REGION Network 14: CYL 6 COUNTER
   RUNG wire#powerrail
      Contact( "AlwaysTRUE" )
      Contact( #ENABLE_CYLINDER[6] )
      Contact( #CYCLE_OK )
      Contact( #CYL_SENSOR6 )
      { S7_Templates := "time_type := Time" } #CYL_STAB_S6.TON(pt := #"SENSING TIME", et =>)
      wire#w1
      Contact( #FIRST_CYCLE )
      P_Trig( #"PLUS BIT"[11] )
      { S7_Templates := "SrcType := Int" } NE_Contact(in1 := #CYL_COUNTER_S6.CV, in2 := #First_Cylinder[6])
      { S7_Templates := "value_type := Int" } #CYL_COUNTER_S6.CTU(r := #"COUNTER RESET", pv := #First_Cylinder[6], cv =>)
   END_RUNG
   RUNG wire#w1
      Contact( #CYCLE_RESTART )
      P_Trig( #"PLUS BIT"[12] )
      { S7_Templates := "SrcType := Int" } NE_Contact(in1 := #CYL_COUNT_CONT_S6.CV, in2 := #"CYL COUNT  VALUE")
      { S7_Templates := "value_type := Int" } #CYL_COUNT_CONT_S6.CTU(r := #"COUNTER RESET", pv := #"CYL COUNT  VALUE", cv =>)
   END_RUNG
   // the same network as SCL:
   #CYL_STAB_S6(IN := "AlwaysTRUE" AND #ENABLE_CYLINDER[6] AND #CYCLE_OK AND #CYL_SENSOR6,   // TON
                PT := #"SENSING TIME");
   #_w1 := #CYL_STAB_S6.Q AND #FIRST_CYCLE;
   #_w2 := #_w1 AND NOT #"PLUS BIT"[11];   // rising edge
   #"PLUS BIT"[11] := #_w1;
   #CYL_COUNTER_S6(CU := #_w2 AND (#CYL_COUNTER_S6.CV <> #First_Cylinder[6]),   // CTU
                   R := #"COUNTER RESET",
                   PV := #First_Cylinder[6]);
   #_w3 := #CYL_STAB_S6.Q AND #CYCLE_RESTART;
   #_w4 := #_w3 AND NOT #"PLUS BIT"[12];   // rising edge
   #"PLUS BIT"[12] := #_w3;
   #CYL_COUNT_CONT_S6(CU := #_w4 AND (#CYL_COUNT_CONT_S6.CV <> #"CYL COUNT  VALUE"),   // CTU
                      R := #"COUNTER RESET",
                      PV := #"CYL COUNT  VALUE");
END_REGION

REGION Network 15: CYL 11 COUNTER
   RUNG wire#powerrail
      Contact( "AlwaysFALSE" )
      Contact( #CYCLE_OK )
      Contact( #"DOWN CONVEYOR" )
      { S7_Templates := "value_type := Int" } #CYL_COUNTER_S11.CTU(r := #"COUNTER RESET", pv := #"CYL COUNT  VALUE", cv =>)
   END_RUNG
   // the same network as SCL:
   #CYL_COUNTER_S11(CU := "AlwaysFALSE" AND #CYCLE_OK AND #"DOWN CONVEYOR",   // CTU
                    R := #"COUNTER RESET",
                    PV := #"CYL COUNT  VALUE");
END_REGION

REGION Network 16: CYL 1 LOCK
   RUNG wire#powerrail
      Contact( "AlwaysTRUE" )
      Contact( #ENABLE_CYLINDER[1] )
      Contact( #CYCLE_OK )
      wire#w1
      Contact( #FIRST_CYCLE )
      { S7_Templates := "SrcType := Int" } EQ_Contact(in1 := #CYL_COUNTER_S1.CV, in2 := #First_Cylinder[1])
      wire#w2
      S_Coil( #"LIFT TABLE1" )
      { S7_Templates := "time_type := Time" } #FILL_STT_1.TON(pt := T#0S, et =>)
      P_Trig( #"PLUS BIT"[31] )
      Contact( #AUTO )
      S_Coil( #FILL_STT_SEQ1 )
   END_RUNG
   RUNG wire#w1
      Contact( #CYCLE_RESTART )
      { S7_Templates := "SrcType := Int" } EQ_Contact(in1 := #CYL_COUNT_CONT_S1.CV, in2 := #"CYL COUNT  VALUE")
   END_RUNG wire#w2
   RUNG wire#w2
      Contact( "Tag_75" )
      S_Coil( #GUN_DOWN1 )
   END_RUNG
   // the same network as SCL:
   #_w1 := "AlwaysTRUE" AND #ENABLE_CYLINDER[1] AND #CYCLE_OK AND ((#FIRST_CYCLE AND (#CYL_COUNTER_S1.CV = #First_Cylinder[1])) OR (#CYCLE_RESTART AND (#CYL_COUNT_CONT_S1.CV = #"CYL COUNT  VALUE")));
   IF #_w1 THEN #"LIFT TABLE1" := TRUE; END_IF;
   #FILL_STT_1(IN := #_w1, PT := T#0S);   // TON
   #_w2 := #FILL_STT_1.Q AND NOT #"PLUS BIT"[31];   // rising edge
   #"PLUS BIT"[31] := #FILL_STT_1.Q;
   IF #_w2 AND #AUTO THEN #FILL_STT_SEQ1 := TRUE; END_IF;
   IF #_w1 AND "Tag_75" THEN #GUN_DOWN1 := TRUE; END_IF;
END_REGION

REGION Network 17: CYL 2 LOCK
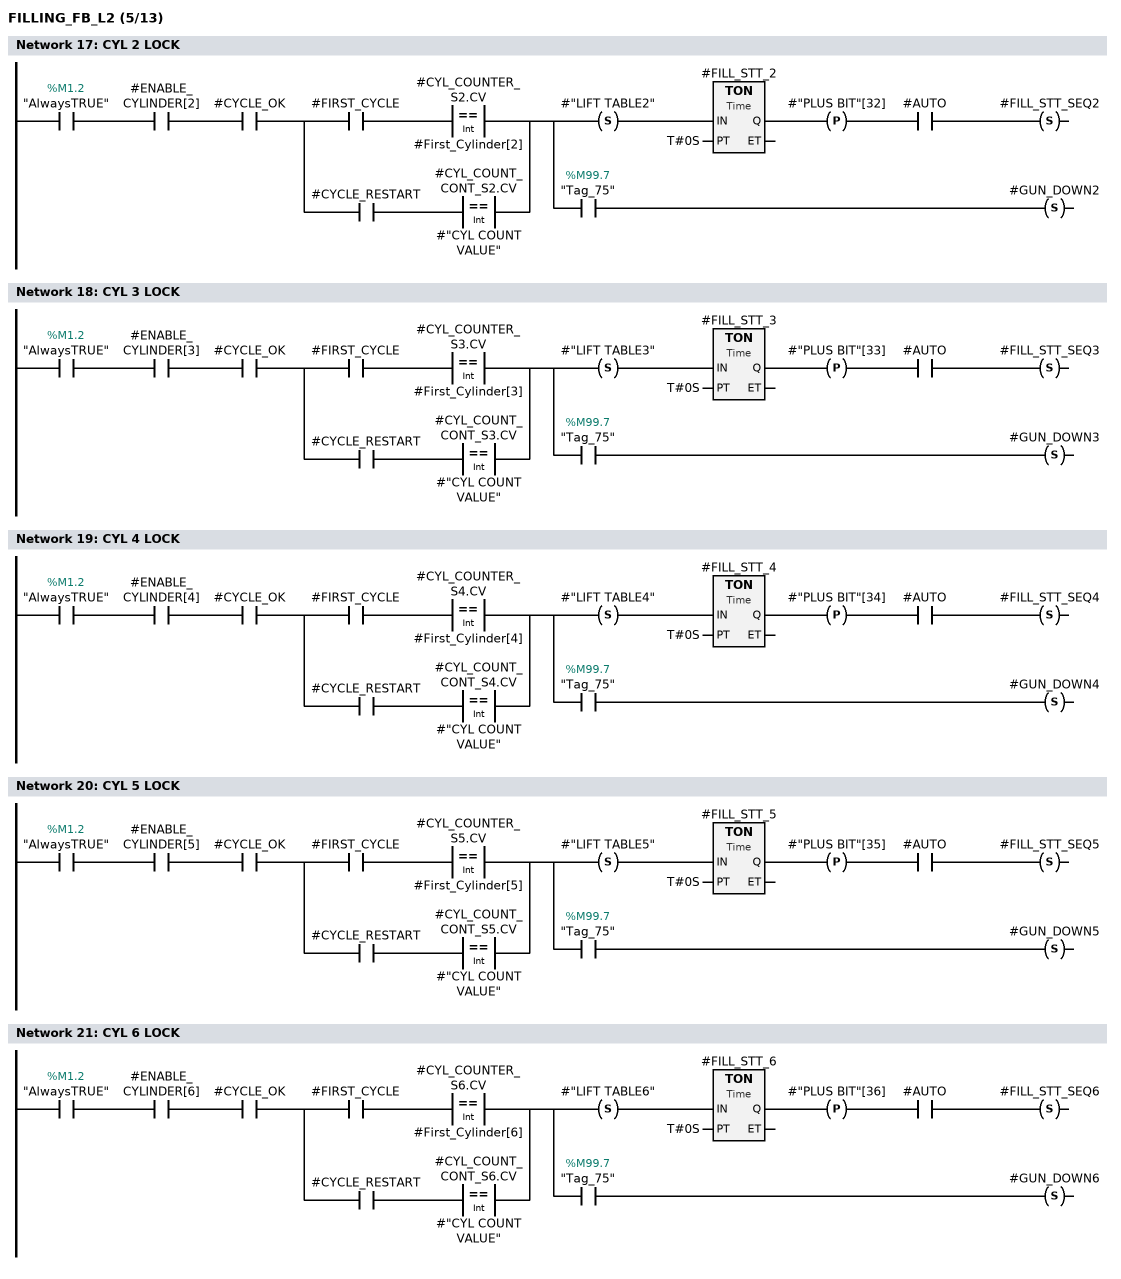
   RUNG wire#powerrail
      Contact( "AlwaysTRUE" )
      Contact( #ENABLE_CYLINDER[2] )
      Contact( #CYCLE_OK )
      wire#w1
      Contact( #FIRST_CYCLE )
      { S7_Templates := "SrcType := Int" } EQ_Contact(in1 := #CYL_COUNTER_S2.CV, in2 := #First_Cylinder[2])
      wire#w2
      S_Coil( #"LIFT TABLE2" )
      { S7_Templates := "time_type := Time" } #FILL_STT_2.TON(pt := T#0S, et =>)
      P_Trig( #"PLUS BIT"[32] )
      Contact( #AUTO )
      S_Coil( #FILL_STT_SEQ2 )
   END_RUNG
   RUNG wire#w1
      Contact( #CYCLE_RESTART )
      { S7_Templates := "SrcType := Int" } EQ_Contact(in1 := #CYL_COUNT_CONT_S2.CV, in2 := #"CYL COUNT  VALUE")
   END_RUNG wire#w2
   RUNG wire#w2
      Contact( "Tag_75" )
      S_Coil( #GUN_DOWN2 )
   END_RUNG
   // the same network as SCL:
   #_w1 := "AlwaysTRUE" AND #ENABLE_CYLINDER[2] AND #CYCLE_OK AND ((#FIRST_CYCLE AND (#CYL_COUNTER_S2.CV = #First_Cylinder[2])) OR (#CYCLE_RESTART AND (#CYL_COUNT_CONT_S2.CV = #"CYL COUNT  VALUE")));
   IF #_w1 THEN #"LIFT TABLE2" := TRUE; END_IF;
   #FILL_STT_2(IN := #_w1, PT := T#0S);   // TON
   #_w2 := #FILL_STT_2.Q AND NOT #"PLUS BIT"[32];   // rising edge
   #"PLUS BIT"[32] := #FILL_STT_2.Q;
   IF #_w2 AND #AUTO THEN #FILL_STT_SEQ2 := TRUE; END_IF;
   IF #_w1 AND "Tag_75" THEN #GUN_DOWN2 := TRUE; END_IF;
END_REGION

REGION Network 18: CYL 3 LOCK
   RUNG wire#powerrail
      Contact( "AlwaysTRUE" )
      Contact( #ENABLE_CYLINDER[3] )
      Contact( #CYCLE_OK )
      wire#w1
      Contact( #FIRST_CYCLE )
      { S7_Templates := "SrcType := Int" } EQ_Contact(in1 := #CYL_COUNTER_S3.CV, in2 := #First_Cylinder[3])
      wire#w2
      S_Coil( #"LIFT TABLE3" )
      { S7_Templates := "time_type := Time" } #FILL_STT_3.TON(pt := T#0S, et =>)
      P_Trig( #"PLUS BIT"[33] )
      Contact( #AUTO )
      S_Coil( #FILL_STT_SEQ3 )
   END_RUNG
   RUNG wire#w1
      Contact( #CYCLE_RESTART )
      { S7_Templates := "SrcType := Int" } EQ_Contact(in1 := #CYL_COUNT_CONT_S3.CV, in2 := #"CYL COUNT  VALUE")
   END_RUNG wire#w2
   RUNG wire#w2
      Contact( "Tag_75" )
      S_Coil( #GUN_DOWN3 )
   END_RUNG
   // the same network as SCL:
   #_w1 := "AlwaysTRUE" AND #ENABLE_CYLINDER[3] AND #CYCLE_OK AND ((#FIRST_CYCLE AND (#CYL_COUNTER_S3.CV = #First_Cylinder[3])) OR (#CYCLE_RESTART AND (#CYL_COUNT_CONT_S3.CV = #"CYL COUNT  VALUE")));
   IF #_w1 THEN #"LIFT TABLE3" := TRUE; END_IF;
   #FILL_STT_3(IN := #_w1, PT := T#0S);   // TON
   #_w2 := #FILL_STT_3.Q AND NOT #"PLUS BIT"[33];   // rising edge
   #"PLUS BIT"[33] := #FILL_STT_3.Q;
   IF #_w2 AND #AUTO THEN #FILL_STT_SEQ3 := TRUE; END_IF;
   IF #_w1 AND "Tag_75" THEN #GUN_DOWN3 := TRUE; END_IF;
END_REGION

REGION Network 19: CYL 4 LOCK
   RUNG wire#powerrail
      Contact( "AlwaysTRUE" )
      Contact( #ENABLE_CYLINDER[4] )
      Contact( #CYCLE_OK )
      wire#w1
      Contact( #FIRST_CYCLE )
      { S7_Templates := "SrcType := Int" } EQ_Contact(in1 := #CYL_COUNTER_S4.CV, in2 := #First_Cylinder[4])
      wire#w2
      S_Coil( #"LIFT TABLE4" )
      { S7_Templates := "time_type := Time" } #FILL_STT_4.TON(pt := T#0S, et =>)
      P_Trig( #"PLUS BIT"[34] )
      Contact( #AUTO )
      S_Coil( #FILL_STT_SEQ4 )
   END_RUNG
   RUNG wire#w1
      Contact( #CYCLE_RESTART )
      { S7_Templates := "SrcType := Int" } EQ_Contact(in1 := #CYL_COUNT_CONT_S4.CV, in2 := #"CYL COUNT  VALUE")
   END_RUNG wire#w2
   RUNG wire#w2
      Contact( "Tag_75" )
      S_Coil( #GUN_DOWN4 )
   END_RUNG
   // the same network as SCL:
   #_w1 := "AlwaysTRUE" AND #ENABLE_CYLINDER[4] AND #CYCLE_OK AND ((#FIRST_CYCLE AND (#CYL_COUNTER_S4.CV = #First_Cylinder[4])) OR (#CYCLE_RESTART AND (#CYL_COUNT_CONT_S4.CV = #"CYL COUNT  VALUE")));
   IF #_w1 THEN #"LIFT TABLE4" := TRUE; END_IF;
   #FILL_STT_4(IN := #_w1, PT := T#0S);   // TON
   #_w2 := #FILL_STT_4.Q AND NOT #"PLUS BIT"[34];   // rising edge
   #"PLUS BIT"[34] := #FILL_STT_4.Q;
   IF #_w2 AND #AUTO THEN #FILL_STT_SEQ4 := TRUE; END_IF;
   IF #_w1 AND "Tag_75" THEN #GUN_DOWN4 := TRUE; END_IF;
END_REGION

REGION Network 20: CYL 5 LOCK
   RUNG wire#powerrail
      Contact( "AlwaysTRUE" )
      Contact( #ENABLE_CYLINDER[5] )
      Contact( #CYCLE_OK )
      wire#w1
      Contact( #FIRST_CYCLE )
      { S7_Templates := "SrcType := Int" } EQ_Contact(in1 := #CYL_COUNTER_S5.CV, in2 := #First_Cylinder[5])
      wire#w2
      S_Coil( #"LIFT TABLE5" )
      { S7_Templates := "time_type := Time" } #FILL_STT_5.TON(pt := T#0S, et =>)
      P_Trig( #"PLUS BIT"[35] )
      Contact( #AUTO )
      S_Coil( #FILL_STT_SEQ5 )
   END_RUNG
   RUNG wire#w1
      Contact( #CYCLE_RESTART )
      { S7_Templates := "SrcType := Int" } EQ_Contact(in1 := #CYL_COUNT_CONT_S5.CV, in2 := #"CYL COUNT  VALUE")
   END_RUNG wire#w2
   RUNG wire#w2
      Contact( "Tag_75" )
      S_Coil( #GUN_DOWN5 )
   END_RUNG
   // the same network as SCL:
   #_w1 := "AlwaysTRUE" AND #ENABLE_CYLINDER[5] AND #CYCLE_OK AND ((#FIRST_CYCLE AND (#CYL_COUNTER_S5.CV = #First_Cylinder[5])) OR (#CYCLE_RESTART AND (#CYL_COUNT_CONT_S5.CV = #"CYL COUNT  VALUE")));
   IF #_w1 THEN #"LIFT TABLE5" := TRUE; END_IF;
   #FILL_STT_5(IN := #_w1, PT := T#0S);   // TON
   #_w2 := #FILL_STT_5.Q AND NOT #"PLUS BIT"[35];   // rising edge
   #"PLUS BIT"[35] := #FILL_STT_5.Q;
   IF #_w2 AND #AUTO THEN #FILL_STT_SEQ5 := TRUE; END_IF;
   IF #_w1 AND "Tag_75" THEN #GUN_DOWN5 := TRUE; END_IF;
END_REGION

REGION Network 21: CYL 6 LOCK
   RUNG wire#powerrail
      Contact( "AlwaysTRUE" )
      Contact( #ENABLE_CYLINDER[6] )
      Contact( #CYCLE_OK )
      wire#w1
      Contact( #FIRST_CYCLE )
      { S7_Templates := "SrcType := Int" } EQ_Contact(in1 := #CYL_COUNTER_S6.CV, in2 := #First_Cylinder[6])
      wire#w2
      S_Coil( #"LIFT TABLE6" )
      { S7_Templates := "time_type := Time" } #FILL_STT_6.TON(pt := T#0S, et =>)
      P_Trig( #"PLUS BIT"[36] )
      Contact( #AUTO )
      S_Coil( #FILL_STT_SEQ6 )
   END_RUNG
   RUNG wire#w1
      Contact( #CYCLE_RESTART )
      { S7_Templates := "SrcType := Int" } EQ_Contact(in1 := #CYL_COUNT_CONT_S6.CV, in2 := #"CYL COUNT  VALUE")
   END_RUNG wire#w2
   RUNG wire#w2
      Contact( "Tag_75" )
      S_Coil( #GUN_DOWN6 )
   END_RUNG
   // the same network as SCL:
   #_w1 := "AlwaysTRUE" AND #ENABLE_CYLINDER[6] AND #CYCLE_OK AND ((#FIRST_CYCLE AND (#CYL_COUNTER_S6.CV = #First_Cylinder[6])) OR (#CYCLE_RESTART AND (#CYL_COUNT_CONT_S6.CV = #"CYL COUNT  VALUE")));
   IF #_w1 THEN #"LIFT TABLE6" := TRUE; END_IF;
   #FILL_STT_6(IN := #_w1, PT := T#0S);   // TON
   #_w2 := #FILL_STT_6.Q AND NOT #"PLUS BIT"[36];   // rising edge
   #"PLUS BIT"[36] := #FILL_STT_6.Q;
   IF #_w2 AND #AUTO THEN #FILL_STT_SEQ6 := TRUE; END_IF;
   IF #_w1 AND "Tag_75" THEN #GUN_DOWN6 := TRUE; END_IF;
END_REGION

REGION Network 22: TIMER TIME MULTIFLY
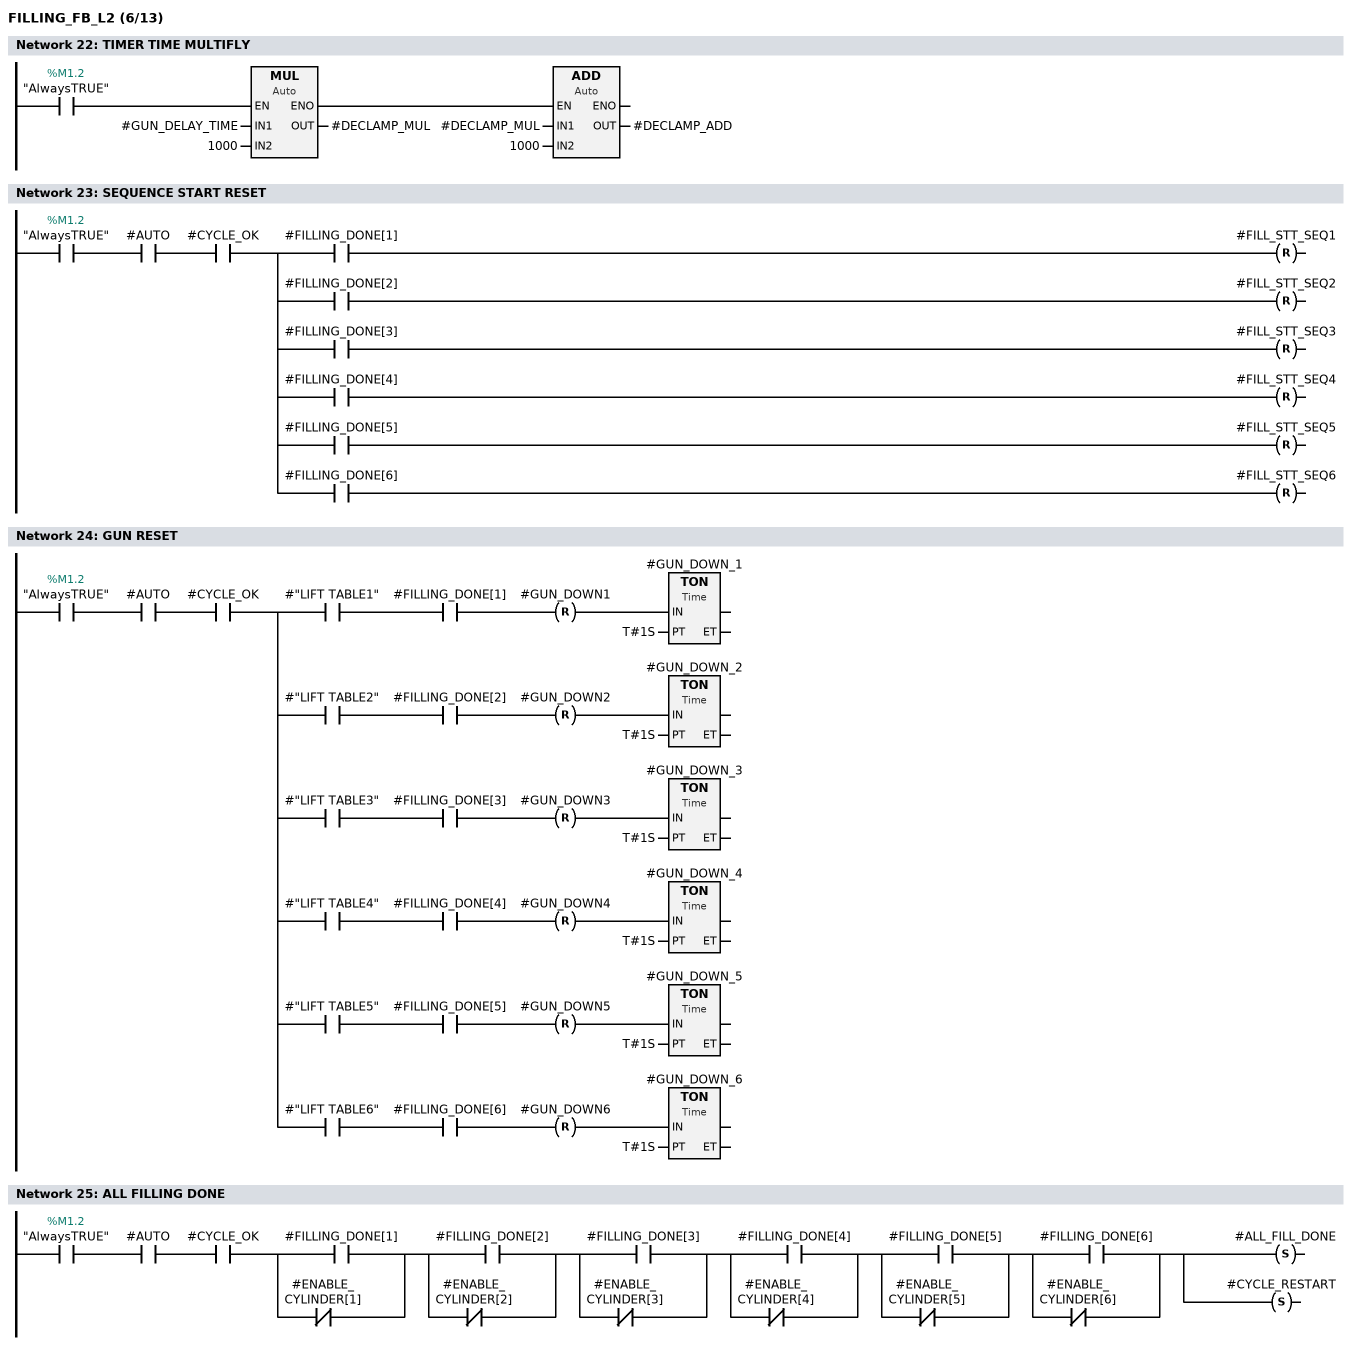
   RUNG wire#powerrail
      Contact( "AlwaysTRUE" )
      Mul(in1 := #GUN_DELAY_TIME, in2 := 1000, out => #DECLAMP_MUL)
      Add(in1 := #DECLAMP_MUL, in2 := 1000, out => #DECLAMP_ADD)
   END_RUNG
   // the same network as SCL:
   IF "AlwaysTRUE" THEN
       #DECLAMP_MUL := #GUN_DELAY_TIME * 1000;
       #DECLAMP_ADD := #DECLAMP_MUL + 1000;
   END_IF;
END_REGION

REGION Network 23: SEQUENCE START RESET
   RUNG wire#powerrail
      Contact( "AlwaysTRUE" )
      Contact( #AUTO )
      Contact( #CYCLE_OK )
      wire#w1
      Contact( #FILLING_DONE[1] )
      R_Coil( #FILL_STT_SEQ1 )
   END_RUNG
   RUNG wire#w1
      Contact( #FILLING_DONE[2] )
      R_Coil( #FILL_STT_SEQ2 )
   END_RUNG
   RUNG wire#w1
      Contact( #FILLING_DONE[3] )
      R_Coil( #FILL_STT_SEQ3 )
   END_RUNG
   RUNG wire#w1
      Contact( #FILLING_DONE[4] )
      R_Coil( #FILL_STT_SEQ4 )
   END_RUNG
   RUNG wire#w1
      Contact( #FILLING_DONE[5] )
      R_Coil( #FILL_STT_SEQ5 )
   END_RUNG
   RUNG wire#w1
      Contact( #FILLING_DONE[6] )
      R_Coil( #FILL_STT_SEQ6 )
   END_RUNG
   // the same network as SCL:
   #_w1 := "AlwaysTRUE" AND #AUTO AND #CYCLE_OK;
   IF #_w1 AND #FILLING_DONE[1] THEN #FILL_STT_SEQ1 := FALSE; END_IF;
   IF #_w1 AND #FILLING_DONE[2] THEN #FILL_STT_SEQ2 := FALSE; END_IF;
   IF #_w1 AND #FILLING_DONE[3] THEN #FILL_STT_SEQ3 := FALSE; END_IF;
   IF #_w1 AND #FILLING_DONE[4] THEN #FILL_STT_SEQ4 := FALSE; END_IF;
   IF #_w1 AND #FILLING_DONE[5] THEN #FILL_STT_SEQ5 := FALSE; END_IF;
   IF #_w1 AND #FILLING_DONE[6] THEN #FILL_STT_SEQ6 := FALSE; END_IF;
END_REGION

REGION Network 24: GUN RESET
   RUNG wire#powerrail
      Contact( "AlwaysTRUE" )
      Contact( #AUTO )
      Contact( #CYCLE_OK )
      wire#w1
      Contact( #"LIFT TABLE1" )
      Contact( #FILLING_DONE[1] )
      R_Coil( #GUN_DOWN1 )
      { S7_Templates := "time_type := Time" } #GUN_DOWN_1.TON(pt := T#1S, et =>)
   END_RUNG
   RUNG wire#w1
      Contact( #"LIFT TABLE2" )
      Contact( #FILLING_DONE[2] )
      R_Coil( #GUN_DOWN2 )
      { S7_Templates := "time_type := Time" } #GUN_DOWN_2.TON(pt := T#1S, et =>)
   END_RUNG
   RUNG wire#w1
      Contact( #"LIFT TABLE3" )
      Contact( #FILLING_DONE[3] )
      R_Coil( #GUN_DOWN3 )
      { S7_Templates := "time_type := Time" } #GUN_DOWN_3.TON(pt := T#1S, et =>)
   END_RUNG
   RUNG wire#w1
      Contact( #"LIFT TABLE4" )
      Contact( #FILLING_DONE[4] )
      R_Coil( #GUN_DOWN4 )
      { S7_Templates := "time_type := Time" } #GUN_DOWN_4.TON(pt := T#1S, et =>)
   END_RUNG
   RUNG wire#w1
      Contact( #"LIFT TABLE5" )
      Contact( #FILLING_DONE[5] )
      R_Coil( #GUN_DOWN5 )
      { S7_Templates := "time_type := Time" } #GUN_DOWN_5.TON(pt := T#1S, et =>)
   END_RUNG
   RUNG wire#w1
      Contact( #"LIFT TABLE6" )
      Contact( #FILLING_DONE[6] )
      R_Coil( #GUN_DOWN6 )
      { S7_Templates := "time_type := Time" } #GUN_DOWN_6.TON(pt := T#1S, et =>)
   END_RUNG
   // the same network as SCL:
   #_w1 := "AlwaysTRUE" AND #AUTO AND #CYCLE_OK;
   #_w2 := #_w1 AND #"LIFT TABLE1" AND #FILLING_DONE[1];
   IF #_w2 THEN #GUN_DOWN1 := FALSE; END_IF;
   #GUN_DOWN_1(IN := #_w2, PT := T#1S);   // TON
   #_w3 := #_w1 AND #"LIFT TABLE2" AND #FILLING_DONE[2];
   IF #_w3 THEN #GUN_DOWN2 := FALSE; END_IF;
   #GUN_DOWN_2(IN := #_w3, PT := T#1S);   // TON
   #_w4 := #_w1 AND #"LIFT TABLE3" AND #FILLING_DONE[3];
   IF #_w4 THEN #GUN_DOWN3 := FALSE; END_IF;
   #GUN_DOWN_3(IN := #_w4, PT := T#1S);   // TON
   #_w5 := #_w1 AND #"LIFT TABLE4" AND #FILLING_DONE[4];
   IF #_w5 THEN #GUN_DOWN4 := FALSE; END_IF;
   #GUN_DOWN_4(IN := #_w5, PT := T#1S);   // TON
   #_w6 := #_w1 AND #"LIFT TABLE5" AND #FILLING_DONE[5];
   IF #_w6 THEN #GUN_DOWN5 := FALSE; END_IF;
   #GUN_DOWN_5(IN := #_w6, PT := T#1S);   // TON
   #_w7 := #_w1 AND #"LIFT TABLE6" AND #FILLING_DONE[6];
   IF #_w7 THEN #GUN_DOWN6 := FALSE; END_IF;
   #GUN_DOWN_6(IN := #_w7, PT := T#1S);   // TON
END_REGION

REGION Network 25: ALL FILLING DONE
   RUNG wire#powerrail
      Contact( "AlwaysTRUE" )
      Contact( #AUTO )
      Contact( #CYCLE_OK )
      wire#w1
      Contact( #FILLING_DONE[1] )
      wire#w2
      Contact( #FILLING_DONE[2] )
      wire#w3
      Contact( #FILLING_DONE[3] )
      wire#w4
      Contact( #FILLING_DONE[4] )
      wire#w5
      Contact( #FILLING_DONE[5] )
      wire#w6
      Contact( #FILLING_DONE[6] )
      wire#w7
      S_Coil( #ALL_FILL_DONE )
   END_RUNG
   RUNG wire#w1
      I_Contact( #ENABLE_CYLINDER[1] )
   END_RUNG wire#w2
   RUNG wire#w2
      I_Contact( #ENABLE_CYLINDER[2] )
   END_RUNG wire#w3
   RUNG wire#w3
      I_Contact( #ENABLE_CYLINDER[3] )
   END_RUNG wire#w4
   RUNG wire#w4
      I_Contact( #ENABLE_CYLINDER[4] )
   END_RUNG wire#w5
   RUNG wire#w5
      I_Contact( #ENABLE_CYLINDER[5] )
   END_RUNG wire#w6
   RUNG wire#w6
      I_Contact( #ENABLE_CYLINDER[6] )
   END_RUNG wire#w7
   RUNG wire#w7
      S_Coil( #CYCLE_RESTART )
   END_RUNG
   // the same network as SCL:
   IF "AlwaysTRUE" AND #AUTO AND #CYCLE_OK AND (#FILLING_DONE[1] OR NOT #ENABLE_CYLINDER[1]) AND (#FILLING_DONE[2] OR NOT #ENABLE_CYLINDER[2]) AND (#FILLING_DONE[3] OR NOT #ENABLE_CYLINDER[3]) AND (#FILLING_DONE[4] OR NOT #ENABLE_CYLINDER[4]) AND (#FILLING_DONE[5] OR NOT #ENABLE_CYLINDER[5]) AND (#FILLING_DONE[6] OR NOT #ENABLE_CYLINDER[6]) THEN
       #ALL_FILL_DONE := TRUE;
       #CYCLE_RESTART := TRUE;
   END_IF;
END_REGION

REGION Network 26: ALL GUN UP
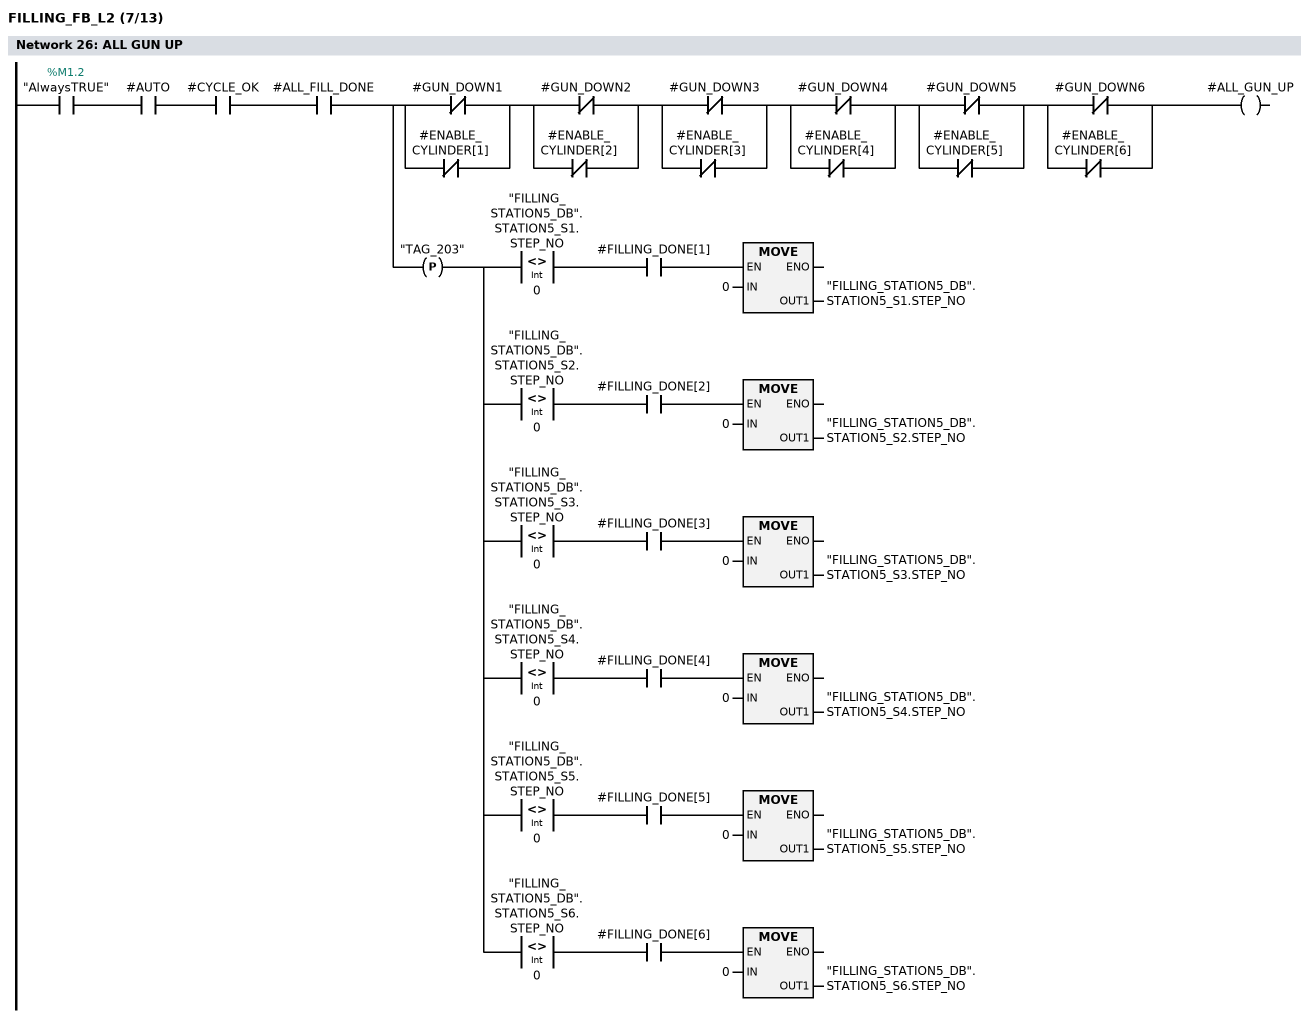
   RUNG wire#powerrail
      Contact( "AlwaysTRUE" )
      Contact( #AUTO )
      Contact( #CYCLE_OK )
      Contact( #ALL_FILL_DONE )
      wire#w1
      I_Contact( #GUN_DOWN1 )
      wire#w2
      I_Contact( #GUN_DOWN2 )
      wire#w3
      I_Contact( #GUN_DOWN3 )
      wire#w4
      I_Contact( #GUN_DOWN4 )
      wire#w5
      I_Contact( #GUN_DOWN5 )
      wire#w6
      I_Contact( #GUN_DOWN6 )
      wire#w7
      Coil( #ALL_GUN_UP )
   END_RUNG
   RUNG wire#w1
      I_Contact( #ENABLE_CYLINDER[1] )
   END_RUNG wire#w2
   RUNG wire#w2
      I_Contact( #ENABLE_CYLINDER[2] )
   END_RUNG wire#w3
   RUNG wire#w3
      I_Contact( #ENABLE_CYLINDER[3] )
   END_RUNG wire#w4
   RUNG wire#w4
      I_Contact( #ENABLE_CYLINDER[4] )
   END_RUNG wire#w5
   RUNG wire#w5
      I_Contact( #ENABLE_CYLINDER[5] )
   END_RUNG wire#w6
   RUNG wire#w6
      I_Contact( #ENABLE_CYLINDER[6] )
   END_RUNG wire#w7
   RUNG wire#w1
      P_Trig( "TAG_203" )
      wire#w8
      { S7_Templates := "SrcType := Int" } NE_Contact(in1 := "FILLING_STATION5_DB".STATION5_S1.STEP_NO, in2 := 0)
      Contact( #FILLING_DONE[1] )
      Move(in := 0, out1 => "FILLING_STATION5_DB".STATION5_S1.STEP_NO)
   END_RUNG
   RUNG wire#w8
      { S7_Templates := "SrcType := Int" } NE_Contact(in1 := "FILLING_STATION5_DB".STATION5_S2.STEP_NO, in2 := 0)
      Contact( #FILLING_DONE[2] )
      Move(in := 0, out1 => "FILLING_STATION5_DB".STATION5_S2.STEP_NO)
   END_RUNG
   RUNG wire#w8
      { S7_Templates := "SrcType := Int" } NE_Contact(in1 := "FILLING_STATION5_DB".STATION5_S3.STEP_NO, in2 := 0)
      Contact( #FILLING_DONE[3] )
      Move(in := 0, out1 => "FILLING_STATION5_DB".STATION5_S3.STEP_NO)
   END_RUNG
   RUNG wire#w8
      { S7_Templates := "SrcType := Int" } NE_Contact(in1 := "FILLING_STATION5_DB".STATION5_S4.STEP_NO, in2 := 0)
      Contact( #FILLING_DONE[4] )
      Move(in := 0, out1 => "FILLING_STATION5_DB".STATION5_S4.STEP_NO)
   END_RUNG
   RUNG wire#w8
      { S7_Templates := "SrcType := Int" } NE_Contact(in1 := "FILLING_STATION5_DB".STATION5_S5.STEP_NO, in2 := 0)
      Contact( #FILLING_DONE[5] )
      Move(in := 0, out1 => "FILLING_STATION5_DB".STATION5_S5.STEP_NO)
   END_RUNG
   RUNG wire#w8
      { S7_Templates := "SrcType := Int" } NE_Contact(in1 := "FILLING_STATION5_DB".STATION5_S6.STEP_NO, in2 := 0)
      Contact( #FILLING_DONE[6] )
      Move(in := 0, out1 => "FILLING_STATION5_DB".STATION5_S6.STEP_NO)
   END_RUNG
   // the same network as SCL:
   #_w1 := "AlwaysTRUE" AND #AUTO AND #CYCLE_OK AND #ALL_FILL_DONE;
   #ALL_GUN_UP := #_w1 AND (NOT #GUN_DOWN1 OR NOT #ENABLE_CYLINDER[1]) AND (NOT #GUN_DOWN2 OR NOT #ENABLE_CYLINDER[2]) AND (NOT #GUN_DOWN3 OR NOT #ENABLE_CYLINDER[3]) AND (NOT #GUN_DOWN4 OR NOT #ENABLE_CYLINDER[4]) AND (NOT #GUN_DOWN5 OR NOT #ENABLE_CYLINDER[5]) AND (NOT #GUN_DOWN6 OR NOT #ENABLE_CYLINDER[6]);
   #_w2 := #_w1 AND NOT "TAG_203";   // rising edge
   "TAG_203" := #_w1;
   IF #_w2 AND ("FILLING_STATION5_DB".STATION5_S1.STEP_NO <> 0) AND #FILLING_DONE[1] THEN
       "FILLING_STATION5_DB".STATION5_S1.STEP_NO := 0;
   END_IF;
   IF #_w2 AND ("FILLING_STATION5_DB".STATION5_S2.STEP_NO <> 0) AND #FILLING_DONE[2] THEN
       "FILLING_STATION5_DB".STATION5_S2.STEP_NO := 0;
   END_IF;
   IF #_w2 AND ("FILLING_STATION5_DB".STATION5_S3.STEP_NO <> 0) AND #FILLING_DONE[3] THEN
       "FILLING_STATION5_DB".STATION5_S3.STEP_NO := 0;
   END_IF;
   IF #_w2 AND ("FILLING_STATION5_DB".STATION5_S4.STEP_NO <> 0) AND #FILLING_DONE[4] THEN
       "FILLING_STATION5_DB".STATION5_S4.STEP_NO := 0;
   END_IF;
   IF #_w2 AND ("FILLING_STATION5_DB".STATION5_S5.STEP_NO <> 0) AND #FILLING_DONE[5] THEN
       "FILLING_STATION5_DB".STATION5_S5.STEP_NO := 0;
   END_IF;
   IF #_w2 AND ("FILLING_STATION5_DB".STATION5_S6.STEP_NO <> 0) AND #FILLING_DONE[6] THEN
       "FILLING_STATION5_DB".STATION5_S6.STEP_NO := 0;
   END_IF;
END_REGION

REGION Network 27: CYCLE COMPLETED
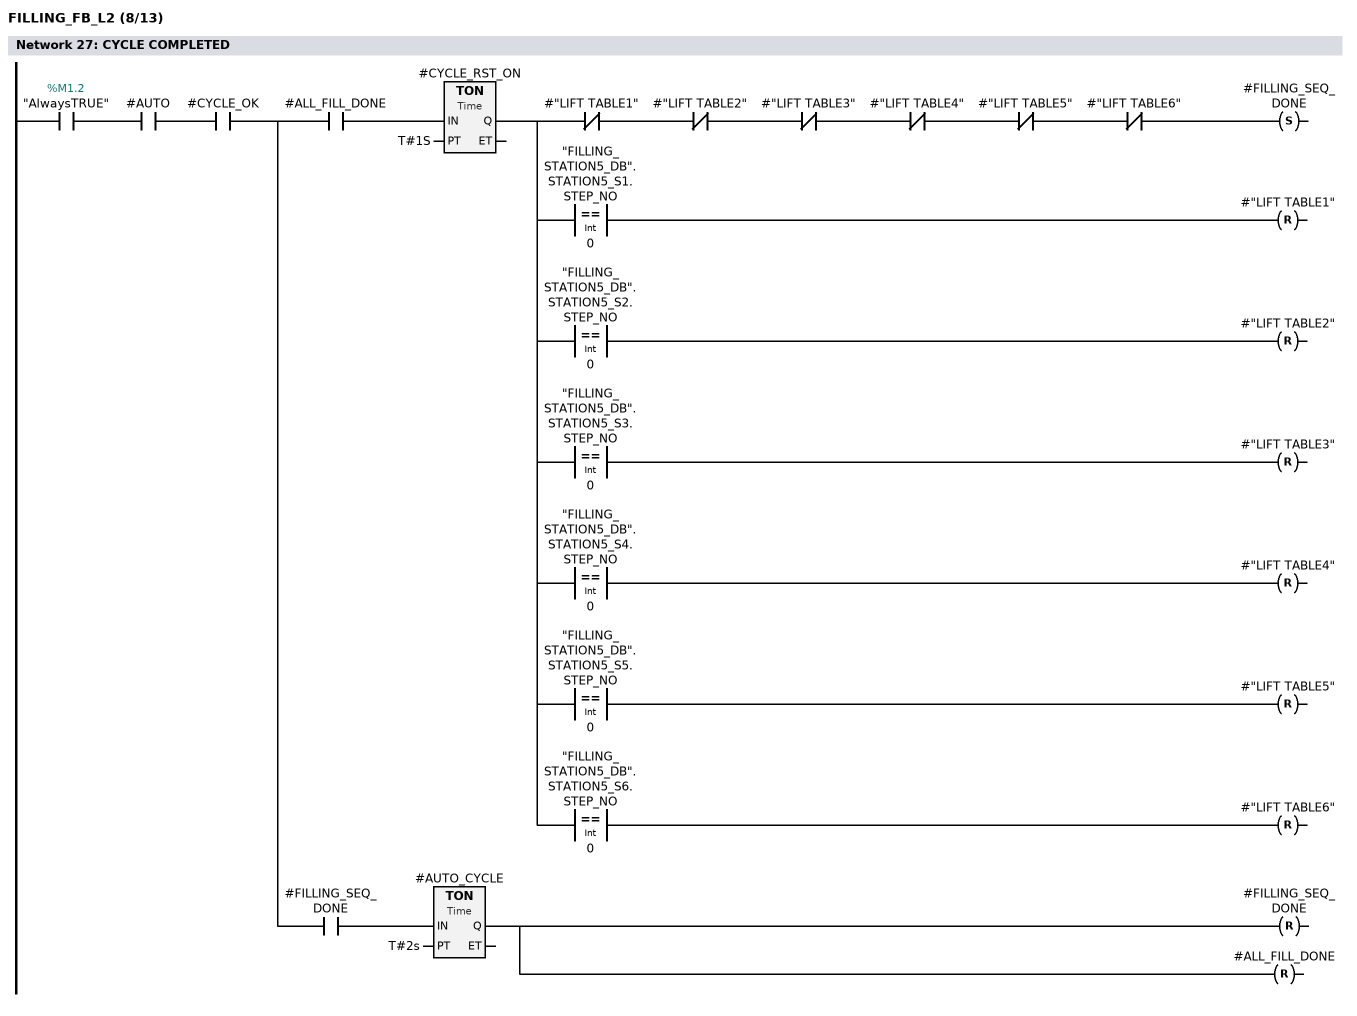
   RUNG wire#powerrail
      Contact( "AlwaysTRUE" )
      Contact( #AUTO )
      Contact( #CYCLE_OK )
      wire#w1
      Contact( #ALL_FILL_DONE )
      { S7_Templates := "time_type := Time" } #CYCLE_RST_ON.TON(pt := T#1S, et =>)
      wire#w2
      I_Contact( #"LIFT TABLE1" )
      I_Contact( #"LIFT TABLE2" )
      I_Contact( #"LIFT TABLE3" )
      I_Contact( #"LIFT TABLE4" )
      I_Contact( #"LIFT TABLE5" )
      I_Contact( #"LIFT TABLE6" )
      S_Coil( #FILLING_SEQ_DONE )
   END_RUNG
   RUNG wire#w2
      { S7_Templates := "SrcType := Int" } EQ_Contact(in1 := "FILLING_STATION5_DB".STATION5_S1.STEP_NO, in2 := 0)
      R_Coil( #"LIFT TABLE1" )
   END_RUNG
   RUNG wire#w2
      { S7_Templates := "SrcType := Int" } EQ_Contact(in1 := "FILLING_STATION5_DB".STATION5_S2.STEP_NO, in2 := 0)
      R_Coil( #"LIFT TABLE2" )
   END_RUNG
   RUNG wire#w2
      { S7_Templates := "SrcType := Int" } EQ_Contact(in1 := "FILLING_STATION5_DB".STATION5_S3.STEP_NO, in2 := 0)
      R_Coil( #"LIFT TABLE3" )
   END_RUNG
   RUNG wire#w2
      { S7_Templates := "SrcType := Int" } EQ_Contact(in1 := "FILLING_STATION5_DB".STATION5_S4.STEP_NO, in2 := 0)
      R_Coil( #"LIFT TABLE4" )
   END_RUNG
   RUNG wire#w2
      { S7_Templates := "SrcType := Int" } EQ_Contact(in1 := "FILLING_STATION5_DB".STATION5_S5.STEP_NO, in2 := 0)
      R_Coil( #"LIFT TABLE5" )
   END_RUNG
   RUNG wire#w2
      { S7_Templates := "SrcType := Int" } EQ_Contact(in1 := "FILLING_STATION5_DB".STATION5_S6.STEP_NO, in2 := 0)
      R_Coil( #"LIFT TABLE6" )
   END_RUNG
   RUNG wire#w1
      Contact( #FILLING_SEQ_DONE )
      { S7_Templates := "time_type := Time" } #AUTO_CYCLE.TON(pt := T#2s, et =>)
      wire#w3
      R_Coil( #FILLING_SEQ_DONE )
   END_RUNG
   RUNG wire#w3
      R_Coil( #ALL_FILL_DONE )
   END_RUNG
   // the same network as SCL:
   #_w1 := "AlwaysTRUE" AND #AUTO AND #CYCLE_OK;
   #CYCLE_RST_ON(IN := #_w1 AND #ALL_FILL_DONE, PT := T#1S);   // TON
   IF #CYCLE_RST_ON.Q AND NOT #"LIFT TABLE1" AND NOT #"LIFT TABLE2" AND NOT #"LIFT TABLE3" AND NOT #"LIFT TABLE4" AND NOT #"LIFT TABLE5" AND NOT #"LIFT TABLE6" THEN
       #FILLING_SEQ_DONE := TRUE;
   END_IF;
   IF #CYCLE_RST_ON.Q AND ("FILLING_STATION5_DB".STATION5_S1.STEP_NO = 0) THEN
       #"LIFT TABLE1" := FALSE;
   END_IF;
   IF #CYCLE_RST_ON.Q AND ("FILLING_STATION5_DB".STATION5_S2.STEP_NO = 0) THEN
       #"LIFT TABLE2" := FALSE;
   END_IF;
   IF #CYCLE_RST_ON.Q AND ("FILLING_STATION5_DB".STATION5_S3.STEP_NO = 0) THEN
       #"LIFT TABLE3" := FALSE;
   END_IF;
   IF #CYCLE_RST_ON.Q AND ("FILLING_STATION5_DB".STATION5_S4.STEP_NO = 0) THEN
       #"LIFT TABLE4" := FALSE;
   END_IF;
   IF #CYCLE_RST_ON.Q AND ("FILLING_STATION5_DB".STATION5_S5.STEP_NO = 0) THEN
       #"LIFT TABLE5" := FALSE;
   END_IF;
   IF #CYCLE_RST_ON.Q AND ("FILLING_STATION5_DB".STATION5_S6.STEP_NO = 0) THEN
       #"LIFT TABLE6" := FALSE;
   END_IF;
   #AUTO_CYCLE(IN := #_w1 AND #FILLING_SEQ_DONE, PT := T#2s);   // TON
   IF #AUTO_CYCLE.Q THEN
       #FILLING_SEQ_DONE := FALSE;
       #ALL_FILL_DONE := FALSE;
   END_IF;
END_REGION

REGION Network 28: CYCLE RESET
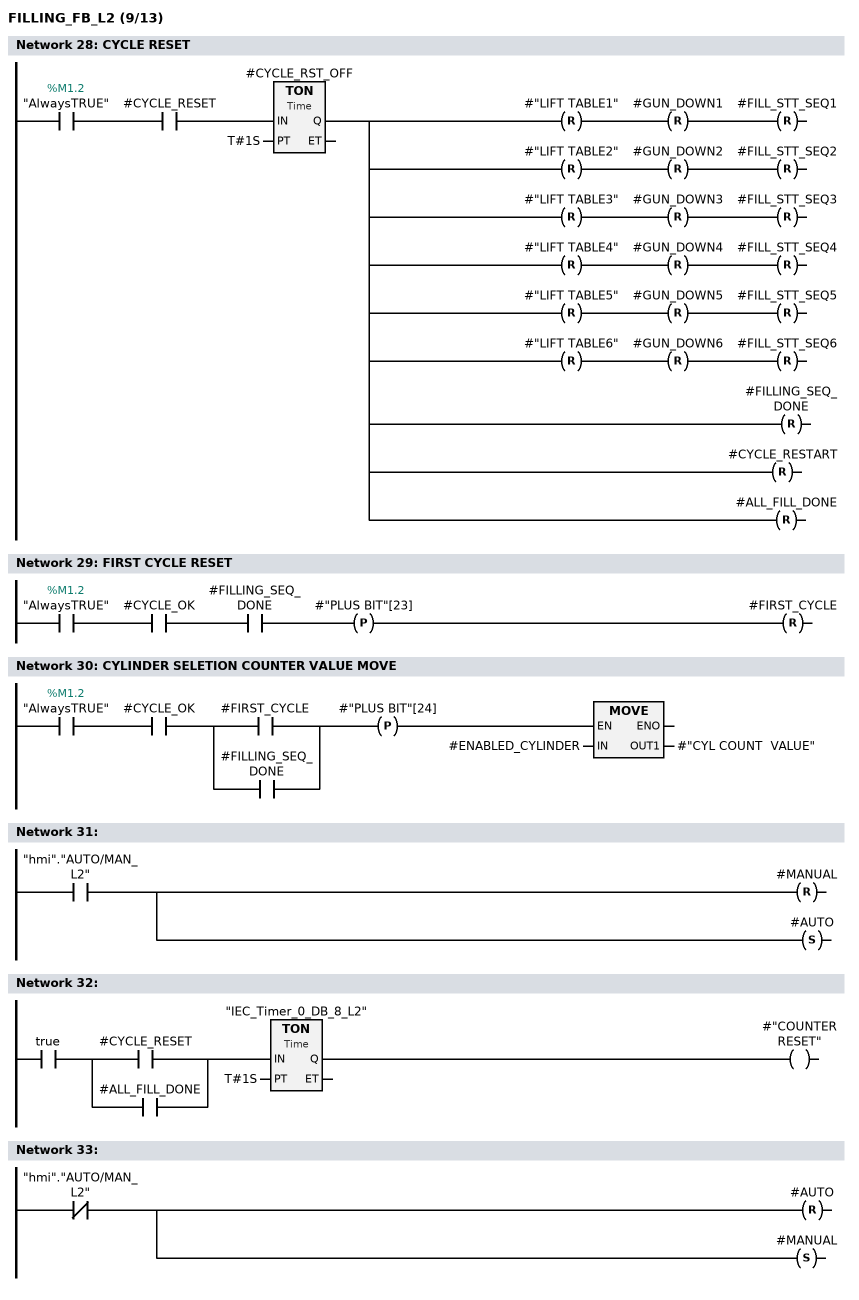
   RUNG wire#powerrail
      Contact( "AlwaysTRUE" )
      Contact( #CYCLE_RESET )
      { S7_Templates := "time_type := Time" } #CYCLE_RST_OFF.TON(pt := T#1S, et =>)
      wire#w1
      R_Coil( #"LIFT TABLE1" )
      R_Coil( #GUN_DOWN1 )
      R_Coil( #FILL_STT_SEQ1 )
   END_RUNG
   RUNG wire#w1
      R_Coil( #"LIFT TABLE2" )
      R_Coil( #GUN_DOWN2 )
      R_Coil( #FILL_STT_SEQ2 )
   END_RUNG
   RUNG wire#w1
      R_Coil( #"LIFT TABLE3" )
      R_Coil( #GUN_DOWN3 )
      R_Coil( #FILL_STT_SEQ3 )
   END_RUNG
   RUNG wire#w1
      R_Coil( #"LIFT TABLE4" )
      R_Coil( #GUN_DOWN4 )
      R_Coil( #FILL_STT_SEQ4 )
   END_RUNG
   RUNG wire#w1
      R_Coil( #"LIFT TABLE5" )
      R_Coil( #GUN_DOWN5 )
      R_Coil( #FILL_STT_SEQ5 )
   END_RUNG
   RUNG wire#w1
      R_Coil( #"LIFT TABLE6" )
      R_Coil( #GUN_DOWN6 )
      R_Coil( #FILL_STT_SEQ6 )
   END_RUNG
   RUNG wire#w1
      R_Coil( #FILLING_SEQ_DONE )
   END_RUNG
   RUNG wire#w1
      R_Coil( #CYCLE_RESTART )
   END_RUNG
   RUNG wire#w1
      R_Coil( #ALL_FILL_DONE )
   END_RUNG
   // the same network as SCL:
   #CYCLE_RST_OFF(IN := "AlwaysTRUE" AND #CYCLE_RESET, PT := T#1S);   // TON
   IF #CYCLE_RST_OFF.Q THEN
       #"LIFT TABLE1" := FALSE;
       #GUN_DOWN1 := FALSE;
       #FILL_STT_SEQ1 := FALSE;
       #"LIFT TABLE2" := FALSE;
       #GUN_DOWN2 := FALSE;
       #FILL_STT_SEQ2 := FALSE;
       #"LIFT TABLE3" := FALSE;
       #GUN_DOWN3 := FALSE;
       #FILL_STT_SEQ3 := FALSE;
       #"LIFT TABLE4" := FALSE;
       #GUN_DOWN4 := FALSE;
       #FILL_STT_SEQ4 := FALSE;
       #"LIFT TABLE5" := FALSE;
       #GUN_DOWN5 := FALSE;
       #FILL_STT_SEQ5 := FALSE;
       #"LIFT TABLE6" := FALSE;
       #GUN_DOWN6 := FALSE;
       #FILL_STT_SEQ6 := FALSE;
       #FILLING_SEQ_DONE := FALSE;
       #CYCLE_RESTART := FALSE;
       #ALL_FILL_DONE := FALSE;
   END_IF;
END_REGION

REGION Network 29: FIRST CYCLE RESET
   RUNG wire#powerrail
      Contact( "AlwaysTRUE" )
      Contact( #CYCLE_OK )
      Contact( #FILLING_SEQ_DONE )
      P_Trig( #"PLUS BIT"[23] )
      R_Coil( #FIRST_CYCLE )
   END_RUNG
   // the same network as SCL:
   #_w1 := "AlwaysTRUE" AND #CYCLE_OK AND #FILLING_SEQ_DONE;
   #_w2 := #_w1 AND NOT #"PLUS BIT"[23];   // rising edge
   #"PLUS BIT"[23] := #_w1;
   IF #_w2 THEN #FIRST_CYCLE := FALSE; END_IF;
END_REGION

REGION Network 30: CYLINDER SELETION COUNTER VALUE MOVE
   RUNG wire#powerrail
      Contact( "AlwaysTRUE" )
      Contact( #CYCLE_OK )
      wire#w1
      Contact( #FIRST_CYCLE )
      wire#w2
      P_Trig( #"PLUS BIT"[24] )
      Move(in := #ENABLED_CYLINDER, out1 => #"CYL COUNT  VALUE")
   END_RUNG
   RUNG wire#w1
      Contact( #FILLING_SEQ_DONE )
   END_RUNG wire#w2
   // the same network as SCL:
   #_w1 := "AlwaysTRUE" AND #CYCLE_OK AND (#FIRST_CYCLE OR #FILLING_SEQ_DONE);
   #_w2 := #_w1 AND NOT #"PLUS BIT"[24];   // rising edge
   #"PLUS BIT"[24] := #_w1;
   IF #_w2 THEN #"CYL COUNT  VALUE" := #ENABLED_CYLINDER; END_IF;
END_REGION

REGION Network 31
   RUNG wire#powerrail
      Contact( "hmi"."AUTO/MAN_L2" )
      wire#w1
      R_Coil( #MANUAL )
   END_RUNG
   RUNG wire#w1
      S_Coil( #AUTO )
   END_RUNG
   // the same network as SCL:
   IF "hmi"."AUTO/MAN_L2" THEN
       #MANUAL := FALSE;
       #AUTO := TRUE;
   END_IF;
END_REGION

REGION Network 32
   RUNG wire#powerrail
      Contact( true )
      wire#w1
      Contact( #CYCLE_RESET )
      wire#w2
      { S7_Templates := "time_type := Time" } "IEC_Timer_0_DB_8_L2".TON(pt := T#1S, et =>)
      Coil( #"COUNTER RESET" )
   END_RUNG
   RUNG wire#w1
      Contact( #ALL_FILL_DONE )
   END_RUNG wire#w2
   // the same network as SCL:
   "IEC_Timer_0_DB_8_L2".TON(IN := true AND (#CYCLE_RESET OR #ALL_FILL_DONE), PT := T#1S);
   #"COUNTER RESET" := "IEC_Timer_0_DB_8_L2".Q;
END_REGION

REGION Network 33
   RUNG wire#powerrail
      I_Contact( "hmi"."AUTO/MAN_L2" )
      wire#w1
      R_Coil( #AUTO )
   END_RUNG
   RUNG wire#w1
      S_Coil( #MANUAL )
   END_RUNG
   // the same network as SCL:
   IF NOT "hmi"."AUTO/MAN_L2" THEN
       #AUTO := FALSE;
       #MANUAL := TRUE;
   END_IF;
END_REGION

REGION Network 34
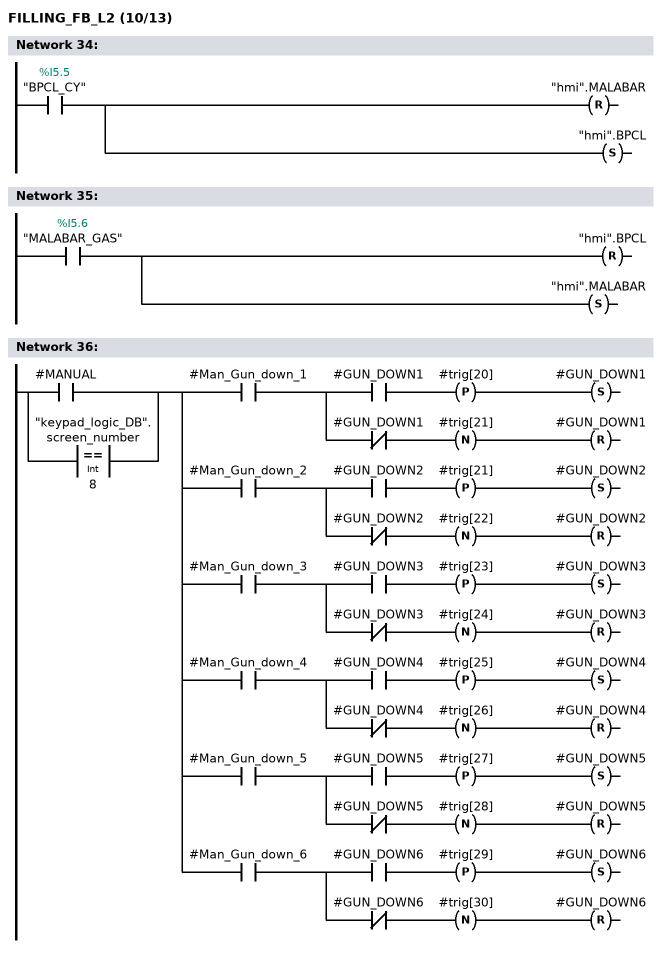
   RUNG wire#powerrail
      Contact( "BPCL_CY" )
      wire#w1
      R_Coil( "hmi".MALABAR )
   END_RUNG
   RUNG wire#w1
      S_Coil( "hmi".BPCL )
   END_RUNG
   // the same network as SCL:
   IF "BPCL_CY" THEN
       "hmi".MALABAR := FALSE;
       "hmi".BPCL := TRUE;
   END_IF;
END_REGION

REGION Network 35
   RUNG wire#powerrail
      Contact( "MALABAR_GAS" )
      wire#w1
      R_Coil( "hmi".BPCL )
   END_RUNG
   RUNG wire#w1
      S_Coil( "hmi".MALABAR )
   END_RUNG
   // the same network as SCL:
   IF "MALABAR_GAS" THEN
       "hmi".BPCL := FALSE;
       "hmi".MALABAR := TRUE;
   END_IF;
END_REGION

REGION Network 36
   RUNG wire#powerrail
      Contact( #MANUAL )
      wire#w1
      Contact( #Man_Gun_down_1 )
      wire#w2
      Contact( #GUN_DOWN1 )
      P_Trig( #trig[20] )
      S_Coil( #GUN_DOWN1 )
   END_RUNG
   RUNG wire#powerrail
      { S7_Templates := "SrcType := Int" } EQ_Contact(in1 := "keypad_logic_DB".screen_number, in2 := 8)
   END_RUNG wire#w1
   RUNG wire#w2
      I_Contact( #GUN_DOWN1 )
      N_Trig( #trig[21] )
      R_Coil( #GUN_DOWN1 )
   END_RUNG
   RUNG wire#w1
      Contact( #Man_Gun_down_2 )
      wire#w3
      Contact( #GUN_DOWN2 )
      P_Trig( #trig[21] )
      S_Coil( #GUN_DOWN2 )
   END_RUNG
   RUNG wire#w3
      I_Contact( #GUN_DOWN2 )
      N_Trig( #trig[22] )
      R_Coil( #GUN_DOWN2 )
   END_RUNG
   RUNG wire#w1
      Contact( #Man_Gun_down_3 )
      wire#w4
      Contact( #GUN_DOWN3 )
      P_Trig( #trig[23] )
      S_Coil( #GUN_DOWN3 )
   END_RUNG
   RUNG wire#w4
      I_Contact( #GUN_DOWN3 )
      N_Trig( #trig[24] )
      R_Coil( #GUN_DOWN3 )
   END_RUNG
   RUNG wire#w1
      Contact( #Man_Gun_down_4 )
      wire#w5
      Contact( #GUN_DOWN4 )
      P_Trig( #trig[25] )
      S_Coil( #GUN_DOWN4 )
   END_RUNG
   RUNG wire#w5
      I_Contact( #GUN_DOWN4 )
      N_Trig( #trig[26] )
      R_Coil( #GUN_DOWN4 )
   END_RUNG
   RUNG wire#w1
      Contact( #Man_Gun_down_5 )
      wire#w6
      Contact( #GUN_DOWN5 )
      P_Trig( #trig[27] )
      S_Coil( #GUN_DOWN5 )
   END_RUNG
   RUNG wire#w6
      I_Contact( #GUN_DOWN5 )
      N_Trig( #trig[28] )
      R_Coil( #GUN_DOWN5 )
   END_RUNG
   RUNG wire#w1
      Contact( #Man_Gun_down_6 )
      wire#w7
      Contact( #GUN_DOWN6 )
      P_Trig( #trig[29] )
      S_Coil( #GUN_DOWN6 )
   END_RUNG
   RUNG wire#w7
      I_Contact( #GUN_DOWN6 )
      N_Trig( #trig[30] )
      R_Coil( #GUN_DOWN6 )
   END_RUNG
   // the same network as SCL:
   #_w1 := #MANUAL OR ("keypad_logic_DB".screen_number = 8);
   #_w2 := #_w1 AND #Man_Gun_down_1;
   #_w3 := #_w2 AND #GUN_DOWN1;
   #_w4 := #_w3 AND NOT #trig[20];   // rising edge
   #trig[20] := #_w3;
   IF #_w4 THEN #GUN_DOWN1 := TRUE; END_IF;
   #_w5 := #_w2 AND NOT #GUN_DOWN1;
   #_w6 := NOT #_w5 AND #trig[21];   // falling edge
   #trig[21] := #_w5;
   IF #_w6 THEN #GUN_DOWN1 := FALSE; END_IF;
   #_w7 := #_w1 AND #Man_Gun_down_2;
   #_w8 := #_w7 AND #GUN_DOWN2;
   #_w9 := #_w8 AND NOT #trig[21];   // rising edge
   #trig[21] := #_w8;
   IF #_w9 THEN #GUN_DOWN2 := TRUE; END_IF;
   #_w10 := #_w7 AND NOT #GUN_DOWN2;
   #_w11 := NOT #_w10 AND #trig[22];   // falling edge
   #trig[22] := #_w10;
   IF #_w11 THEN #GUN_DOWN2 := FALSE; END_IF;
   #_w12 := #_w1 AND #Man_Gun_down_3;
   #_w13 := #_w12 AND #GUN_DOWN3;
   #_w14 := #_w13 AND NOT #trig[23];   // rising edge
   #trig[23] := #_w13;
   IF #_w14 THEN #GUN_DOWN3 := TRUE; END_IF;
   #_w15 := #_w12 AND NOT #GUN_DOWN3;
   #_w16 := NOT #_w15 AND #trig[24];   // falling edge
   #trig[24] := #_w15;
   IF #_w16 THEN #GUN_DOWN3 := FALSE; END_IF;
   #_w17 := #_w1 AND #Man_Gun_down_4;
   #_w18 := #_w17 AND #GUN_DOWN4;
   #_w19 := #_w18 AND NOT #trig[25];   // rising edge
   #trig[25] := #_w18;
   IF #_w19 THEN #GUN_DOWN4 := TRUE; END_IF;
   #_w20 := #_w17 AND NOT #GUN_DOWN4;
   #_w21 := NOT #_w20 AND #trig[26];   // falling edge
   #trig[26] := #_w20;
   IF #_w21 THEN #GUN_DOWN4 := FALSE; END_IF;
   #_w22 := #_w1 AND #Man_Gun_down_5;
   #_w23 := #_w22 AND #GUN_DOWN5;
   #_w24 := #_w23 AND NOT #trig[27];   // rising edge
   #trig[27] := #_w23;
   IF #_w24 THEN #GUN_DOWN5 := TRUE; END_IF;
   #_w25 := #_w22 AND NOT #GUN_DOWN5;
   #_w26 := NOT #_w25 AND #trig[28];   // falling edge
   #trig[28] := #_w25;
   IF #_w26 THEN #GUN_DOWN5 := FALSE; END_IF;
   #_w27 := #_w1 AND #Man_Gun_down_6;
   #_w28 := #_w27 AND #GUN_DOWN6;
   #_w29 := #_w28 AND NOT #trig[29];   // rising edge
   #trig[29] := #_w28;
   IF #_w29 THEN #GUN_DOWN6 := TRUE; END_IF;
   #_w30 := #_w27 AND NOT #GUN_DOWN6;
   #_w31 := NOT #_w30 AND #trig[30];   // falling edge
   #trig[30] := #_w30;
   IF #_w31 THEN #GUN_DOWN6 := FALSE; END_IF;
END_REGION

REGION Network 37
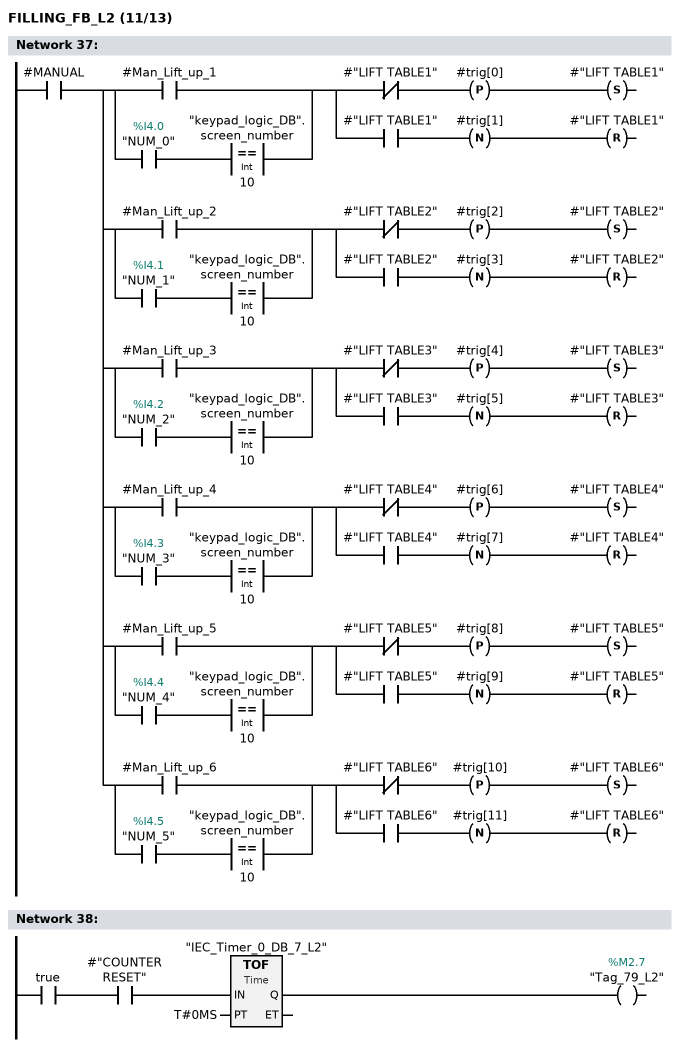
   RUNG wire#powerrail
      Contact( #MANUAL )
      wire#w1
      Contact( #Man_Lift_up_1 )
      wire#w2
      I_Contact( #"LIFT TABLE1" )
      P_Trig( #trig[0] )
      S_Coil( #"LIFT TABLE1" )
   END_RUNG
   RUNG wire#w1
      Contact( "NUM_0" )
      { S7_Templates := "SrcType := Int" } EQ_Contact(in1 := "keypad_logic_DB".screen_number, in2 := 10)
   END_RUNG wire#w2
   RUNG wire#w2
      Contact( #"LIFT TABLE1" )
      N_Trig( #trig[1] )
      R_Coil( #"LIFT TABLE1" )
   END_RUNG
   RUNG wire#w1
      Contact( #Man_Lift_up_2 )
      wire#w3
      I_Contact( #"LIFT TABLE2" )
      P_Trig( #trig[2] )
      S_Coil( #"LIFT TABLE2" )
   END_RUNG
   RUNG wire#w1
      Contact( "NUM_1" )
      { S7_Templates := "SrcType := Int" } EQ_Contact(in1 := "keypad_logic_DB".screen_number, in2 := 10)
   END_RUNG wire#w3
   RUNG wire#w3
      Contact( #"LIFT TABLE2" )
      N_Trig( #trig[3] )
      R_Coil( #"LIFT TABLE2" )
   END_RUNG
   RUNG wire#w1
      Contact( #Man_Lift_up_3 )
      wire#w4
      I_Contact( #"LIFT TABLE3" )
      P_Trig( #trig[4] )
      S_Coil( #"LIFT TABLE3" )
   END_RUNG
   RUNG wire#w1
      Contact( "NUM_2" )
      { S7_Templates := "SrcType := Int" } EQ_Contact(in1 := "keypad_logic_DB".screen_number, in2 := 10)
   END_RUNG wire#w4
   RUNG wire#w4
      Contact( #"LIFT TABLE3" )
      N_Trig( #trig[5] )
      R_Coil( #"LIFT TABLE3" )
   END_RUNG
   RUNG wire#w1
      Contact( #Man_Lift_up_4 )
      wire#w5
      I_Contact( #"LIFT TABLE4" )
      P_Trig( #trig[6] )
      S_Coil( #"LIFT TABLE4" )
   END_RUNG
   RUNG wire#w1
      Contact( "NUM_3" )
      { S7_Templates := "SrcType := Int" } EQ_Contact(in1 := "keypad_logic_DB".screen_number, in2 := 10)
   END_RUNG wire#w5
   RUNG wire#w5
      Contact( #"LIFT TABLE4" )
      N_Trig( #trig[7] )
      R_Coil( #"LIFT TABLE4" )
   END_RUNG
   RUNG wire#w1
      Contact( #Man_Lift_up_5 )
      wire#w6
      I_Contact( #"LIFT TABLE5" )
      P_Trig( #trig[8] )
      S_Coil( #"LIFT TABLE5" )
   END_RUNG
   RUNG wire#w1
      Contact( "NUM_4" )
      { S7_Templates := "SrcType := Int" } EQ_Contact(in1 := "keypad_logic_DB".screen_number, in2 := 10)
   END_RUNG wire#w6
   RUNG wire#w6
      Contact( #"LIFT TABLE5" )
      N_Trig( #trig[9] )
      R_Coil( #"LIFT TABLE5" )
   END_RUNG
   RUNG wire#w1
      Contact( #Man_Lift_up_6 )
      wire#w7
      I_Contact( #"LIFT TABLE6" )
      P_Trig( #trig[10] )
      S_Coil( #"LIFT TABLE6" )
   END_RUNG
   RUNG wire#w1
      Contact( "NUM_5" )
      { S7_Templates := "SrcType := Int" } EQ_Contact(in1 := "keypad_logic_DB".screen_number, in2 := 10)
   END_RUNG wire#w7
   RUNG wire#w7
      Contact( #"LIFT TABLE6" )
      N_Trig( #trig[11] )
      R_Coil( #"LIFT TABLE6" )
   END_RUNG
   // the same network as SCL:
   #_w1 := #MANUAL AND (#Man_Lift_up_1 OR ("NUM_0" AND ("keypad_logic_DB".screen_number = 10)));
   #_w2 := #_w1 AND NOT #"LIFT TABLE1";
   #_w3 := #_w2 AND NOT #trig[0];   // rising edge
   #trig[0] := #_w2;
   IF #_w3 THEN #"LIFT TABLE1" := TRUE; END_IF;
   #_w4 := #_w1 AND #"LIFT TABLE1";
   #_w5 := NOT #_w4 AND #trig[1];   // falling edge
   #trig[1] := #_w4;
   IF #_w5 THEN #"LIFT TABLE1" := FALSE; END_IF;
   #_w6 := #MANUAL AND (#Man_Lift_up_2 OR ("NUM_1" AND ("keypad_logic_DB".screen_number = 10)));
   #_w7 := #_w6 AND NOT #"LIFT TABLE2";
   #_w8 := #_w7 AND NOT #trig[2];   // rising edge
   #trig[2] := #_w7;
   IF #_w8 THEN #"LIFT TABLE2" := TRUE; END_IF;
   #_w9 := #_w6 AND #"LIFT TABLE2";
   #_w10 := NOT #_w9 AND #trig[3];   // falling edge
   #trig[3] := #_w9;
   IF #_w10 THEN #"LIFT TABLE2" := FALSE; END_IF;
   #_w11 := #MANUAL AND (#Man_Lift_up_3 OR ("NUM_2" AND ("keypad_logic_DB".screen_number = 10)));
   #_w12 := #_w11 AND NOT #"LIFT TABLE3";
   #_w13 := #_w12 AND NOT #trig[4];   // rising edge
   #trig[4] := #_w12;
   IF #_w13 THEN #"LIFT TABLE3" := TRUE; END_IF;
   #_w14 := #_w11 AND #"LIFT TABLE3";
   #_w15 := NOT #_w14 AND #trig[5];   // falling edge
   #trig[5] := #_w14;
   IF #_w15 THEN #"LIFT TABLE3" := FALSE; END_IF;
   #_w16 := #MANUAL AND (#Man_Lift_up_4 OR ("NUM_3" AND ("keypad_logic_DB".screen_number = 10)));
   #_w17 := #_w16 AND NOT #"LIFT TABLE4";
   #_w18 := #_w17 AND NOT #trig[6];   // rising edge
   #trig[6] := #_w17;
   IF #_w18 THEN #"LIFT TABLE4" := TRUE; END_IF;
   #_w19 := #_w16 AND #"LIFT TABLE4";
   #_w20 := NOT #_w19 AND #trig[7];   // falling edge
   #trig[7] := #_w19;
   IF #_w20 THEN #"LIFT TABLE4" := FALSE; END_IF;
   #_w21 := #MANUAL AND (#Man_Lift_up_5 OR ("NUM_4" AND ("keypad_logic_DB".screen_number = 10)));
   #_w22 := #_w21 AND NOT #"LIFT TABLE5";
   #_w23 := #_w22 AND NOT #trig[8];   // rising edge
   #trig[8] := #_w22;
   IF #_w23 THEN #"LIFT TABLE5" := TRUE; END_IF;
   #_w24 := #_w21 AND #"LIFT TABLE5";
   #_w25 := NOT #_w24 AND #trig[9];   // falling edge
   #trig[9] := #_w24;
   IF #_w25 THEN #"LIFT TABLE5" := FALSE; END_IF;
   #_w26 := #MANUAL AND (#Man_Lift_up_6 OR ("NUM_5" AND ("keypad_logic_DB".screen_number = 10)));
   #_w27 := #_w26 AND NOT #"LIFT TABLE6";
   #_w28 := #_w27 AND NOT #trig[10];   // rising edge
   #trig[10] := #_w27;
   IF #_w28 THEN #"LIFT TABLE6" := TRUE; END_IF;
   #_w29 := #_w26 AND #"LIFT TABLE6";
   #_w30 := NOT #_w29 AND #trig[11];   // falling edge
   #trig[11] := #_w29;
   IF #_w30 THEN #"LIFT TABLE6" := FALSE; END_IF;
END_REGION

REGION Network 38
   RUNG wire#powerrail
      Contact( true )
      Contact( #"COUNTER RESET" )
      { S7_Templates := "time_type := Time" } "IEC_Timer_0_DB_7_L2".TOF(pt := T#0MS, et =>)
      Coil( "Tag_79_L2" )
   END_RUNG
   // the same network as SCL:
   "IEC_Timer_0_DB_7_L2".TOF(IN := true AND #"COUNTER RESET", PT := T#0MS);
   "Tag_79_L2" := "IEC_Timer_0_DB_7_L2".Q;
END_REGION

REGION Network 39
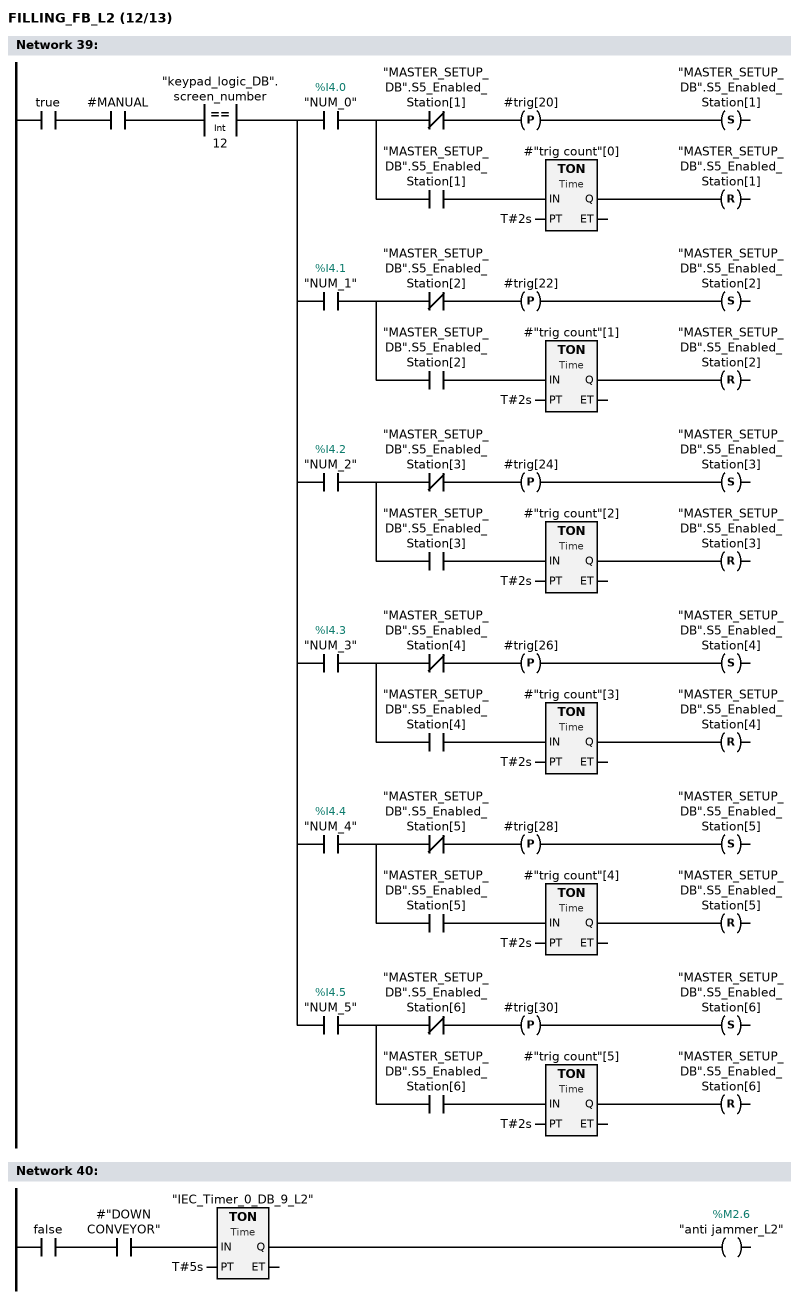
   RUNG wire#powerrail
      Contact( true )
      Contact( #MANUAL )
      { S7_Templates := "SrcType := Int" } EQ_Contact(in1 := "keypad_logic_DB".screen_number, in2 := 12)
      wire#w1
      Contact( "NUM_0" )
      wire#w2
      I_Contact( "MASTER_SETUP_DB".S5_Enabled_Station[1] )
      P_Trig( #trig[20] )
      S_Coil( "MASTER_SETUP_DB".S5_Enabled_Station[1] )
   END_RUNG
   RUNG wire#w2
      Contact( "MASTER_SETUP_DB".S5_Enabled_Station[1] )
      { S7_Templates := "time_type := Time" } #"trig count"[0].TON(pt := T#2s, et =>)
      R_Coil( "MASTER_SETUP_DB".S5_Enabled_Station[1] )
   END_RUNG
   RUNG wire#w1
      Contact( "NUM_1" )
      wire#w3
      I_Contact( "MASTER_SETUP_DB".S5_Enabled_Station[2] )
      P_Trig( #trig[22] )
      S_Coil( "MASTER_SETUP_DB".S5_Enabled_Station[2] )
   END_RUNG
   RUNG wire#w3
      Contact( "MASTER_SETUP_DB".S5_Enabled_Station[2] )
      { S7_Templates := "time_type := Time" } #"trig count"[1].TON(pt := T#2s, et =>)
      R_Coil( "MASTER_SETUP_DB".S5_Enabled_Station[2] )
   END_RUNG
   RUNG wire#w1
      Contact( "NUM_2" )
      wire#w4
      I_Contact( "MASTER_SETUP_DB".S5_Enabled_Station[3] )
      P_Trig( #trig[24] )
      S_Coil( "MASTER_SETUP_DB".S5_Enabled_Station[3] )
   END_RUNG
   RUNG wire#w4
      Contact( "MASTER_SETUP_DB".S5_Enabled_Station[3] )
      { S7_Templates := "time_type := Time" } #"trig count"[2].TON(pt := T#2s, et =>)
      R_Coil( "MASTER_SETUP_DB".S5_Enabled_Station[3] )
   END_RUNG
   RUNG wire#w1
      Contact( "NUM_3" )
      wire#w5
      I_Contact( "MASTER_SETUP_DB".S5_Enabled_Station[4] )
      P_Trig( #trig[26] )
      S_Coil( "MASTER_SETUP_DB".S5_Enabled_Station[4] )
   END_RUNG
   RUNG wire#w5
      Contact( "MASTER_SETUP_DB".S5_Enabled_Station[4] )
      { S7_Templates := "time_type := Time" } #"trig count"[3].TON(pt := T#2s, et =>)
      R_Coil( "MASTER_SETUP_DB".S5_Enabled_Station[4] )
   END_RUNG
   RUNG wire#w1
      Contact( "NUM_4" )
      wire#w6
      I_Contact( "MASTER_SETUP_DB".S5_Enabled_Station[5] )
      P_Trig( #trig[28] )
      S_Coil( "MASTER_SETUP_DB".S5_Enabled_Station[5] )
   END_RUNG
   RUNG wire#w6
      Contact( "MASTER_SETUP_DB".S5_Enabled_Station[5] )
      { S7_Templates := "time_type := Time" } #"trig count"[4].TON(pt := T#2s, et =>)
      R_Coil( "MASTER_SETUP_DB".S5_Enabled_Station[5] )
   END_RUNG
   RUNG wire#w1
      Contact( "NUM_5" )
      wire#w7
      I_Contact( "MASTER_SETUP_DB".S5_Enabled_Station[6] )
      P_Trig( #trig[30] )
      S_Coil( "MASTER_SETUP_DB".S5_Enabled_Station[6] )
   END_RUNG
   RUNG wire#w7
      Contact( "MASTER_SETUP_DB".S5_Enabled_Station[6] )
      { S7_Templates := "time_type := Time" } #"trig count"[5].TON(pt := T#2s, et =>)
      R_Coil( "MASTER_SETUP_DB".S5_Enabled_Station[6] )
   END_RUNG
   // the same network as SCL:
   #_w1 := true AND #MANUAL AND ("keypad_logic_DB".screen_number = 12);
   #_w2 := #_w1 AND "NUM_0";
   #_w3 := #_w2 AND NOT "MASTER_SETUP_DB".S5_Enabled_Station[1];
   #_w4 := #_w3 AND NOT #trig[20];   // rising edge
   #trig[20] := #_w3;
   IF #_w4 THEN "MASTER_SETUP_DB".S5_Enabled_Station[1] := TRUE; END_IF;
   #"trig count"[0].TON(IN := #_w2 AND "MASTER_SETUP_DB".S5_Enabled_Station[1], PT := T#2s);
   IF #"trig count"[0].Q THEN "MASTER_SETUP_DB".S5_Enabled_Station[1] := FALSE; END_IF;
   #_w5 := #_w1 AND "NUM_1";
   #_w6 := #_w5 AND NOT "MASTER_SETUP_DB".S5_Enabled_Station[2];
   #_w7 := #_w6 AND NOT #trig[22];   // rising edge
   #trig[22] := #_w6;
   IF #_w7 THEN "MASTER_SETUP_DB".S5_Enabled_Station[2] := TRUE; END_IF;
   #"trig count"[1].TON(IN := #_w5 AND "MASTER_SETUP_DB".S5_Enabled_Station[2], PT := T#2s);
   IF #"trig count"[1].Q THEN "MASTER_SETUP_DB".S5_Enabled_Station[2] := FALSE; END_IF;
   #_w8 := #_w1 AND "NUM_2";
   #_w9 := #_w8 AND NOT "MASTER_SETUP_DB".S5_Enabled_Station[3];
   #_w10 := #_w9 AND NOT #trig[24];   // rising edge
   #trig[24] := #_w9;
   IF #_w10 THEN "MASTER_SETUP_DB".S5_Enabled_Station[3] := TRUE; END_IF;
   #"trig count"[2].TON(IN := #_w8 AND "MASTER_SETUP_DB".S5_Enabled_Station[3], PT := T#2s);
   IF #"trig count"[2].Q THEN "MASTER_SETUP_DB".S5_Enabled_Station[3] := FALSE; END_IF;
   #_w11 := #_w1 AND "NUM_3";
   #_w12 := #_w11 AND NOT "MASTER_SETUP_DB".S5_Enabled_Station[4];
   #_w13 := #_w12 AND NOT #trig[26];   // rising edge
   #trig[26] := #_w12;
   IF #_w13 THEN "MASTER_SETUP_DB".S5_Enabled_Station[4] := TRUE; END_IF;
   #"trig count"[3].TON(IN := #_w11 AND "MASTER_SETUP_DB".S5_Enabled_Station[4], PT := T#2s);
   IF #"trig count"[3].Q THEN "MASTER_SETUP_DB".S5_Enabled_Station[4] := FALSE; END_IF;
   #_w14 := #_w1 AND "NUM_4";
   #_w15 := #_w14 AND NOT "MASTER_SETUP_DB".S5_Enabled_Station[5];
   #_w16 := #_w15 AND NOT #trig[28];   // rising edge
   #trig[28] := #_w15;
   IF #_w16 THEN "MASTER_SETUP_DB".S5_Enabled_Station[5] := TRUE; END_IF;
   #"trig count"[4].TON(IN := #_w14 AND "MASTER_SETUP_DB".S5_Enabled_Station[5], PT := T#2s);
   IF #"trig count"[4].Q THEN "MASTER_SETUP_DB".S5_Enabled_Station[5] := FALSE; END_IF;
   #_w17 := #_w1 AND "NUM_5";
   #_w18 := #_w17 AND NOT "MASTER_SETUP_DB".S5_Enabled_Station[6];
   #_w19 := #_w18 AND NOT #trig[30];   // rising edge
   #trig[30] := #_w18;
   IF #_w19 THEN "MASTER_SETUP_DB".S5_Enabled_Station[6] := TRUE; END_IF;
   #"trig count"[5].TON(IN := #_w17 AND "MASTER_SETUP_DB".S5_Enabled_Station[6], PT := T#2s);
   IF #"trig count"[5].Q THEN "MASTER_SETUP_DB".S5_Enabled_Station[6] := FALSE; END_IF;
END_REGION

REGION Network 40
   RUNG wire#powerrail
      Contact( false )
      Contact( #"DOWN CONVEYOR" )
      { S7_Templates := "time_type := Time" } "IEC_Timer_0_DB_9_L2".TON(pt := T#5s, et =>)
      Coil( "anti jammer_L2" )
   END_RUNG
   // the same network as SCL:
   "IEC_Timer_0_DB_9_L2".TON(IN := false AND #"DOWN CONVEYOR", PT := T#5s);
   "anti jammer_L2" := "IEC_Timer_0_DB_9_L2".Q;
END_REGION

REGION Network 41
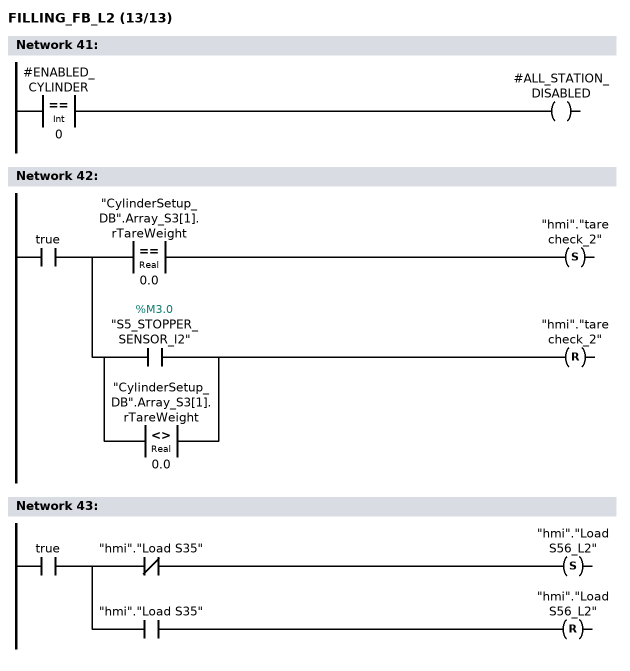
   RUNG wire#powerrail
      { S7_Templates := "SrcType := Int" } EQ_Contact(in1 := #ENABLED_CYLINDER, in2 := 0)
      Coil( #ALL_STATION_DISABLED )
   END_RUNG
   // the same network as SCL:
   #ALL_STATION_DISABLED := #ENABLED_CYLINDER = 0;
END_REGION

REGION Network 42
   RUNG wire#powerrail
      Contact( true )
      wire#w1
      { S7_Templates := "SrcType := Real" } EQ_Contact(in1 := "CylinderSetup_DB".Array_S3[1].rTareWeight, in2 := 0.0)
      S_Coil( "hmi"."tare check_2" )
   END_RUNG
   RUNG wire#w1
      Contact( "S5_STOPPER_SENSOR_l2" )
      wire#w2
      R_Coil( "hmi"."tare check_2" )
   END_RUNG
   RUNG wire#w1
      { S7_Templates := "SrcType := Real" } NE_Contact(in1 := "CylinderSetup_DB".Array_S3[1].rTareWeight, in2 := 0.0)
   END_RUNG wire#w2
   // the same network as SCL:
   IF true AND ("CylinderSetup_DB".Array_S3[1].rTareWeight = 0.0) THEN "hmi"."tare check_2" := TRUE; END_IF;
   IF true AND ("S5_STOPPER_SENSOR_l2" OR ("CylinderSetup_DB".Array_S3[1].rTareWeight <> 0.0)) THEN
       "hmi"."tare check_2" := FALSE;
   END_IF;
END_REGION

REGION Network 43
   RUNG wire#powerrail
      Contact( true )
      wire#w1
      I_Contact( "hmi"."Load S35" )
      S_Coil( "hmi"."Load S56_L2" )
   END_RUNG
   RUNG wire#w1
      Contact( "hmi"."Load S35" )
      R_Coil( "hmi"."Load S56_L2" )
   END_RUNG
   // the same network as SCL:
   IF true AND NOT "hmi"."Load S35" THEN "hmi"."Load S56_L2" := TRUE; END_IF;
   IF true AND "hmi"."Load S35" THEN "hmi"."Load S56_L2" := FALSE; END_IF;
END_REGION
END_FUNCTION_BLOCK

FUNCTION_BLOCK "keypad_logic"   // FB6, LAD
{ S7_Optimized_Access := 'TRUE' }
VERSION : 0.1
// stored: AutoNumber true, IsIECCheckEnabled false, IsRetainMemResEnabled false, MemoryReserve 100, SetENOAutomatically false, UDAEnableTagReadback false
   VAR_INPUT
      Num_0 : Bool;
      Num_1 : Bool;
      Num_2 : Bool;
      Num_3 : Bool;
      Num_4 : Bool;
      Num_5 : Bool;
      Num_6 : Bool;
      Num_7 : Bool;
      Num_8 : Bool;
      Num_9 : Bool;
      enter : Bool;
      clear : Bool;
   END_VAR
   VAR
      count_0 : CTU_INT;
   END_VAR
   VAR RETAIN
      Tens { S7_SetPoint := 'True'} : Int;
   END_VAR
   VAR
      ones : Int;
      decimal : Int;
      P_TRIG : Bool;
      MUL : Int;
      MUL_1 : Int;
      Tare_weight : Real;
      "count _reset" : Bool;
      Tare_Entry : Real;
      "screen count" : Int;
      screen_number : Int;
      screen_reset : Bool;
      MUL_2 : Int;
      count_1 : CTU_INT;
      count_cv_1 : Int;
      "BPCL COUNT" : Int;
      DOMESTIC : Bool;
      COMMERCIAL : Bool;
      MALALBAR_COUNT : Int;
   END_VAR
   VAR RETAIN
      SENSE_1 : Int;
      SENSE_2 : Int;
      SENSE_3 : Int;
      SENSE_4 : Int;
   END_VAR
   VAR
      "SENSI NG_TIME" : Int;
      sens_reset : Bool;
      "open screen" : Bool;
      DOMESTIC_1 : Bool;
      COMMERCIAL_1 : Bool;
      count_2 : CTU_INT;
   END_VAR
   VAR RETAIN
      password { S7_SetPoint := 'True'} : Int;
   END_VAR
   VAR
      password_1 : Int;
      password_2 : Int;
      password_3 : Int;
      password_4 : Int;
      password_5 : Int;
      mul_3 : Int;
      mul_4 : Int;
      mul_5 : Int;
      mul_6 : Int;
      password_reset : Bool;
      sens : Bool;
   END_VAR
   VAR_TEMP
      value_0 : Int;
      count_cv_0 : Int;
   END_VAR
   VAR_TEMP   // added for the SCL form of the ladder/FBD networks
      _w1 : Bool;
      _w2 : Bool;
      _w3 : Bool;
      _w4 : Bool;
      _w5 : Bool;
      _w6 : Bool;
   END_VAR
BEGIN

REGION Network 1
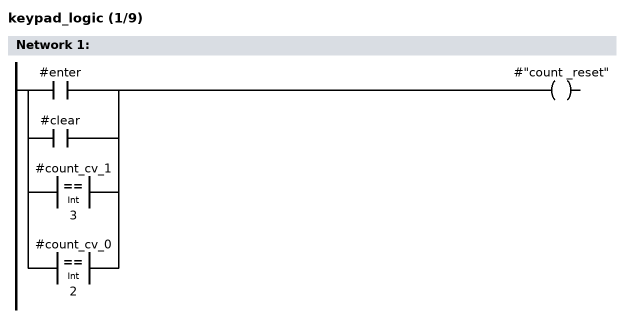
   RUNG wire#powerrail
      Contact( #enter )
      wire#w1
      Coil( #"count _reset" )
   END_RUNG
   RUNG wire#powerrail
      Contact( #clear )
   END_RUNG wire#w1
   RUNG wire#powerrail
      { S7_Templates := "SrcType := Int" } EQ_Contact(in1 := #count_cv_1, in2 := 3)
   END_RUNG wire#w1
   RUNG wire#powerrail
      { S7_Templates := "SrcType := Int" } EQ_Contact(in1 := #count_cv_0, in2 := 2)
   END_RUNG wire#w1
   // the same network as SCL:
   #"count _reset" := #enter OR #clear OR (#count_cv_1 = 3) OR (#count_cv_0 = 2);
END_REGION

REGION Network 2
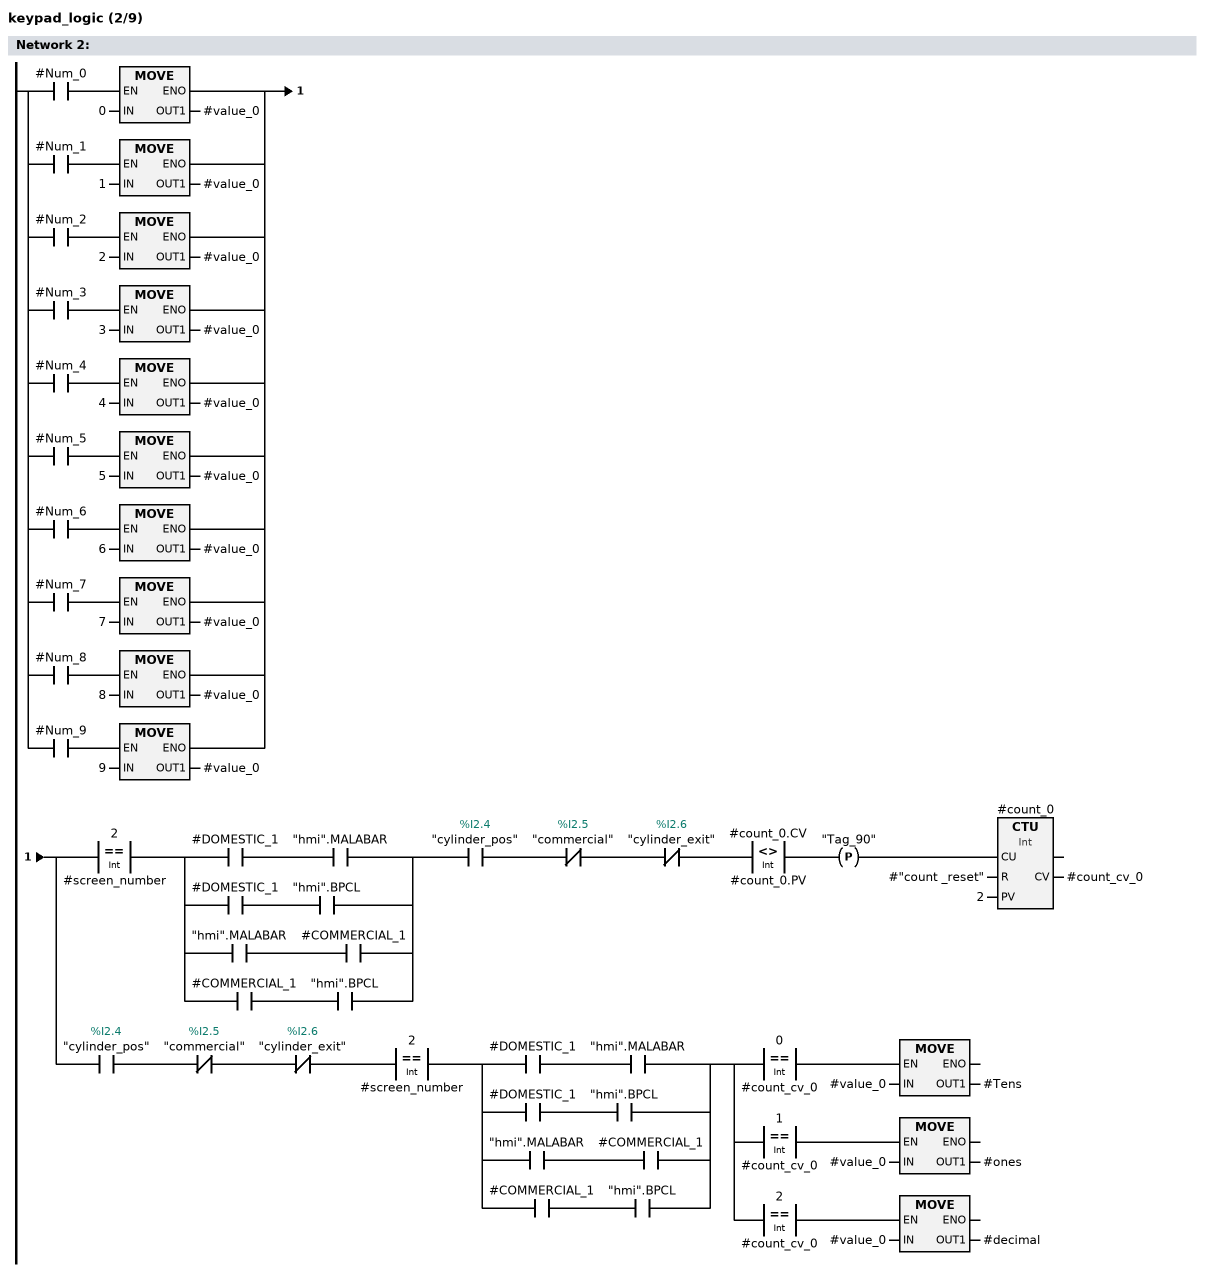
   RUNG wire#powerrail
      Contact( #Num_0 )
      Move(in := 0, out1 => #value_0)
      wire#w1
      { S7_Templates := "SrcType := Int" } EQ_Contact(in1 := 2, in2 := #screen_number)
      wire#w2
      Contact( #DOMESTIC_1 )
      Contact( "hmi".MALABAR )
      wire#w3
      Contact( "cylinder_pos" )
      I_Contact( "commercial" )
      I_Contact( "cylinder_exit" )
      { S7_Templates := "SrcType := Int" } NE_Contact(in1 := #count_0.CV, in2 := #count_0.PV)
      P_Trig( "Tag_90" )
      { S7_Templates := "value_type := Int" } #count_0.CTU(r := #"count _reset", pv := 2, cv => #count_cv_0)
   END_RUNG
   RUNG wire#powerrail
      Contact( #Num_1 )
      Move(in := 1, out1 => #value_0)
   END_RUNG wire#w1
   RUNG wire#powerrail
      Contact( #Num_2 )
      Move(in := 2, out1 => #value_0)
   END_RUNG wire#w1
   RUNG wire#powerrail
      Contact( #Num_3 )
      Move(in := 3, out1 => #value_0)
   END_RUNG wire#w1
   RUNG wire#powerrail
      Contact( #Num_4 )
      Move(in := 4, out1 => #value_0)
   END_RUNG wire#w1
   RUNG wire#powerrail
      Contact( #Num_5 )
      Move(in := 5, out1 => #value_0)
   END_RUNG wire#w1
   RUNG wire#powerrail
      Contact( #Num_6 )
      Move(in := 6, out1 => #value_0)
   END_RUNG wire#w1
   RUNG wire#powerrail
      Contact( #Num_7 )
      Move(in := 7, out1 => #value_0)
   END_RUNG wire#w1
   RUNG wire#powerrail
      Contact( #Num_8 )
      Move(in := 8, out1 => #value_0)
   END_RUNG wire#w1
   RUNG wire#powerrail
      Contact( #Num_9 )
      Move(in := 9, out1 => #value_0)
   END_RUNG wire#w1
   RUNG wire#w2
      Contact( #DOMESTIC_1 )
      Contact( "hmi".BPCL )
   END_RUNG wire#w3
   RUNG wire#w2
      Contact( "hmi".MALABAR )
      Contact( #COMMERCIAL_1 )
   END_RUNG wire#w3
   RUNG wire#w2
      Contact( #COMMERCIAL_1 )
      Contact( "hmi".BPCL )
   END_RUNG wire#w3
   RUNG wire#w1
      Contact( "cylinder_pos" )
      I_Contact( "commercial" )
      I_Contact( "cylinder_exit" )
      { S7_Templates := "SrcType := Int" } EQ_Contact(in1 := 2, in2 := #screen_number)
      wire#w4
      Contact( #DOMESTIC_1 )
      Contact( "hmi".MALABAR )
      wire#w5
      { S7_Templates := "SrcType := Int" } EQ_Contact(in1 := 0, in2 := #count_cv_0)
      Move(in := #value_0, out1 => #Tens)
   END_RUNG
   RUNG wire#w4
      Contact( #DOMESTIC_1 )
      Contact( "hmi".BPCL )
   END_RUNG wire#w5
   RUNG wire#w4
      Contact( "hmi".MALABAR )
      Contact( #COMMERCIAL_1 )
   END_RUNG wire#w5
   RUNG wire#w4
      Contact( #COMMERCIAL_1 )
      Contact( "hmi".BPCL )
   END_RUNG wire#w5
   RUNG wire#w5
      { S7_Templates := "SrcType := Int" } EQ_Contact(in1 := 1, in2 := #count_cv_0)
      Move(in := #value_0, out1 => #ones)
   END_RUNG
   RUNG wire#w5
      { S7_Templates := "SrcType := Int" } EQ_Contact(in1 := 2, in2 := #count_cv_0)
      Move(in := #value_0, out1 => #decimal)
   END_RUNG
   // the same network as SCL:
   IF #Num_0 THEN #value_0 := 0; END_IF;
   IF #Num_1 THEN #value_0 := 1; END_IF;
   IF #Num_2 THEN #value_0 := 2; END_IF;
   IF #Num_3 THEN #value_0 := 3; END_IF;
   IF #Num_4 THEN #value_0 := 4; END_IF;
   IF #Num_5 THEN #value_0 := 5; END_IF;
   IF #Num_6 THEN #value_0 := 6; END_IF;
   IF #Num_7 THEN #value_0 := 7; END_IF;
   IF #Num_8 THEN #value_0 := 8; END_IF;
   IF #Num_9 THEN #value_0 := 9; END_IF;
   #_w1 := #Num_0 OR #Num_1 OR #Num_2 OR #Num_3 OR #Num_4 OR #Num_5 OR #Num_6 OR #Num_7 OR #Num_8 OR #Num_9;
   #_w2 := #_w1 AND (2 = #screen_number) AND ((#DOMESTIC_1 AND "hmi".MALABAR) OR (#DOMESTIC_1 AND "hmi".BPCL) OR ("hmi".MALABAR AND #COMMERCIAL_1) OR (#COMMERCIAL_1 AND "hmi".BPCL)) AND "cylinder_pos" AND NOT "commercial" AND NOT "cylinder_exit" AND (#count_0.CV <> #count_0.PV);
   #_w3 := #_w2 AND NOT "Tag_90";   // rising edge
   "Tag_90" := #_w2;
   #count_0(CU := #_w3, R := #"count _reset", PV := 2, CV => #count_cv_0);   // CTU
   #_w4 := #_w1 AND "cylinder_pos" AND NOT "commercial" AND NOT "cylinder_exit" AND (2 = #screen_number) AND ((#DOMESTIC_1 AND "hmi".MALABAR) OR (#DOMESTIC_1 AND "hmi".BPCL) OR ("hmi".MALABAR AND #COMMERCIAL_1) OR (#COMMERCIAL_1 AND "hmi".BPCL));
   IF #_w4 AND (0 = #count_cv_0) THEN #Tens := #value_0; END_IF;
   IF #_w4 AND (1 = #count_cv_0) THEN #ones := #value_0; END_IF;
   IF #_w4 AND (2 = #count_cv_0) THEN #decimal := #value_0; END_IF;
END_REGION

REGION Network 3
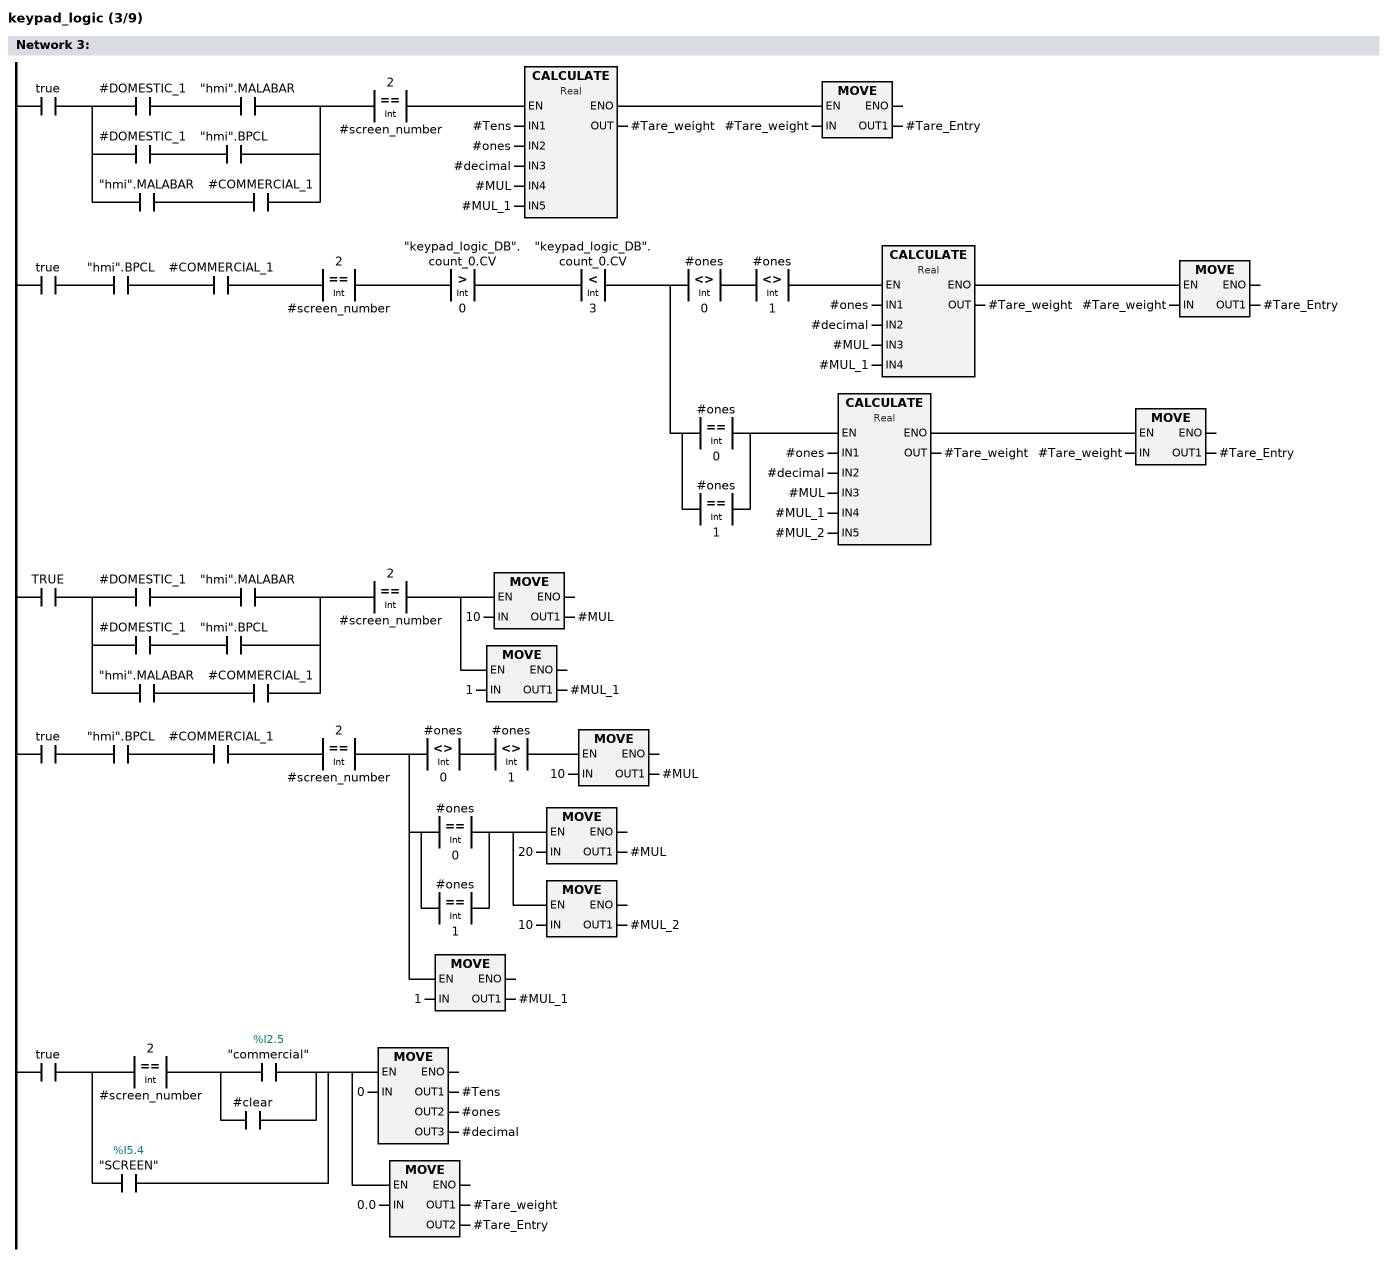
   RUNG wire#powerrail
      Contact( true )
      wire#w1
      Contact( #DOMESTIC_1 )
      Contact( "hmi".MALABAR )
      wire#w2
      { S7_Templates := "SrcType := Int" } EQ_Contact(in1 := 2, in2 := #screen_number)
      { S7_Templates := "SrcType := Real"; S7_Expression := "IN4+(IN2*IN5)+(IN3/IN4)" } Calculate(in1 := #Tens, in2 := #ones, in3 := #decimal, in4 := #MUL, in5 := #MUL_1, out => #Tare_weight)
      Move(in := #Tare_weight, out1 => #Tare_Entry)
   END_RUNG
   RUNG wire#w1
      Contact( #DOMESTIC_1 )
      Contact( "hmi".BPCL )
   END_RUNG wire#w2
   RUNG wire#w1
      Contact( "hmi".MALABAR )
      Contact( #COMMERCIAL_1 )
   END_RUNG wire#w2
   RUNG wire#powerrail
      Contact( true )
      Contact( "hmi".BPCL )
      Contact( #COMMERCIAL_1 )
      { S7_Templates := "SrcType := Int" } EQ_Contact(in1 := 2, in2 := #screen_number)
      { S7_Templates := "SrcType := Int" } GT_Contact(in1 := "keypad_logic_DB".count_0.CV, in2 := 0)
      { S7_Templates := "SrcType := Int" } LT_Contact(in1 := "keypad_logic_DB".count_0.CV, in2 := 3)
      wire#w3
      { S7_Templates := "SrcType := Int" } NE_Contact(in1 := #ones, in2 := 0)
      { S7_Templates := "SrcType := Int" } NE_Contact(in1 := #ones, in2 := 1)
      { S7_Templates := "SrcType := Real"; S7_Expression := "IN3+(IN1*IN4)+(IN2/IN3)" } Calculate(in1 := #ones, in2 := #decimal, in3 := #MUL, in4 := #MUL_1, out => #Tare_weight)
      Move(in := #Tare_weight, out1 => #Tare_Entry)
   END_RUNG
   RUNG wire#w3
      { S7_Templates := "SrcType := Int" } EQ_Contact(in1 := #ones, in2 := 0)
      wire#w4
      { S7_Templates := "SrcType := Real"; S7_Expression := "IN3+(IN1*IN4)+(IN2/IN5)" } Calculate(in1 := #ones, in2 := #decimal, in3 := #MUL, in4 := #MUL_1, in5 := #MUL_2, out => #Tare_weight)
      Move(in := #Tare_weight, out1 => #Tare_Entry)
   END_RUNG
   RUNG wire#w3
      { S7_Templates := "SrcType := Int" } EQ_Contact(in1 := #ones, in2 := 1)
   END_RUNG wire#w4
   RUNG wire#powerrail
      Contact( TRUE )
      wire#w5
      Contact( #DOMESTIC_1 )
      Contact( "hmi".MALABAR )
      wire#w6
      { S7_Templates := "SrcType := Int" } EQ_Contact(in1 := 2, in2 := #screen_number)
      wire#w7
      Move(in := 10, out1 => #MUL)
   END_RUNG
   RUNG wire#w5
      Contact( #DOMESTIC_1 )
      Contact( "hmi".BPCL )
   END_RUNG wire#w6
   RUNG wire#w5
      Contact( "hmi".MALABAR )
      Contact( #COMMERCIAL_1 )
   END_RUNG wire#w6
   RUNG wire#w7
      Move(in := 1, out1 => #MUL_1)
   END_RUNG
   RUNG wire#powerrail
      Contact( true )
      Contact( "hmi".BPCL )
      Contact( #COMMERCIAL_1 )
      { S7_Templates := "SrcType := Int" } EQ_Contact(in1 := 2, in2 := #screen_number)
      wire#w8
      { S7_Templates := "SrcType := Int" } NE_Contact(in1 := #ones, in2 := 0)
      { S7_Templates := "SrcType := Int" } NE_Contact(in1 := #ones, in2 := 1)
      Move(in := 10, out1 => #MUL)
   END_RUNG
   RUNG wire#w8
      { S7_Templates := "SrcType := Int" } EQ_Contact(in1 := #ones, in2 := 0)
      wire#w9
      Move(in := 20, out1 => #MUL)
   END_RUNG
   RUNG wire#w8
      { S7_Templates := "SrcType := Int" } EQ_Contact(in1 := #ones, in2 := 1)
   END_RUNG wire#w9
   RUNG wire#w9
      Move(in := 10, out1 => #MUL_2)
   END_RUNG
   RUNG wire#w8
      Move(in := 1, out1 => #MUL_1)
   END_RUNG
   RUNG wire#powerrail
      Contact( true )
      wire#w10
      { S7_Templates := "SrcType := Int" } EQ_Contact(in1 := 2, in2 := #screen_number)
      wire#w11
      Contact( "commercial" )
      wire#w12
      Move(in := 0, out1 => #Tens, out2 => #ones, out3 => #decimal)
   END_RUNG
   RUNG wire#w11
      Contact( #clear )
   END_RUNG wire#w12
   RUNG wire#w10
      Contact( "SCREEN" )
   END_RUNG wire#w12
   RUNG wire#w12
      Move(in := 0.0, out1 => #Tare_weight, out2 => #Tare_Entry)
   END_RUNG
   // the same network as SCL:
   IF true AND ((#DOMESTIC_1 AND "hmi".MALABAR) OR (#DOMESTIC_1 AND "hmi".BPCL) OR ("hmi".MALABAR AND #COMMERCIAL_1)) AND (2 = #screen_number) THEN
       #Tare_weight := #MUL+(#ones*#MUL_1)+(#decimal/#MUL);
       #Tare_Entry := #Tare_weight;
   END_IF;
   #_w1 := true AND "hmi".BPCL AND #COMMERCIAL_1 AND (2 = #screen_number) AND ("keypad_logic_DB".count_0.CV > 0) AND ("keypad_logic_DB".count_0.CV < 3);
   IF #_w1 AND (#ones <> 0) AND (#ones <> 1) THEN
       #Tare_weight := #MUL+(#ones*#MUL_1)+(#decimal/#MUL);
       #Tare_Entry := #Tare_weight;
   END_IF;
   IF #_w1 AND ((#ones = 0) OR (#ones = 1)) THEN
       #Tare_weight := #MUL+(#ones*#MUL_1)+(#decimal/#MUL_2);
       #Tare_Entry := #Tare_weight;
   END_IF;
   IF TRUE AND ((#DOMESTIC_1 AND "hmi".MALABAR) OR (#DOMESTIC_1 AND "hmi".BPCL) OR ("hmi".MALABAR AND #COMMERCIAL_1)) AND (2 = #screen_number) THEN
       #MUL := 10;
       #MUL_1 := 1;
   END_IF;
   #_w2 := true AND "hmi".BPCL AND #COMMERCIAL_1 AND (2 = #screen_number);
   IF #_w2 AND (#ones <> 0) AND (#ones <> 1) THEN #MUL := 10; END_IF;
   IF #_w2 AND ((#ones = 0) OR (#ones = 1)) THEN
       #MUL := 20;
       #MUL_2 := 10;
   END_IF;
   IF #_w2 THEN #MUL_1 := 1; END_IF;
   IF true AND (((2 = #screen_number) AND ("commercial" OR #clear)) OR "SCREEN") THEN
       #Tens := 0;
       #ones := 0;
       #decimal := 0;
       #Tare_weight := 0.0;
       #Tare_Entry := 0.0;
   END_IF;
END_REGION

REGION Network 4
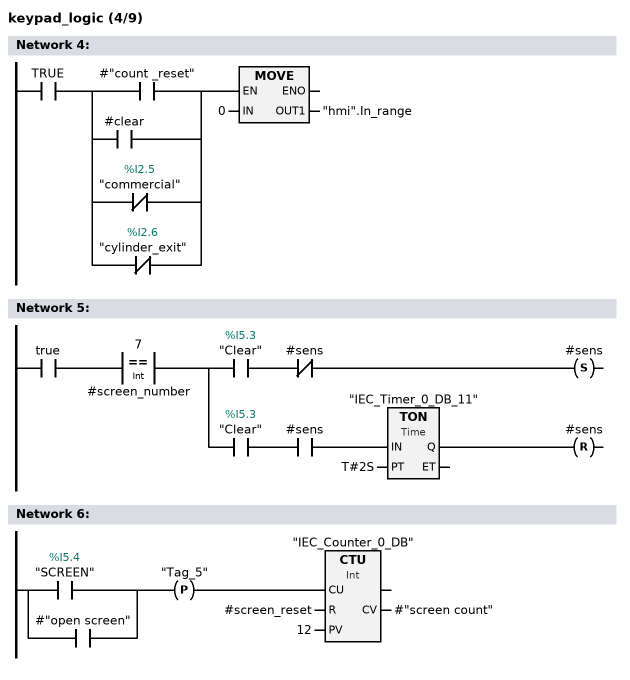
   RUNG wire#powerrail
      Contact( TRUE )
      wire#w1
      Contact( #"count _reset" )
      wire#w2
      Move(in := 0, out1 => "hmi".In_range)
   END_RUNG
   RUNG wire#w1
      Contact( #clear )
   END_RUNG wire#w2
   RUNG wire#w1
      I_Contact( "commercial" )
   END_RUNG wire#w2
   RUNG wire#w1
      I_Contact( "cylinder_exit" )
   END_RUNG wire#w2
   // the same network as SCL:
   IF TRUE AND (#"count _reset" OR #clear OR NOT "commercial" OR NOT "cylinder_exit") THEN
       "hmi".In_range := 0;
   END_IF;
END_REGION

REGION Network 5
   RUNG wire#powerrail
      Contact( true )
      { S7_Templates := "SrcType := Int" } EQ_Contact(in1 := 7, in2 := #screen_number)
      wire#w1
      Contact( "Clear" )
      I_Contact( #sens )
      S_Coil( #sens )
   END_RUNG
   RUNG wire#w1
      Contact( "Clear" )
      Contact( #sens )
      { S7_Templates := "time_type := Time" } "IEC_Timer_0_DB_11".TON(pt := T#2S, et =>)
      R_Coil( #sens )
   END_RUNG
   // the same network as SCL:
   #_w1 := true AND (7 = #screen_number);
   IF #_w1 AND "Clear" AND NOT #sens THEN #sens := TRUE; END_IF;
   "IEC_Timer_0_DB_11".TON(IN := #_w1 AND "Clear" AND #sens, PT := T#2S);
   IF "IEC_Timer_0_DB_11".Q THEN #sens := FALSE; END_IF;
END_REGION

REGION Network 6
   RUNG wire#powerrail
      Contact( "SCREEN" )
      wire#w1
      P_Trig( "Tag_5" )
      { S7_Templates := "value_type := Int" } "IEC_Counter_0_DB".CTU(r := #screen_reset, pv := 12, cv => #"screen count")
   END_RUNG
   RUNG wire#powerrail
      Contact( #"open screen" )
   END_RUNG wire#w1
   // the same network as SCL:
   #_w1 := "SCREEN" OR #"open screen";
   #_w2 := #_w1 AND NOT "Tag_5";   // rising edge
   "Tag_5" := #_w1;
   "IEC_Counter_0_DB".CTU(CU := #_w2, R := #screen_reset, PV := 12, CV => #"screen count");
END_REGION

REGION Network 7
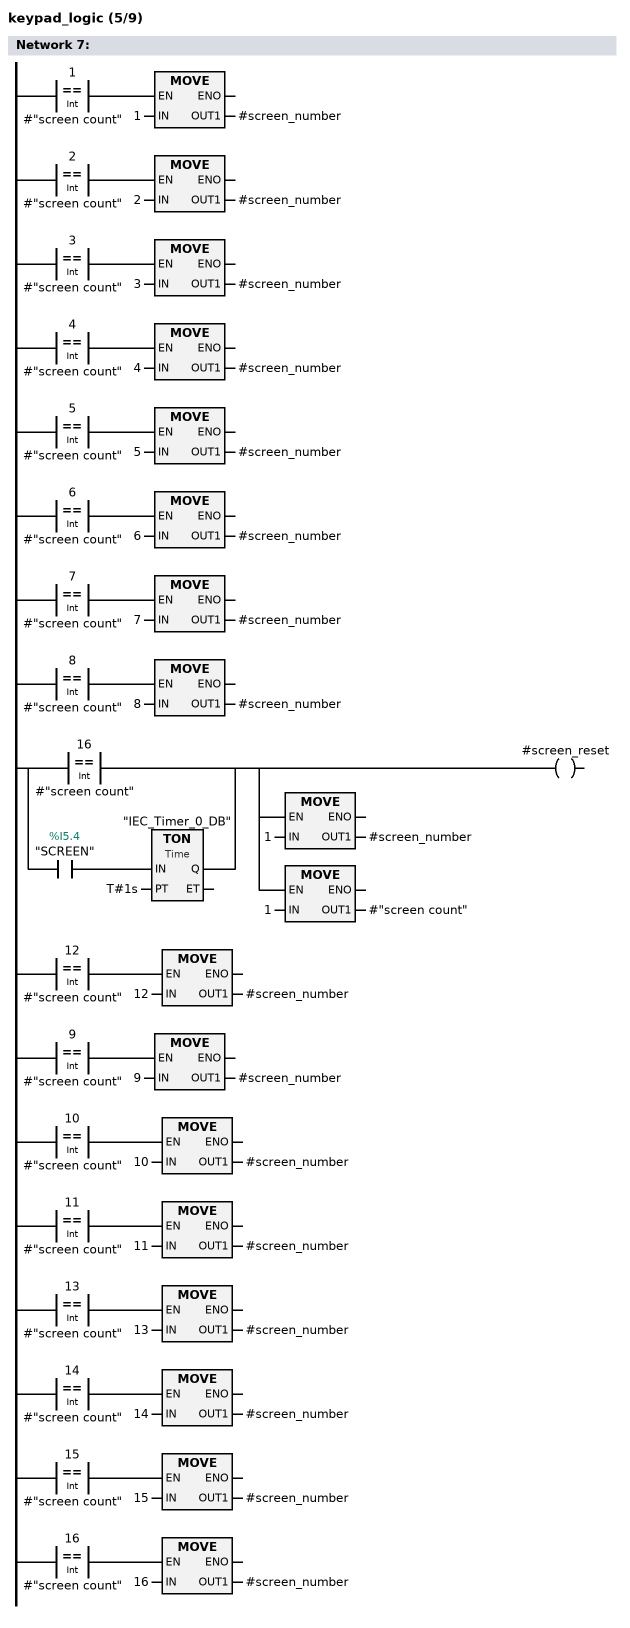
   RUNG wire#powerrail
      { S7_Templates := "SrcType := Int" } EQ_Contact(in1 := 1, in2 := #"screen count")
      Move(in := 1, out1 => #screen_number)
   END_RUNG
   RUNG wire#powerrail
      { S7_Templates := "SrcType := Int" } EQ_Contact(in1 := 2, in2 := #"screen count")
      Move(in := 2, out1 => #screen_number)
   END_RUNG
   RUNG wire#powerrail
      { S7_Templates := "SrcType := Int" } EQ_Contact(in1 := 3, in2 := #"screen count")
      Move(in := 3, out1 => #screen_number)
   END_RUNG
   RUNG wire#powerrail
      { S7_Templates := "SrcType := Int" } EQ_Contact(in1 := 4, in2 := #"screen count")
      Move(in := 4, out1 => #screen_number)
   END_RUNG
   RUNG wire#powerrail
      { S7_Templates := "SrcType := Int" } EQ_Contact(in1 := 5, in2 := #"screen count")
      Move(in := 5, out1 => #screen_number)
   END_RUNG
   RUNG wire#powerrail
      { S7_Templates := "SrcType := Int" } EQ_Contact(in1 := 6, in2 := #"screen count")
      Move(in := 6, out1 => #screen_number)
   END_RUNG
   RUNG wire#powerrail
      { S7_Templates := "SrcType := Int" } EQ_Contact(in1 := 7, in2 := #"screen count")
      Move(in := 7, out1 => #screen_number)
   END_RUNG
   RUNG wire#powerrail
      { S7_Templates := "SrcType := Int" } EQ_Contact(in1 := 8, in2 := #"screen count")
      Move(in := 8, out1 => #screen_number)
   END_RUNG
   RUNG wire#powerrail
      { S7_Templates := "SrcType := Int" } EQ_Contact(in1 := 16, in2 := #"screen count")
      wire#w1
      Coil( #screen_reset )
   END_RUNG
   RUNG wire#powerrail
      Contact( "SCREEN" )
      { S7_Templates := "time_type := Time" } "IEC_Timer_0_DB".TON(pt := T#1s, et =>)
   END_RUNG wire#w1
   RUNG wire#w1
      Move(in := 1, out1 => #screen_number)
   END_RUNG
   RUNG wire#w1
      Move(in := 1, out1 => #"screen count")
   END_RUNG
   RUNG wire#powerrail
      { S7_Templates := "SrcType := Int" } EQ_Contact(in1 := 12, in2 := #"screen count")
      Move(in := 12, out1 => #screen_number)
   END_RUNG
   RUNG wire#powerrail
      { S7_Templates := "SrcType := Int" } EQ_Contact(in1 := 9, in2 := #"screen count")
      Move(in := 9, out1 => #screen_number)
   END_RUNG
   RUNG wire#powerrail
      { S7_Templates := "SrcType := Int" } EQ_Contact(in1 := 10, in2 := #"screen count")
      Move(in := 10, out1 => #screen_number)
   END_RUNG
   RUNG wire#powerrail
      { S7_Templates := "SrcType := Int" } EQ_Contact(in1 := 11, in2 := #"screen count")
      Move(in := 11, out1 => #screen_number)
   END_RUNG
   RUNG wire#powerrail
      { S7_Templates := "SrcType := Int" } EQ_Contact(in1 := 13, in2 := #"screen count")
      Move(in := 13, out1 => #screen_number)
   END_RUNG
   RUNG wire#powerrail
      { S7_Templates := "SrcType := Int" } EQ_Contact(in1 := 14, in2 := #"screen count")
      Move(in := 14, out1 => #screen_number)
   END_RUNG
   RUNG wire#powerrail
      { S7_Templates := "SrcType := Int" } EQ_Contact(in1 := 15, in2 := #"screen count")
      Move(in := 15, out1 => #screen_number)
   END_RUNG
   RUNG wire#powerrail
      { S7_Templates := "SrcType := Int" } EQ_Contact(in1 := 16, in2 := #"screen count")
      Move(in := 16, out1 => #screen_number)
   END_RUNG
   // the same network as SCL:
   IF 1 = #"screen count" THEN #screen_number := 1; END_IF;
   IF 2 = #"screen count" THEN #screen_number := 2; END_IF;
   IF 3 = #"screen count" THEN #screen_number := 3; END_IF;
   IF 4 = #"screen count" THEN #screen_number := 4; END_IF;
   IF 5 = #"screen count" THEN #screen_number := 5; END_IF;
   IF 6 = #"screen count" THEN #screen_number := 6; END_IF;
   IF 7 = #"screen count" THEN #screen_number := 7; END_IF;
   IF 8 = #"screen count" THEN #screen_number := 8; END_IF;
   "IEC_Timer_0_DB".TON(IN := "SCREEN", PT := T#1s);
   #screen_reset := (16 = #"screen count") OR "IEC_Timer_0_DB".Q;
   IF #screen_reset THEN
       #screen_number := 1;
       #"screen count" := 1;
   END_IF;
   IF 12 = #"screen count" THEN #screen_number := 12; END_IF;
   IF 9 = #"screen count" THEN #screen_number := 9; END_IF;
   IF 10 = #"screen count" THEN #screen_number := 10; END_IF;
   IF 11 = #"screen count" THEN #screen_number := 11; END_IF;
   IF 13 = #"screen count" THEN #screen_number := 13; END_IF;
   IF 14 = #"screen count" THEN #screen_number := 14; END_IF;
   IF 15 = #"screen count" THEN #screen_number := 15; END_IF;
   IF 16 = #"screen count" THEN #screen_number := 16; END_IF;
END_REGION

REGION Network 8
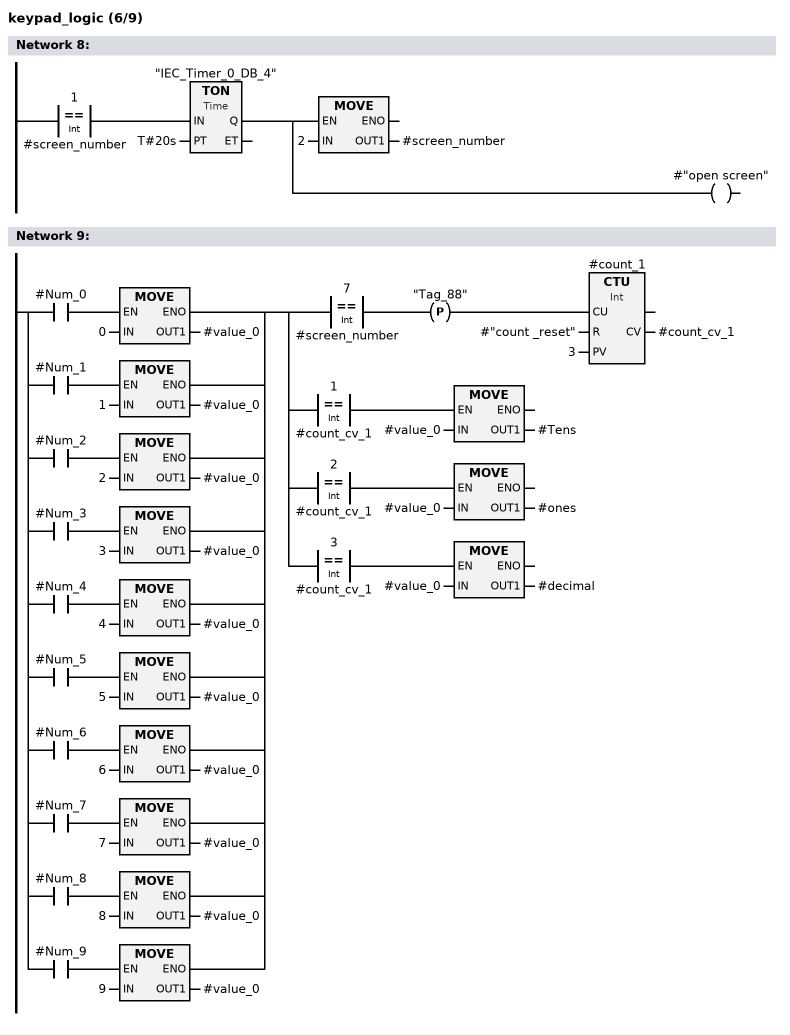
   RUNG wire#powerrail
      { S7_Templates := "SrcType := Int" } EQ_Contact(in1 := 1, in2 := #screen_number)
      { S7_Templates := "time_type := Time" } "IEC_Timer_0_DB_4".TON(pt := T#20s, et =>)
      wire#w1
      Move(in := 2, out1 => #screen_number)
   END_RUNG
   RUNG wire#w1
      Coil( #"open screen" )
   END_RUNG
   // the same network as SCL:
   "IEC_Timer_0_DB_4".TON(IN := 1 = #screen_number, PT := T#20s);
   IF "IEC_Timer_0_DB_4".Q THEN #screen_number := 2; END_IF;
   #"open screen" := "IEC_Timer_0_DB_4".Q;
END_REGION

REGION Network 9
   RUNG wire#powerrail
      Contact( #Num_0 )
      Move(in := 0, out1 => #value_0)
      wire#w1
      { S7_Templates := "SrcType := Int" } EQ_Contact(in1 := 7, in2 := #screen_number)
      P_Trig( "Tag_88" )
      { S7_Templates := "value_type := Int" } #count_1.CTU(r := #"count _reset", pv := 3, cv => #count_cv_1)
   END_RUNG
   RUNG wire#powerrail
      Contact( #Num_1 )
      Move(in := 1, out1 => #value_0)
   END_RUNG wire#w1
   RUNG wire#powerrail
      Contact( #Num_2 )
      Move(in := 2, out1 => #value_0)
   END_RUNG wire#w1
   RUNG wire#powerrail
      Contact( #Num_3 )
      Move(in := 3, out1 => #value_0)
   END_RUNG wire#w1
   RUNG wire#powerrail
      Contact( #Num_4 )
      Move(in := 4, out1 => #value_0)
   END_RUNG wire#w1
   RUNG wire#powerrail
      Contact( #Num_5 )
      Move(in := 5, out1 => #value_0)
   END_RUNG wire#w1
   RUNG wire#powerrail
      Contact( #Num_6 )
      Move(in := 6, out1 => #value_0)
   END_RUNG wire#w1
   RUNG wire#powerrail
      Contact( #Num_7 )
      Move(in := 7, out1 => #value_0)
   END_RUNG wire#w1
   RUNG wire#powerrail
      Contact( #Num_8 )
      Move(in := 8, out1 => #value_0)
   END_RUNG wire#w1
   RUNG wire#powerrail
      Contact( #Num_9 )
      Move(in := 9, out1 => #value_0)
   END_RUNG wire#w1
   RUNG wire#w1
      { S7_Templates := "SrcType := Int" } EQ_Contact(in1 := 1, in2 := #count_cv_1)
      Move(in := #value_0, out1 => #Tens)
   END_RUNG
   RUNG wire#w1
      { S7_Templates := "SrcType := Int" } EQ_Contact(in1 := 2, in2 := #count_cv_1)
      Move(in := #value_0, out1 => #ones)
   END_RUNG
   RUNG wire#w1
      { S7_Templates := "SrcType := Int" } EQ_Contact(in1 := 3, in2 := #count_cv_1)
      Move(in := #value_0, out1 => #decimal)
   END_RUNG
   // the same network as SCL:
   IF #Num_0 THEN #value_0 := 0; END_IF;
   IF #Num_1 THEN #value_0 := 1; END_IF;
   IF #Num_2 THEN #value_0 := 2; END_IF;
   IF #Num_3 THEN #value_0 := 3; END_IF;
   IF #Num_4 THEN #value_0 := 4; END_IF;
   IF #Num_5 THEN #value_0 := 5; END_IF;
   IF #Num_6 THEN #value_0 := 6; END_IF;
   IF #Num_7 THEN #value_0 := 7; END_IF;
   IF #Num_8 THEN #value_0 := 8; END_IF;
   IF #Num_9 THEN #value_0 := 9; END_IF;
   #_w1 := #Num_0 OR #Num_1 OR #Num_2 OR #Num_3 OR #Num_4 OR #Num_5 OR #Num_6 OR #Num_7 OR #Num_8 OR #Num_9;
   #_w2 := #_w1 AND (7 = #screen_number);
   #_w3 := #_w2 AND NOT "Tag_88";   // rising edge
   "Tag_88" := #_w2;
   #count_1(CU := #_w3, R := #"count _reset", PV := 3, CV => #count_cv_1);   // CTU
   IF #_w1 AND (1 = #count_cv_1) THEN #Tens := #value_0; END_IF;
   IF #_w1 AND (2 = #count_cv_1) THEN #ones := #value_0; END_IF;
   IF #_w1 AND (3 = #count_cv_1) THEN #decimal := #value_0; END_IF;
END_REGION

REGION Network 10
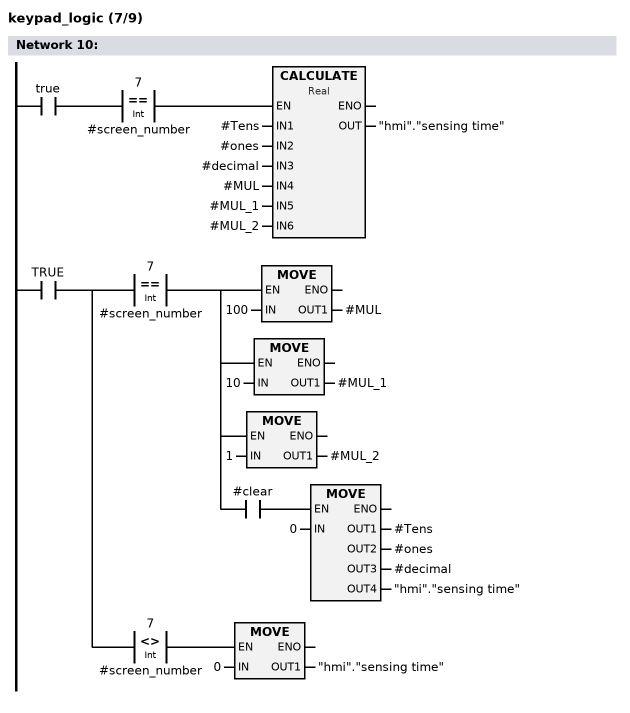
   RUNG wire#powerrail
      Contact( true )
      { S7_Templates := "SrcType := Int" } EQ_Contact(in1 := 7, in2 := #screen_number)
      { S7_Templates := "SrcType := Real"; S7_Expression := "(IN1*IN4)+(IN2*IN5)+(IN3*IN6)" } Calculate(in1 := #Tens, in2 := #ones, in3 := #decimal, in4 := #MUL, in5 := #MUL_1, in6 := #MUL_2, out => "hmi"."sensing time")
   END_RUNG
   RUNG wire#powerrail
      Contact( TRUE )
      wire#w1
      { S7_Templates := "SrcType := Int" } EQ_Contact(in1 := 7, in2 := #screen_number)
      wire#w2
      Move(in := 100, out1 => #MUL)
   END_RUNG
   RUNG wire#w2
      Move(in := 10, out1 => #MUL_1)
   END_RUNG
   RUNG wire#w2
      Move(in := 1, out1 => #MUL_2)
   END_RUNG
   RUNG wire#w2
      Contact( #clear )
      Move(in := 0, out1 => #Tens, out2 => #ones, out3 => #decimal, out4 => "hmi"."sensing time")
   END_RUNG
   RUNG wire#w1
      { S7_Templates := "SrcType := Int" } NE_Contact(in1 := 7, in2 := #screen_number)
      Move(in := 0, out1 => "hmi"."sensing time")
   END_RUNG
   // the same network as SCL:
   IF true AND (7 = #screen_number) THEN
       "hmi"."sensing time" := (#Tens*#MUL)+(#ones*#MUL_1)+(#decimal*#MUL_2);
   END_IF;
   #_w1 := TRUE AND (7 = #screen_number);
   IF #_w1 THEN
       #MUL := 100;
       #MUL_1 := 10;
       #MUL_2 := 1;
   END_IF;
   IF #_w1 AND #clear THEN
       #Tens := 0;
       #ones := 0;
       #decimal := 0;
       "hmi"."sensing time" := 0;
   END_IF;
   IF TRUE AND (7 <> #screen_number) THEN "hmi"."sensing time" := 0; END_IF;
END_REGION

REGION Network 11
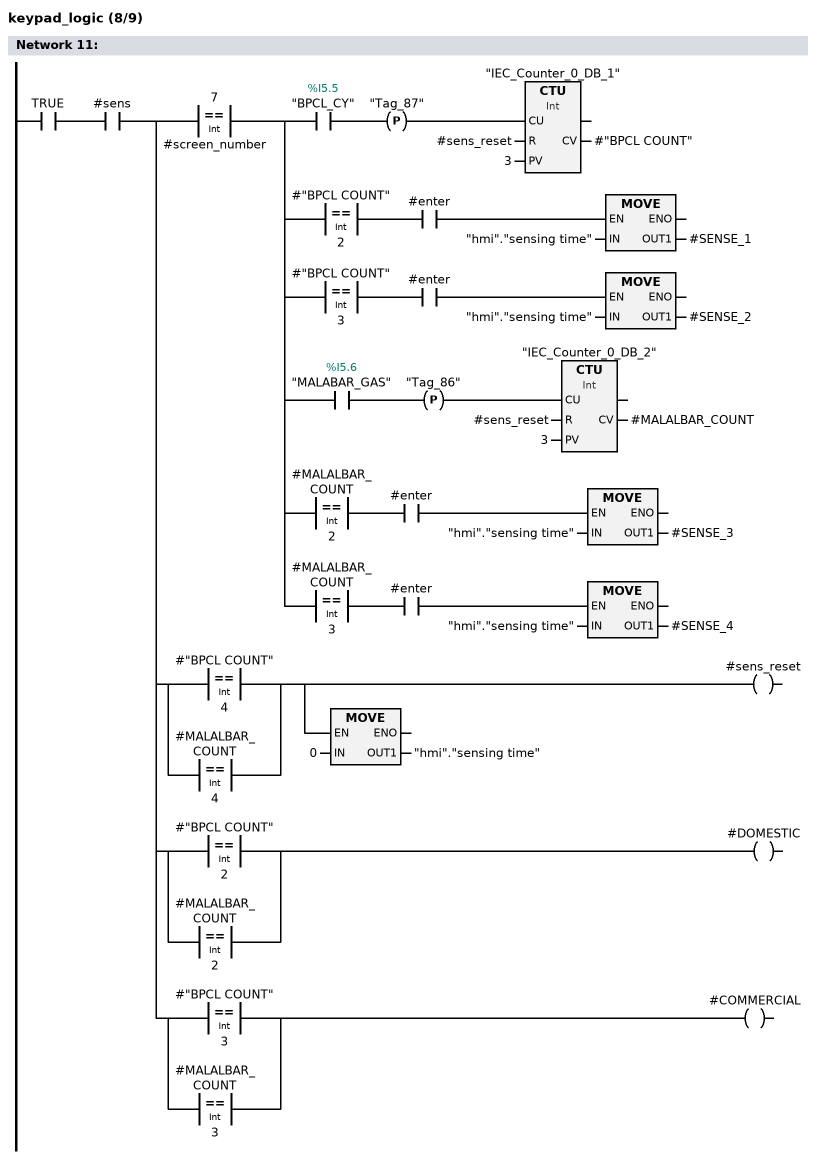
   RUNG wire#powerrail
      Contact( TRUE )
      Contact( #sens )
      wire#w1
      { S7_Templates := "SrcType := Int" } EQ_Contact(in1 := 7, in2 := #screen_number)
      wire#w2
      Contact( "BPCL_CY" )
      P_Trig( "Tag_87" )
      { S7_Templates := "value_type := Int" } "IEC_Counter_0_DB_1".CTU(r := #sens_reset, pv := 3, cv => #"BPCL COUNT")
   END_RUNG
   RUNG wire#w2
      { S7_Templates := "SrcType := Int" } EQ_Contact(in1 := #"BPCL COUNT", in2 := 2)
      Contact( #enter )
      Move(in := "hmi"."sensing time", out1 => #SENSE_1)
   END_RUNG
   RUNG wire#w2
      { S7_Templates := "SrcType := Int" } EQ_Contact(in1 := #"BPCL COUNT", in2 := 3)
      Contact( #enter )
      Move(in := "hmi"."sensing time", out1 => #SENSE_2)
   END_RUNG
   RUNG wire#w2
      Contact( "MALABAR_GAS" )
      P_Trig( "Tag_86" )
      { S7_Templates := "value_type := Int" } "IEC_Counter_0_DB_2".CTU(r := #sens_reset, pv := 3, cv => #MALALBAR_COUNT)
   END_RUNG
   RUNG wire#w2
      { S7_Templates := "SrcType := Int" } EQ_Contact(in1 := #MALALBAR_COUNT, in2 := 2)
      Contact( #enter )
      Move(in := "hmi"."sensing time", out1 => #SENSE_3)
   END_RUNG
   RUNG wire#w2
      { S7_Templates := "SrcType := Int" } EQ_Contact(in1 := #MALALBAR_COUNT, in2 := 3)
      Contact( #enter )
      Move(in := "hmi"."sensing time", out1 => #SENSE_4)
   END_RUNG
   RUNG wire#w1
      { S7_Templates := "SrcType := Int" } EQ_Contact(in1 := #"BPCL COUNT", in2 := 4)
      wire#w3
      Coil( #sens_reset )
   END_RUNG
   RUNG wire#w1
      { S7_Templates := "SrcType := Int" } EQ_Contact(in1 := #MALALBAR_COUNT, in2 := 4)
   END_RUNG wire#w3
   RUNG wire#w3
      Move(in := 0, out1 => "hmi"."sensing time")
   END_RUNG
   RUNG wire#w1
      { S7_Templates := "SrcType := Int" } EQ_Contact(in1 := #"BPCL COUNT", in2 := 2)
      wire#w4
      Coil( #DOMESTIC )
   END_RUNG
   RUNG wire#w1
      { S7_Templates := "SrcType := Int" } EQ_Contact(in1 := #MALALBAR_COUNT, in2 := 2)
   END_RUNG wire#w4
   RUNG wire#w1
      { S7_Templates := "SrcType := Int" } EQ_Contact(in1 := #"BPCL COUNT", in2 := 3)
      wire#w5
      Coil( #COMMERCIAL )
   END_RUNG
   RUNG wire#w1
      { S7_Templates := "SrcType := Int" } EQ_Contact(in1 := #MALALBAR_COUNT, in2 := 3)
   END_RUNG wire#w5
   // the same network as SCL:
   #_w1 := TRUE AND #sens;
   #_w2 := #_w1 AND (7 = #screen_number);
   #_w3 := #_w2 AND "BPCL_CY";
   #_w4 := #_w3 AND NOT "Tag_87";   // rising edge
   "Tag_87" := #_w3;
   "IEC_Counter_0_DB_1".CTU(CU := #_w4, R := #sens_reset, PV := 3, CV => #"BPCL COUNT");
   IF #_w2 AND (#"BPCL COUNT" = 2) AND #enter THEN #SENSE_1 := "hmi"."sensing time"; END_IF;
   IF #_w2 AND (#"BPCL COUNT" = 3) AND #enter THEN #SENSE_2 := "hmi"."sensing time"; END_IF;
   #_w5 := #_w2 AND "MALABAR_GAS";
   #_w6 := #_w5 AND NOT "Tag_86";   // rising edge
   "Tag_86" := #_w5;
   "IEC_Counter_0_DB_2".CTU(CU := #_w6, R := #sens_reset, PV := 3, CV => #MALALBAR_COUNT);
   IF #_w2 AND (#MALALBAR_COUNT = 2) AND #enter THEN #SENSE_3 := "hmi"."sensing time"; END_IF;
   IF #_w2 AND (#MALALBAR_COUNT = 3) AND #enter THEN #SENSE_4 := "hmi"."sensing time"; END_IF;
   #sens_reset := #_w1 AND ((#"BPCL COUNT" = 4) OR (#MALALBAR_COUNT = 4));
   IF #sens_reset THEN "hmi"."sensing time" := 0; END_IF;
   #DOMESTIC := #_w1 AND ((#"BPCL COUNT" = 2) OR (#MALALBAR_COUNT = 2));
   #COMMERCIAL := #_w1 AND ((#"BPCL COUNT" = 3) OR (#MALALBAR_COUNT = 3));
END_REGION

REGION Network 12
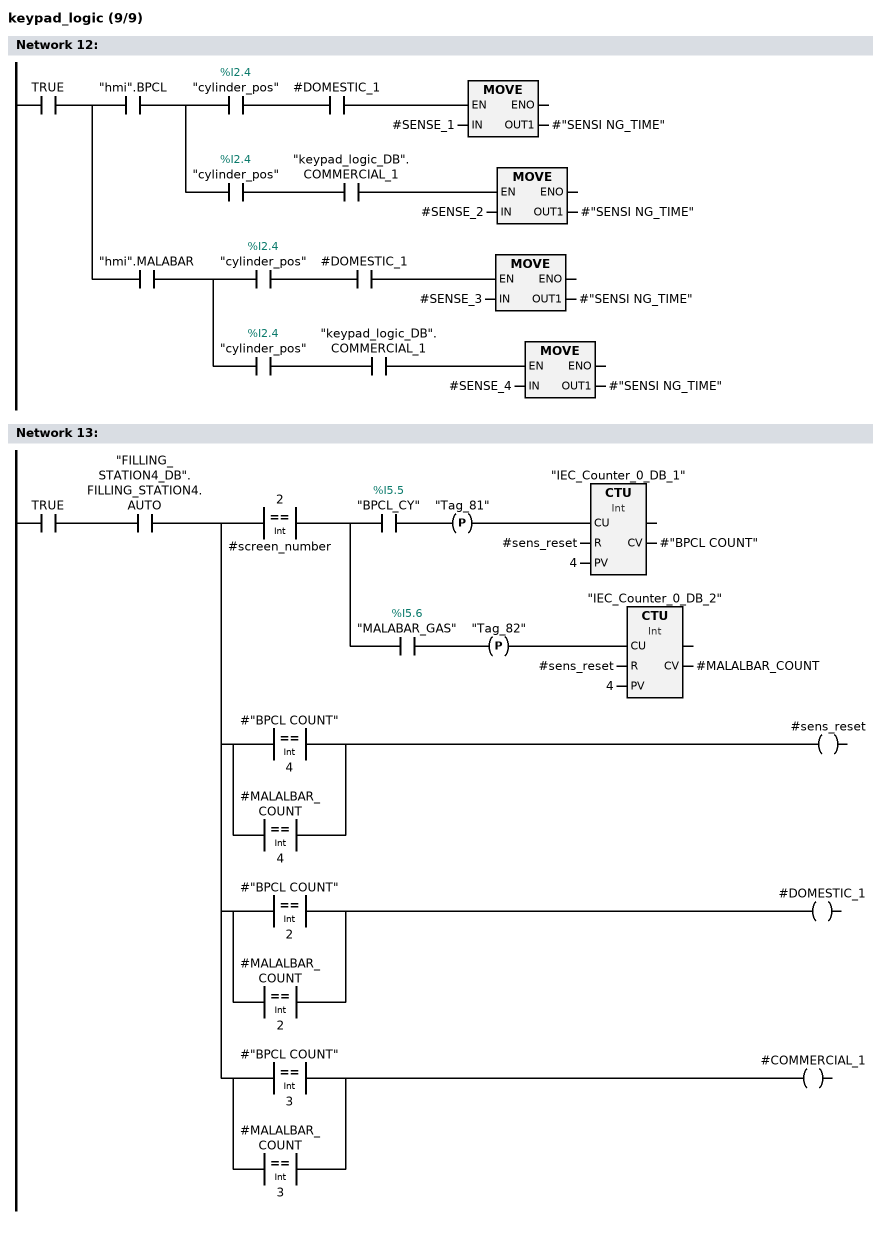
   RUNG wire#powerrail
      Contact( TRUE )
      wire#w1
      Contact( "hmi".BPCL )
      wire#w2
      Contact( "cylinder_pos" )
      Contact( #DOMESTIC_1 )
      Move(in := #SENSE_1, out1 => #"SENSI NG_TIME")
   END_RUNG
   RUNG wire#w2
      Contact( "cylinder_pos" )
      Contact( "keypad_logic_DB".COMMERCIAL_1 )
      Move(in := #SENSE_2, out1 => #"SENSI NG_TIME")
   END_RUNG
   RUNG wire#w1
      Contact( "hmi".MALABAR )
      wire#w3
      Contact( "cylinder_pos" )
      Contact( #DOMESTIC_1 )
      Move(in := #SENSE_3, out1 => #"SENSI NG_TIME")
   END_RUNG
   RUNG wire#w3
      Contact( "cylinder_pos" )
      Contact( "keypad_logic_DB".COMMERCIAL_1 )
      Move(in := #SENSE_4, out1 => #"SENSI NG_TIME")
   END_RUNG
   // the same network as SCL:
   #_w1 := TRUE AND "hmi".BPCL;
   IF #_w1 AND "cylinder_pos" AND #DOMESTIC_1 THEN #"SENSI NG_TIME" := #SENSE_1; END_IF;
   IF #_w1 AND "cylinder_pos" AND "keypad_logic_DB".COMMERCIAL_1 THEN #"SENSI NG_TIME" := #SENSE_2; END_IF;
   #_w2 := TRUE AND "hmi".MALABAR;
   IF #_w2 AND "cylinder_pos" AND #DOMESTIC_1 THEN #"SENSI NG_TIME" := #SENSE_3; END_IF;
   IF #_w2 AND "cylinder_pos" AND "keypad_logic_DB".COMMERCIAL_1 THEN #"SENSI NG_TIME" := #SENSE_4; END_IF;
END_REGION

REGION Network 13
   RUNG wire#powerrail
      Contact( TRUE )
      Contact( "FILLING_STATION4_DB".FILLING_STATION4.AUTO )
      wire#w1
      { S7_Templates := "SrcType := Int" } EQ_Contact(in1 := 2, in2 := #screen_number)
      wire#w2
      Contact( "BPCL_CY" )
      P_Trig( "Tag_81" )
      { S7_Templates := "value_type := Int" } "IEC_Counter_0_DB_1".CTU(r := #sens_reset, pv := 4, cv => #"BPCL COUNT")
   END_RUNG
   RUNG wire#w2
      Contact( "MALABAR_GAS" )
      P_Trig( "Tag_82" )
      { S7_Templates := "value_type := Int" } "IEC_Counter_0_DB_2".CTU(r := #sens_reset, pv := 4, cv => #MALALBAR_COUNT)
   END_RUNG
   RUNG wire#w1
      { S7_Templates := "SrcType := Int" } EQ_Contact(in1 := #"BPCL COUNT", in2 := 4)
      wire#w3
      Coil( #sens_reset )
   END_RUNG
   RUNG wire#w1
      { S7_Templates := "SrcType := Int" } EQ_Contact(in1 := #MALALBAR_COUNT, in2 := 4)
   END_RUNG wire#w3
   RUNG wire#w1
      { S7_Templates := "SrcType := Int" } EQ_Contact(in1 := #"BPCL COUNT", in2 := 2)
      wire#w4
      Coil( #DOMESTIC_1 )
   END_RUNG
   RUNG wire#w1
      { S7_Templates := "SrcType := Int" } EQ_Contact(in1 := #MALALBAR_COUNT, in2 := 2)
   END_RUNG wire#w4
   RUNG wire#w1
      { S7_Templates := "SrcType := Int" } EQ_Contact(in1 := #"BPCL COUNT", in2 := 3)
      wire#w5
      Coil( #COMMERCIAL_1 )
   END_RUNG
   RUNG wire#w1
      { S7_Templates := "SrcType := Int" } EQ_Contact(in1 := #MALALBAR_COUNT, in2 := 3)
   END_RUNG wire#w5
   // the same network as SCL:
   #_w1 := TRUE AND "FILLING_STATION4_DB".FILLING_STATION4.AUTO;
   #_w2 := #_w1 AND (2 = #screen_number);
   #_w3 := #_w2 AND "BPCL_CY";
   #_w4 := #_w3 AND NOT "Tag_81";   // rising edge
   "Tag_81" := #_w3;
   "IEC_Counter_0_DB_1".CTU(CU := #_w4, R := #sens_reset, PV := 4, CV => #"BPCL COUNT");
   #_w5 := #_w2 AND "MALABAR_GAS";
   #_w6 := #_w5 AND NOT "Tag_82";   // rising edge
   "Tag_82" := #_w5;
   "IEC_Counter_0_DB_2".CTU(CU := #_w6, R := #sens_reset, PV := 4, CV => #MALALBAR_COUNT);
   #sens_reset := #_w1 AND ((#"BPCL COUNT" = 4) OR (#MALALBAR_COUNT = 4));
   #DOMESTIC_1 := #_w1 AND ((#"BPCL COUNT" = 2) OR (#MALALBAR_COUNT = 2));
   #COMMERCIAL_1 := #_w1 AND ((#"BPCL COUNT" = 3) OR (#MALALBAR_COUNT = 3));
END_REGION
END_FUNCTION_BLOCK

FUNCTION "CHECK_SCALE" : Void   // FC2, LAD
{ S7_Optimized_Access := 'TRUE' }
VERSION : 0.1
// stored: AutoNumber true, IsIECCheckEnabled false, SetENOAutomatically false, UDAEnableTagReadback false
   VAR_TEMP
      cycle_start : Bool;
      temp : Int;
   END_VAR
BEGIN

REGION Network 1
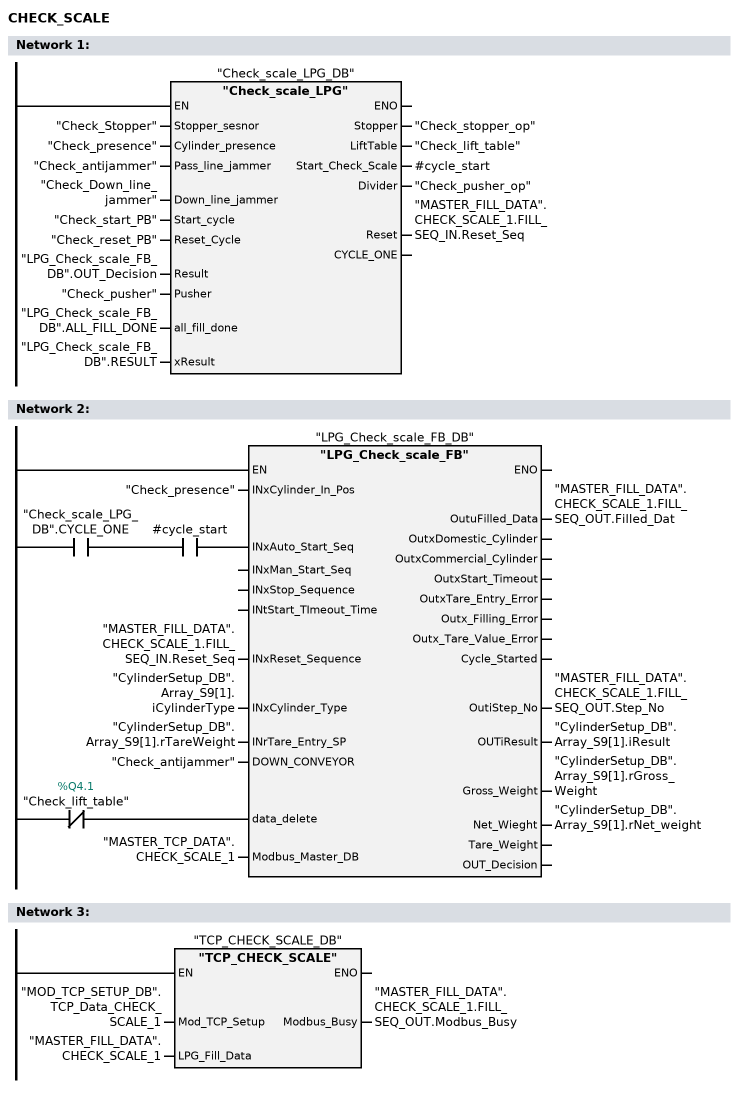
   RUNG wire#powerrail
      "Check_scale_LPG_DB"(Stopper_sesnor := "Check_Stopper", Cylinder_presence := "Check_presence", Pass_line_jammer := "Check_antijammer", Down_line_jammer := "Check_Down_line_jammer", Start_cycle := "Check_start_PB", Reset_Cycle := "Check_reset_PB", Result := "LPG_Check_scale_FB_DB".OUT_Decision, Pusher := "Check_pusher", all_fill_done := "LPG_Check_scale_FB_DB".ALL_FILL_DONE, xResult := "LPG_Check_scale_FB_DB".RESULT, Stopper => "Check_stopper_op", LiftTable => "Check_lift_table", Start_Check_Scale => #cycle_start, Divider => "Check_pusher_op", Reset => "MASTER_FILL_DATA".CHECK_SCALE_1.FILL_SEQ_IN.Reset_Seq, CYCLE_ONE =>)
   END_RUNG
   // the same network as SCL:
   "Check_scale_LPG_DB"(Stopper_sesnor := "Check_Stopper",   // "Check_scale_LPG"
                        Cylinder_presence := "Check_presence",
                        Pass_line_jammer := "Check_antijammer",
                        Down_line_jammer := "Check_Down_line_jammer",
                        Start_cycle := "Check_start_PB",
                        Reset_Cycle := "Check_reset_PB",
                        Result := "LPG_Check_scale_FB_DB".OUT_Decision,
                        Pusher := "Check_pusher",
                        all_fill_done := "LPG_Check_scale_FB_DB".ALL_FILL_DONE,
                        xResult := "LPG_Check_scale_FB_DB".RESULT,
                        Stopper => "Check_stopper_op",
                        LiftTable => "Check_lift_table",
                        Start_Check_Scale => #cycle_start,
                        Divider => "Check_pusher_op",
                        Reset => "MASTER_FILL_DATA".CHECK_SCALE_1.FILL_SEQ_IN.Reset_Seq);
END_REGION

REGION Network 2
   RUNG wire#powerrail
      "LPG_Check_scale_FB_DB"(INxAuto_Start_Seq := wire#w1, data_delete := wire#w2, INxCylinder_In_Pos := "Check_presence", INxMan_Start_Seq :=, INxStop_Sequence :=, INtStart_TImeout_Time :=, INxReset_Sequence := "MASTER_FILL_DATA".CHECK_SCALE_1.FILL_SEQ_IN.Reset_Seq, INxCylinder_Type := "CylinderSetup_DB".Array_S9[1].iCylinderType, INrTare_Entry_SP := "CylinderSetup_DB".Array_S9[1].rTareWeight, DOWN_CONVEYOR := "Check_antijammer", Modbus_Master_DB := "MASTER_TCP_DATA".CHECK_SCALE_1, OutuFilled_Data => "MASTER_FILL_DATA".CHECK_SCALE_1.FILL_SEQ_OUT.Filled_Dat, OutxDomestic_Cylinder =>, OutxCommercial_Cylinder =>, OutxStart_Timeout =>, OutxTare_Entry_Error =>, Outx_Filling_Error =>, Outx_Tare_Value_Error =>, Cycle_Started =>, OutiStep_No => "MASTER_FILL_DATA".CHECK_SCALE_1.FILL_SEQ_OUT.Step_No, OUTiResult => "CylinderSetup_DB".Array_S9[1].iResult, Gross_Weight => "CylinderSetup_DB".Array_S9[1].rGross_Weight, Net_Wieght => "CylinderSetup_DB".Array_S9[1].rNet_weight, Tare_Weight =>, OUT_Decision =>)
   END_RUNG
   RUNG wire#powerrail
      Contact( "Check_scale_LPG_DB".CYCLE_ONE )
      Contact( #cycle_start )
   END_RUNG wire#w1
   RUNG wire#powerrail
      I_Contact( "Check_lift_table" )
   END_RUNG wire#w2
   // the same network as SCL:
   "LPG_Check_scale_FB_DB"(INxCylinder_In_Pos := "Check_presence",   // "LPG_Check_scale_FB"
                           INxAuto_Start_Seq := "Check_scale_LPG_DB".CYCLE_ONE AND #cycle_start,
                           INxReset_Sequence := "MASTER_FILL_DATA".CHECK_SCALE_1.FILL_SEQ_IN.Reset_Seq,
                           INxCylinder_Type := "CylinderSetup_DB".Array_S9[1].iCylinderType,
                           INrTare_Entry_SP := "CylinderSetup_DB".Array_S9[1].rTareWeight,
                           DOWN_CONVEYOR := "Check_antijammer",
                           data_delete := NOT "Check_lift_table",
                           Modbus_Master_DB := "MASTER_TCP_DATA".CHECK_SCALE_1,
                           OutuFilled_Data => "MASTER_FILL_DATA".CHECK_SCALE_1.FILL_SEQ_OUT.Filled_Dat,
                           OutiStep_No => "MASTER_FILL_DATA".CHECK_SCALE_1.FILL_SEQ_OUT.Step_No,
                           OUTiResult => "CylinderSetup_DB".Array_S9[1].iResult,
                           Gross_Weight => "CylinderSetup_DB".Array_S9[1].rGross_Weight,
                           Net_Wieght => "CylinderSetup_DB".Array_S9[1].rNet_weight);
END_REGION

REGION Network 3
   RUNG wire#powerrail
      "TCP_CHECK_SCALE_DB"(Mod_TCP_Setup := "MOD_TCP_SETUP_DB".TCP_Data_CHECK_SCALE_1, LPG_Fill_Data := "MASTER_FILL_DATA".CHECK_SCALE_1, Modbus_Busy => "MASTER_FILL_DATA".CHECK_SCALE_1.FILL_SEQ_OUT.Modbus_Busy)
   END_RUNG
   // the same network as SCL:
   "TCP_CHECK_SCALE_DB"(Mod_TCP_Setup := "MOD_TCP_SETUP_DB".TCP_Data_CHECK_SCALE_1,   // "TCP_CHECK_SCALE"
                        LPG_Fill_Data := "MASTER_FILL_DATA".CHECK_SCALE_1,
                        Modbus_Busy => "MASTER_FILL_DATA".CHECK_SCALE_1.FILL_SEQ_OUT.Modbus_Busy);
END_REGION
END_FUNCTION

FUNCTION_BLOCK "Check_scale_LPG"   // FB7, LAD
{ S7_Optimized_Access := 'TRUE' }
VERSION : 0.1
// stored: AutoNumber true, IsIECCheckEnabled false, IsRetainMemResEnabled false, MemoryReserve 100, SetENOAutomatically false, UDAEnableTagReadback false
   VAR_INPUT
      Stopper_sesnor : Bool;
      Cylinder_presence : Bool;
      Pass_line_jammer : Bool;
      Down_line_jammer : Bool;
      Start_cycle : Bool;
      Reset_Cycle : Bool;
      Result : Int;
      Pusher : Bool;
      all_fill_done : Bool;
      xResult : Bool;
   END_VAR
   VAR_OUTPUT
      Stopper : Bool;
      LiftTable : Bool;
      Start_Check_Scale : Bool;
      Divider : Bool;
      Reset : Bool;
      CYCLE_ONE : Bool;
   END_VAR
   VAR
      Check_Scale_Started : Bool;
      Lift_Table { S7_SetPoint := 'True'} : TON_TIME;
      PASS : Bool;
      FAIL : Bool;
      LIFT_down { S7_SetPoint := 'True'} : TON_TIME;
      Temp_1 : Int;
      p_trig : Array[0..10] of Bool;
   END_VAR
   VAR RETAIN
      Stopper_count { S7_SetPoint := 'True'} : CTU_INT;
   END_VAR
   VAR
      counter_reset : Bool;
      Scale { S7_SetPoint := 'True'} : TON_TIME;
      Pusher_reset { S7_SetPoint := 'True'} : TON_TIME;
      datasend { ExternalAccessible := 'False'; ExternalVisible := 'False'; ExternalWritable := 'False'} : Bool;
      fb_Fifo_Instance { S7_SetPoint := 'True'} : "fb_Fifo";
      idx7 : Int;
      fb_Compress_Instance { S7_SetPoint := 'True'} : "fb_Compress";
      jammer_on { S7_SetPoint := 'True'} : TON_TIME;
      jammer : Bool;
      pusher_enable : Bool;
      Scale_done : Bool;
   END_VAR
   VAR RETAIN
      Lift_Table_UP { S7_SetPoint := 'True'} : CTU_INT;
   END_VAR
   VAR
      fb_Fifo_Instance_1 { S7_SetPoint := 'True'} : "fb_Fifo";
      fb_Compress_Instance_1 { S7_SetPoint := 'True'} : "fb_Compress";
      timer_1 { S7_SetPoint := 'True'} : TON_TIME;
   END_VAR
   VAR_TEMP
      temp : Int;
   END_VAR
   VAR_TEMP   // added for the SCL form of the ladder/FBD networks
      _w1 : Bool;
      _w2 : Bool;
   END_VAR
BEGIN

REGION Network 1
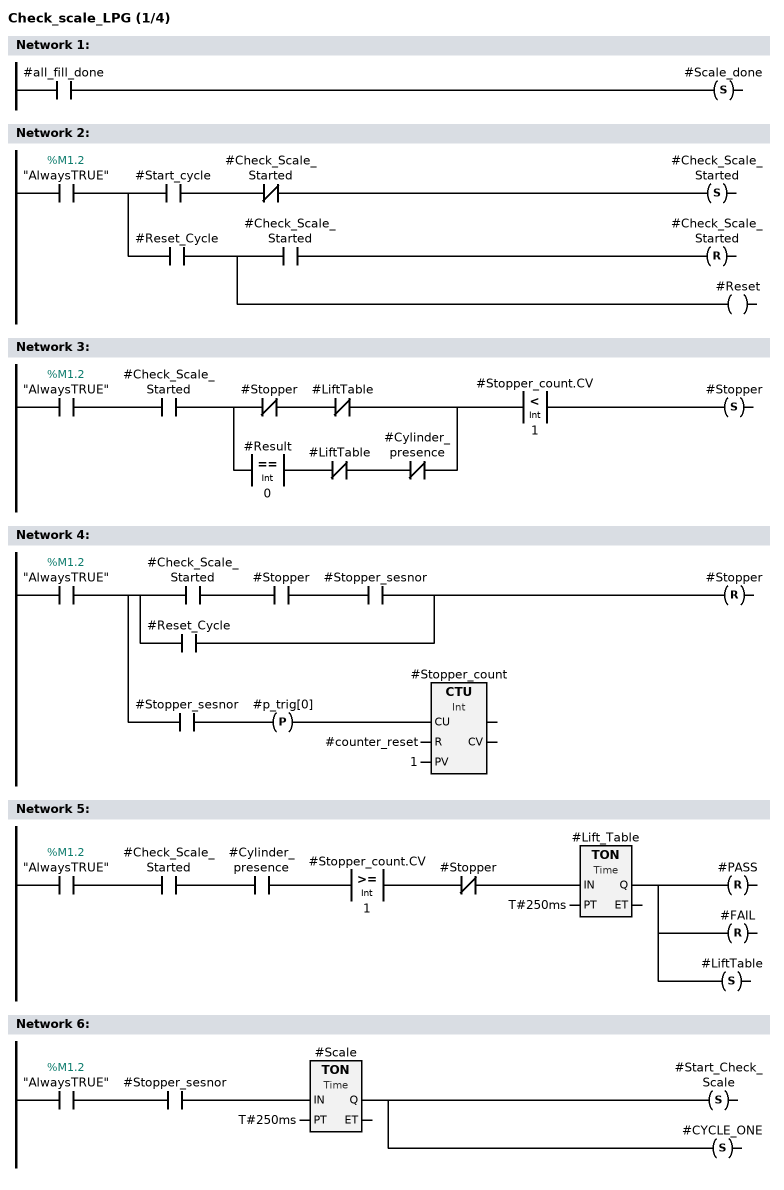
   RUNG wire#powerrail
      Contact( #all_fill_done )
      S_Coil( #Scale_done )
   END_RUNG
   // the same network as SCL:
   IF #all_fill_done THEN #Scale_done := TRUE; END_IF;
END_REGION

REGION Network 2
   RUNG wire#powerrail
      Contact( "AlwaysTRUE" )
      wire#w1
      Contact( #Start_cycle )
      I_Contact( #Check_Scale_Started )
      S_Coil( #Check_Scale_Started )
   END_RUNG
   RUNG wire#w1
      Contact( #Reset_Cycle )
      wire#w2
      Contact( #Check_Scale_Started )
      R_Coil( #Check_Scale_Started )
   END_RUNG
   RUNG wire#w2
      Coil( #Reset )
   END_RUNG
   // the same network as SCL:
   IF "AlwaysTRUE" AND #Start_cycle AND NOT #Check_Scale_Started THEN #Check_Scale_Started := TRUE; END_IF;
   #_w1 := "AlwaysTRUE" AND #Reset_Cycle;
   IF #_w1 AND #Check_Scale_Started THEN #Check_Scale_Started := FALSE; END_IF;
   #Reset := #_w1;
END_REGION

REGION Network 3
   RUNG wire#powerrail
      Contact( "AlwaysTRUE" )
      Contact( #Check_Scale_Started )
      wire#w1
      I_Contact( #Stopper )
      I_Contact( #LiftTable )
      wire#w2
      { S7_Templates := "SrcType := Int" } LT_Contact(in1 := #Stopper_count.CV, in2 := 1)
      S_Coil( #Stopper )
   END_RUNG
   RUNG wire#w1
      { S7_Templates := "SrcType := Int" } EQ_Contact(in1 := #Result, in2 := 0)
      I_Contact( #LiftTable )
      I_Contact( #Cylinder_presence )
   END_RUNG wire#w2
   // the same network as SCL:
   IF "AlwaysTRUE" AND #Check_Scale_Started AND ((NOT #Stopper AND NOT #LiftTable) OR ((#Result = 0) AND NOT #LiftTable AND NOT #Cylinder_presence)) AND (#Stopper_count.CV < 1) THEN
       #Stopper := TRUE;
   END_IF;
END_REGION

REGION Network 4
   RUNG wire#powerrail
      Contact( "AlwaysTRUE" )
      wire#w1
      Contact( #Check_Scale_Started )
      Contact( #Stopper )
      Contact( #Stopper_sesnor )
      wire#w2
      R_Coil( #Stopper )
   END_RUNG
   RUNG wire#w1
      Contact( #Reset_Cycle )
   END_RUNG wire#w2
   RUNG wire#w1
      Contact( #Stopper_sesnor )
      P_Trig( #p_trig[0] )
      { S7_Templates := "value_type := Int" } #Stopper_count.CTU(r := #counter_reset, pv := 1, cv =>)
   END_RUNG
   // the same network as SCL:
   IF "AlwaysTRUE" AND ((#Check_Scale_Started AND #Stopper AND #Stopper_sesnor) OR #Reset_Cycle) THEN
       #Stopper := FALSE;
   END_IF;
   #_w1 := "AlwaysTRUE" AND #Stopper_sesnor;
   #_w2 := #_w1 AND NOT #p_trig[0];   // rising edge
   #p_trig[0] := #_w1;
   #Stopper_count(CU := #_w2, R := #counter_reset, PV := 1);   // CTU
END_REGION

REGION Network 5
   RUNG wire#powerrail
      Contact( "AlwaysTRUE" )
      Contact( #Check_Scale_Started )
      Contact( #Cylinder_presence )
      { S7_Templates := "SrcType := Int" } GE_Contact(in1 := #Stopper_count.CV, in2 := 1)
      I_Contact( #Stopper )
      { S7_Templates := "time_type := Time" } #Lift_Table.TON(pt := T#250ms, et =>)
      wire#w1
      R_Coil( #PASS )
   END_RUNG
   RUNG wire#w1
      R_Coil( #FAIL )
   END_RUNG
   RUNG wire#w1
      S_Coil( #LiftTable )
   END_RUNG
   // the same network as SCL:
   #Lift_Table(IN := "AlwaysTRUE" AND #Check_Scale_Started AND #Cylinder_presence AND (#Stopper_count.CV >= 1) AND NOT #Stopper,   // TON
               PT := T#250ms);
   IF #Lift_Table.Q THEN
       #PASS := FALSE;
       #FAIL := FALSE;
       #LiftTable := TRUE;
   END_IF;
END_REGION

REGION Network 6
   RUNG wire#powerrail
      Contact( "AlwaysTRUE" )
      Contact( #Stopper_sesnor )
      { S7_Templates := "time_type := Time" } #Scale.TON(pt := T#250ms, et =>)
      wire#w1
      S_Coil( #Start_Check_Scale )
   END_RUNG
   RUNG wire#w1
      S_Coil( #CYCLE_ONE )
   END_RUNG
   // the same network as SCL:
   #Scale(IN := "AlwaysTRUE" AND #Stopper_sesnor, PT := T#250ms);   // TON
   IF #Scale.Q THEN
       #Start_Check_Scale := TRUE;
       #CYCLE_ONE := TRUE;
   END_IF;
END_REGION

REGION Network 7
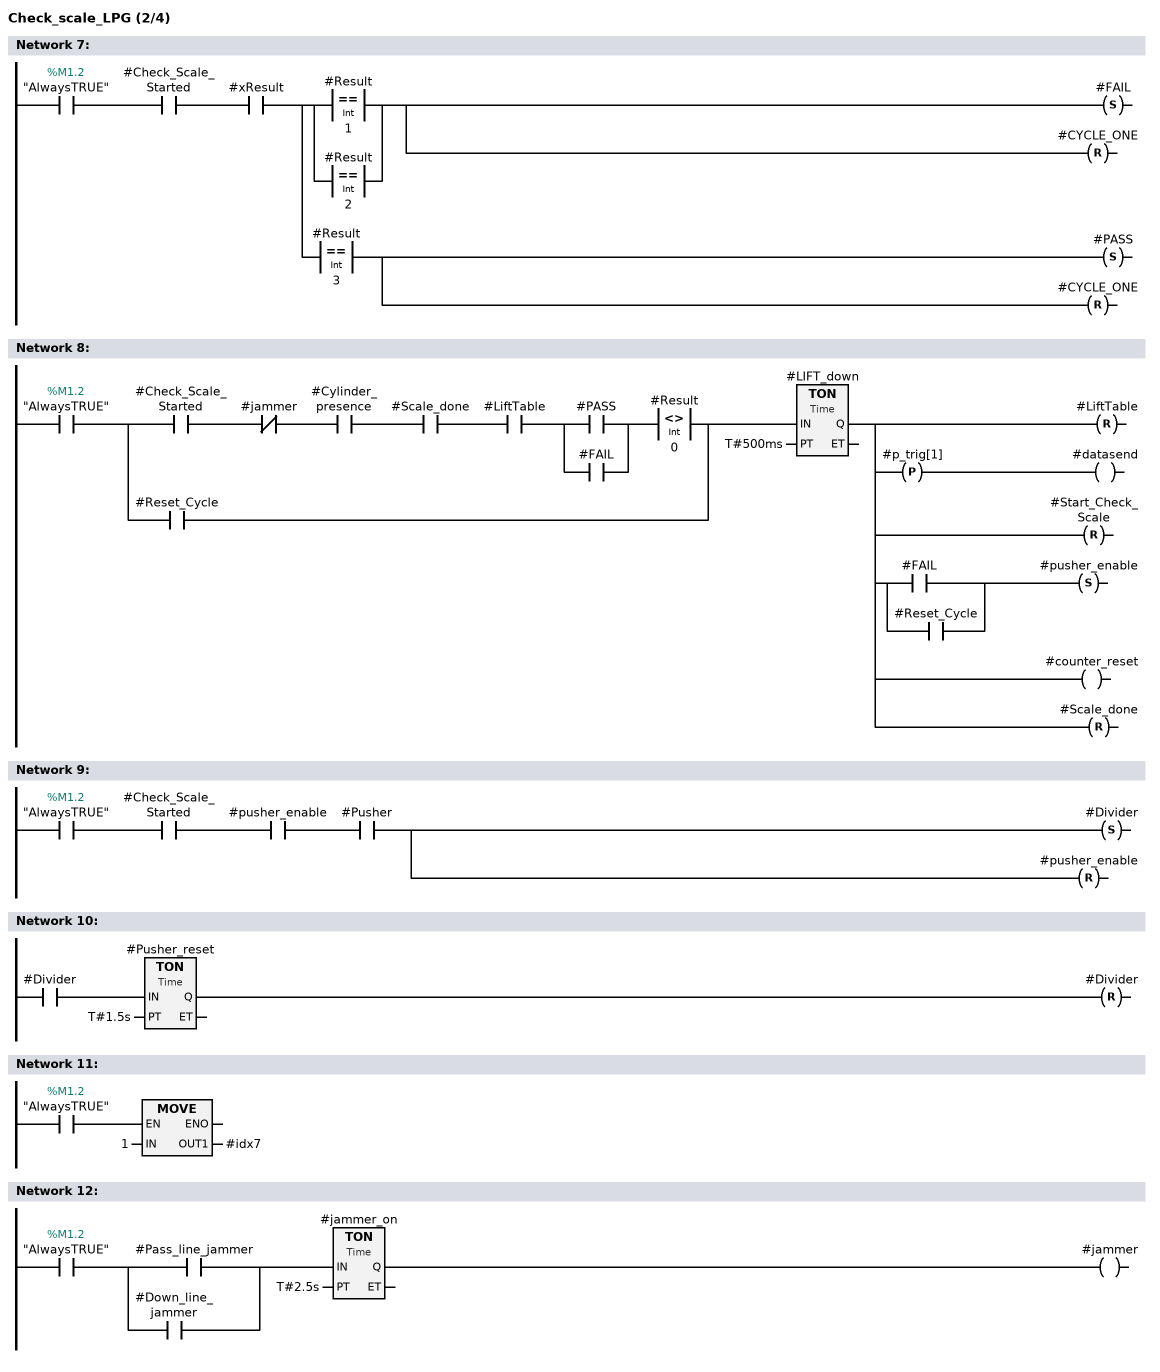
   RUNG wire#powerrail
      Contact( "AlwaysTRUE" )
      Contact( #Check_Scale_Started )
      Contact( #xResult )
      wire#w1
      { S7_Templates := "SrcType := Int" } EQ_Contact(in1 := #Result, in2 := 1)
      wire#w2
      S_Coil( #FAIL )
   END_RUNG
   RUNG wire#w1
      { S7_Templates := "SrcType := Int" } EQ_Contact(in1 := #Result, in2 := 2)
   END_RUNG wire#w2
   RUNG wire#w2
      R_Coil( #CYCLE_ONE )
   END_RUNG
   RUNG wire#w1
      { S7_Templates := "SrcType := Int" } EQ_Contact(in1 := #Result, in2 := 3)
      wire#w3
      S_Coil( #PASS )
   END_RUNG
   RUNG wire#w3
      R_Coil( #CYCLE_ONE )
   END_RUNG
   // the same network as SCL:
   #_w1 := "AlwaysTRUE" AND #Check_Scale_Started AND #xResult;
   IF #_w1 AND ((#Result = 1) OR (#Result = 2)) THEN
       #FAIL := TRUE;
       #CYCLE_ONE := FALSE;
   END_IF;
   IF #_w1 AND (#Result = 3) THEN
       #PASS := TRUE;
       #CYCLE_ONE := FALSE;
   END_IF;
END_REGION

REGION Network 8
   RUNG wire#powerrail
      Contact( "AlwaysTRUE" )
      wire#w1
      Contact( #Check_Scale_Started )
      I_Contact( #jammer )
      Contact( #Cylinder_presence )
      Contact( #Scale_done )
      Contact( #LiftTable )
      wire#w2
      Contact( #PASS )
      wire#w3
      { S7_Templates := "SrcType := Int" } NE_Contact(in1 := #Result, in2 := 0)
      wire#w4
      { S7_Templates := "time_type := Time" } #LIFT_down.TON(pt := T#500ms, et =>)
      wire#w5
      R_Coil( #LiftTable )
   END_RUNG
   RUNG wire#w2
      Contact( #FAIL )
   END_RUNG wire#w3
   RUNG wire#w1
      Contact( #Reset_Cycle )
   END_RUNG wire#w4
   RUNG wire#w5
      P_Trig( #p_trig[1] )
      Coil( #datasend )
   END_RUNG
   RUNG wire#w5
      R_Coil( #Start_Check_Scale )
   END_RUNG
   RUNG wire#w5
      Contact( #FAIL )
      wire#w6
      S_Coil( #pusher_enable )
   END_RUNG
   RUNG wire#w5
      Contact( #Reset_Cycle )
   END_RUNG wire#w6
   RUNG wire#w5
      Coil( #counter_reset )
   END_RUNG
   RUNG wire#w5
      R_Coil( #Scale_done )
   END_RUNG
   // the same network as SCL:
   #LIFT_down(IN := "AlwaysTRUE" AND ((#Check_Scale_Started AND NOT #jammer AND #Cylinder_presence AND #Scale_done AND #LiftTable AND (#PASS OR #FAIL) AND (#Result <> 0)) OR #Reset_Cycle),   // TON
              PT := T#500ms);
   IF #LIFT_down.Q THEN #LiftTable := FALSE; END_IF;
   #_w1 := #LIFT_down.Q AND NOT #p_trig[1];   // rising edge
   #p_trig[1] := #LIFT_down.Q;
   #datasend := #_w1;
   IF #LIFT_down.Q THEN #Start_Check_Scale := FALSE; END_IF;
   IF #LIFT_down.Q AND (#FAIL OR #Reset_Cycle) THEN #pusher_enable := TRUE; END_IF;
   #counter_reset := #LIFT_down.Q;
   IF #LIFT_down.Q THEN #Scale_done := FALSE; END_IF;
END_REGION

REGION Network 9
   RUNG wire#powerrail
      Contact( "AlwaysTRUE" )
      Contact( #Check_Scale_Started )
      Contact( #pusher_enable )
      Contact( #Pusher )
      wire#w1
      S_Coil( #Divider )
   END_RUNG
   RUNG wire#w1
      R_Coil( #pusher_enable )
   END_RUNG
   // the same network as SCL:
   IF "AlwaysTRUE" AND #Check_Scale_Started AND #pusher_enable AND #Pusher THEN
       #Divider := TRUE;
       #pusher_enable := FALSE;
   END_IF;
END_REGION

REGION Network 10
   RUNG wire#powerrail
      Contact( #Divider )
      { S7_Templates := "time_type := Time" } #Pusher_reset.TON(pt := T#1.5s, et =>)
      R_Coil( #Divider )
   END_RUNG
   // the same network as SCL:
   #Pusher_reset(IN := #Divider, PT := T#1.5s);   // TON
   IF #Pusher_reset.Q THEN #Divider := FALSE; END_IF;
END_REGION

REGION Network 11
   RUNG wire#powerrail
      Contact( "AlwaysTRUE" )
      Move(in := 1, out1 => #idx7)
   END_RUNG
   // the same network as SCL:
   IF "AlwaysTRUE" THEN #idx7 := 1; END_IF;
END_REGION

REGION Network 12
   RUNG wire#powerrail
      Contact( "AlwaysTRUE" )
      wire#w1
      Contact( #Pass_line_jammer )
      wire#w2
      { S7_Templates := "time_type := Time" } #jammer_on.TON(pt := T#2.5s, et =>)
      Coil( #jammer )
   END_RUNG
   RUNG wire#w1
      Contact( #Down_line_jammer )
   END_RUNG wire#w2
   // the same network as SCL:
   #jammer_on(IN := "AlwaysTRUE" AND (#Pass_line_jammer OR #Down_line_jammer), PT := T#2.5s);   // TON
   #jammer := #jammer_on.Q;
END_REGION

REGION Network 13: cylinder FAIL
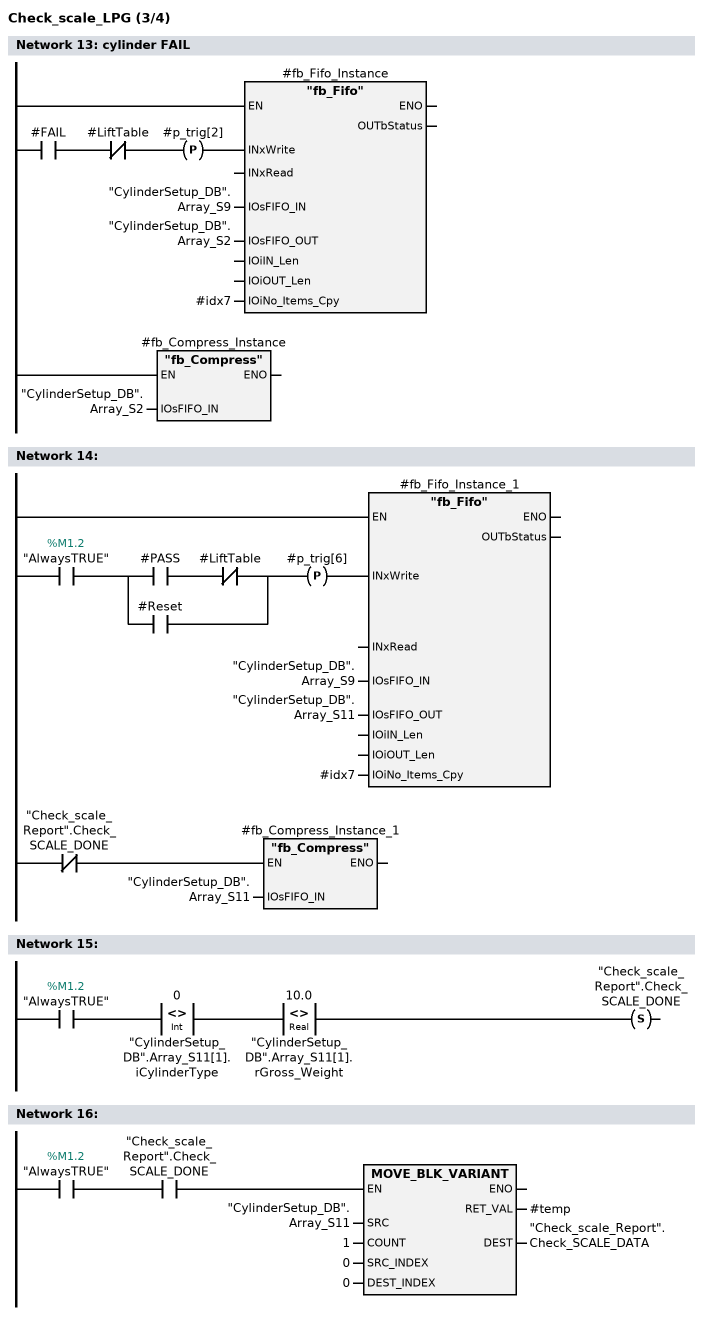
   RUNG wire#powerrail
      #fb_Fifo_Instance(INxWrite := wire#w1, INxRead :=, IOsFIFO_IN := "CylinderSetup_DB".Array_S9, IOsFIFO_OUT := "CylinderSetup_DB".Array_S2, IOiIN_Len :=, IOiOUT_Len :=, IOiNo_Items_Cpy := #idx7, OUTbStatus =>)
   END_RUNG
   RUNG wire#powerrail
      Contact( #FAIL )
      I_Contact( #LiftTable )
      P_Trig( #p_trig[2] )
   END_RUNG wire#w1
   RUNG wire#powerrail
      #fb_Compress_Instance(IOsFIFO_IN := "CylinderSetup_DB".Array_S2)
   END_RUNG
   // the same network as SCL:
   #_w1 := #FAIL AND NOT #LiftTable;
   #_w2 := #_w1 AND NOT #p_trig[2];   // rising edge
   #p_trig[2] := #_w1;
   #fb_Fifo_Instance(INxWrite := #_w2,   // "fb_Fifo"
                     IOsFIFO_IN := "CylinderSetup_DB".Array_S9,
                     IOsFIFO_OUT := "CylinderSetup_DB".Array_S2,
                     IOiNo_Items_Cpy := #idx7);
   #fb_Compress_Instance(IOsFIFO_IN := "CylinderSetup_DB".Array_S2);   // "fb_Compress"
END_REGION

REGION Network 14
   RUNG wire#powerrail
      #fb_Fifo_Instance_1(INxWrite := wire#w3, INxRead :=, IOsFIFO_IN := "CylinderSetup_DB".Array_S9, IOsFIFO_OUT := "CylinderSetup_DB".Array_S11, IOiIN_Len :=, IOiOUT_Len :=, IOiNo_Items_Cpy := #idx7, OUTbStatus =>)
   END_RUNG
   RUNG wire#powerrail
      Contact( "AlwaysTRUE" )
      wire#w1
      Contact( #PASS )
      I_Contact( #LiftTable )
      wire#w2
      P_Trig( #p_trig[6] )
   END_RUNG wire#w3
   RUNG wire#w1
      Contact( #Reset )
   END_RUNG wire#w2
   RUNG wire#powerrail
      I_Contact( "Check_scale_Report".Check_SCALE_DONE )
      #fb_Compress_Instance_1(IOsFIFO_IN := "CylinderSetup_DB".Array_S11)
   END_RUNG
   // the same network as SCL:
   #_w1 := "AlwaysTRUE" AND ((#PASS AND NOT #LiftTable) OR #Reset);
   #_w2 := #_w1 AND NOT #p_trig[6];   // rising edge
   #p_trig[6] := #_w1;
   #fb_Fifo_Instance_1(INxWrite := #_w2,   // "fb_Fifo"
                       IOsFIFO_IN := "CylinderSetup_DB".Array_S9,
                       IOsFIFO_OUT := "CylinderSetup_DB".Array_S11,
                       IOiNo_Items_Cpy := #idx7);
   IF NOT "Check_scale_Report".Check_SCALE_DONE THEN
       #fb_Compress_Instance_1(IOsFIFO_IN := "CylinderSetup_DB".Array_S11);   // "fb_Compress"
   END_IF;
END_REGION

REGION Network 15
   RUNG wire#powerrail
      Contact( "AlwaysTRUE" )
      { S7_Templates := "SrcType := Int" } NE_Contact(in1 := 0, in2 := "CylinderSetup_DB".Array_S11[1].iCylinderType)
      { S7_Templates := "SrcType := Real" } NE_Contact(in1 := 10.0, in2 := "CylinderSetup_DB".Array_S11[1].rGross_Weight)
      S_Coil( "Check_scale_Report".Check_SCALE_DONE )
   END_RUNG
   // the same network as SCL:
   IF "AlwaysTRUE" AND (0 <> "CylinderSetup_DB".Array_S11[1].iCylinderType) AND (10.0 <> "CylinderSetup_DB".Array_S11[1].rGross_Weight) THEN
       "Check_scale_Report".Check_SCALE_DONE := TRUE;
   END_IF;
END_REGION

REGION Network 16
   RUNG wire#powerrail
      Contact( "AlwaysTRUE" )
      Contact( "Check_scale_Report".Check_SCALE_DONE )
      MOVE_BLK_VARIANT(SRC := "CylinderSetup_DB".Array_S11, COUNT := 1, SRC_INDEX := 0, DEST_INDEX := 0, Ret_Val => #temp, DEST => "Check_scale_Report".Check_SCALE_DATA)
   END_RUNG
   // the same network as SCL:
   IF "AlwaysTRUE" AND "Check_scale_Report".Check_SCALE_DONE THEN
       #temp := MOVE_BLK_VARIANT(SRC := "CylinderSetup_DB".Array_S11,
                               COUNT := 1,
                               SRC_INDEX := 0,
                               DEST_INDEX := 0,
                               DEST => "Check_scale_Report".Check_SCALE_DATA);
   END_IF;
END_REGION

REGION Network 17
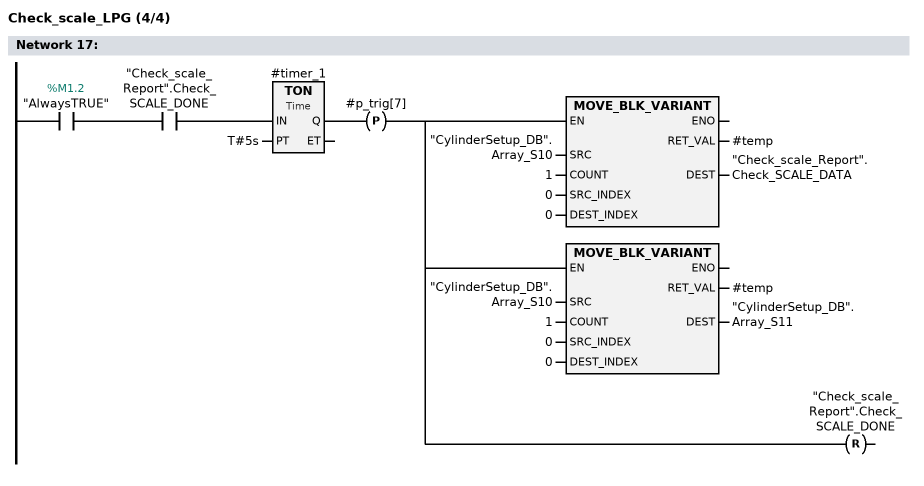
   RUNG wire#powerrail
      Contact( "AlwaysTRUE" )
      Contact( "Check_scale_Report".Check_SCALE_DONE )
      { S7_Templates := "time_type := Time" } #timer_1.TON(pt := T#5s, et =>)
      P_Trig( #p_trig[7] )
      wire#w1
      MOVE_BLK_VARIANT(SRC := "CylinderSetup_DB".Array_S10, COUNT := 1, SRC_INDEX := 0, DEST_INDEX := 0, Ret_Val => #temp, DEST => "Check_scale_Report".Check_SCALE_DATA)
   END_RUNG
   RUNG wire#w1
      MOVE_BLK_VARIANT(SRC := "CylinderSetup_DB".Array_S10, COUNT := 1, SRC_INDEX := 0, DEST_INDEX := 0, Ret_Val => #temp, DEST => "CylinderSetup_DB".Array_S11)
   END_RUNG
   RUNG wire#w1
      R_Coil( "Check_scale_Report".Check_SCALE_DONE )
   END_RUNG
   // the same network as SCL:
   #timer_1(IN := "AlwaysTRUE" AND "Check_scale_Report".Check_SCALE_DONE, PT := T#5s);   // TON
   #_w1 := #timer_1.Q AND NOT #p_trig[7];   // rising edge
   #p_trig[7] := #timer_1.Q;
   IF #_w1 THEN
       #temp := MOVE_BLK_VARIANT(SRC := "CylinderSetup_DB".Array_S10,
                               COUNT := 1,
                               SRC_INDEX := 0,
                               DEST_INDEX := 0,
                               DEST => "Check_scale_Report".Check_SCALE_DATA);
       #temp := MOVE_BLK_VARIANT(SRC := "CylinderSetup_DB".Array_S10,
                               COUNT := 1,
                               SRC_INDEX := 0,
                               DEST_INDEX := 0,
                               DEST => "CylinderSetup_DB".Array_S11);
       "Check_scale_Report".Check_SCALE_DONE := FALSE;
   END_IF;
END_REGION
END_FUNCTION_BLOCK

FUNCTION_BLOCK "LPG_Check_scale_FB"   // FB102, LAD
TITLE = Fiiling Operation FB
{ S7_Optimized_Access := 'TRUE' }
VERSION : 0.1
// stored: AutoNumber false, IsIECCheckEnabled false, IsRetainMemResEnabled false, MemoryReserve 100, SetENOAutomatically false, UDAEnableTagReadback false
   VAR_INPUT
      INxCylinder_In_Pos : Bool;   // Cylinder In Position
      INxAuto_Start_Seq : Bool;   // Start Filling Sequence
      INxMan_Start_Seq : Bool;
      INxStop_Sequence : Bool;   // Stop Filling Sequence
      INtStart_TImeout_Time : DInt;   // Start Timeout Time in Sec
      INxReset_Sequence : Bool;   // Reset Sequence
      INxCylinder_Type : Int;
      INrTare_Entry_SP : Real;
      DOWN_CONVEYOR : Bool;
      data_delete : Bool;
   END_VAR
   VAR_OUTPUT
      OutuFilled_Data : Array[1..10] of Real;
      OutxDomestic_Cylinder : Bool;
      OutxCommercial_Cylinder : Bool;
      OutxStart_Timeout : Bool;
      OutxTare_Entry_Error : Bool;   // Coil 27
      Outx_Filling_Error : Bool;
      Outx_Tare_Value_Error : Bool;
      Cycle_Started : Bool;
      OutiStep_No : Int;
      OUTiResult : Int;
      Gross_Weight : Real;
      Net_Wieght : Real;
      Tare_Weight : Real;
      OUT_Decision : Int;
   END_VAR
   VAR_IN_OUT
      Modbus_Master_DB : "MOD_MASTER_DATA_1";
   END_VAR
   VAR
      TRIG : Array[1..25] of Bool;
      STEP_NO : Int;
      Step_Timer { S7_SetPoint := 'True'} : Array[1..15] of IEC_TIMER;
      Domestic_Cylinder { S7_SetPoint := 'True'} : Bool;
      Commercial_Cylinder : Bool;
      Cyl_Done { S7_SetPoint := 'True'} : TOF_TIME;
      Tare_Enrty_Extn { S7_SetPoint := 'True'} : TOF_TIME;
      Start_Timeout_Err { S7_SetPoint := 'True'} : TON_TIME;
      Tare_Entry_Timer { S7_SetPoint := 'True'} : TON_TIME;
      Filled_Gross : Real;
      Filled_Net : Real;
      Punched_Tare : Real;
      Test_Seq : Int;
      RESULT : Bool;
      IEC_Timer_0_Instance { S7_SetPoint := 'True'} : TOF_TIME;
      Gross { S7_SetPoint := 'True'} : Real;
      gross_diff : Real;
      pass : Bool;
      Decision : Word;
      IEC_Timer_0_Instance_1 { S7_SetPoint := 'True'} : TON_TIME;
      fill { S7_SetPoint := 'True'} : TON_TIME;
      ALL_FILL_DONE : Bool;
   END_VAR
   VAR RETAIN
      cycle_start { S7_SetPoint := 'True'} : CTU_INT;
   END_VAR
   VAR_TEMP
      Tare_Weight_Mul : Real;
      Tare_Enter_Time : DInt;
      Stt_TImeout_Time : DInt;
      Tare_Entry_Time : DInt;
      Tare_SP_Weigher : Int;
      Filled_Gross_Mul : Int;
      Filled_Net_Mul : Int;
      Filled_Tare_Mul : Int;
      "final wieght" : Real;
      final_weight_1 : Real;
   END_VAR
   // Tare_Enrty_Extn.PT := T#1s;
   VAR_TEMP   // added for the SCL form of the ladder/FBD networks
      _w1 : Bool;
      _w2 : Bool;
      _w3 : Bool;
   END_VAR
BEGIN

REGION Network 1: Empty Network
END_REGION

REGION Network 2: Input Mapping
END_REGION

